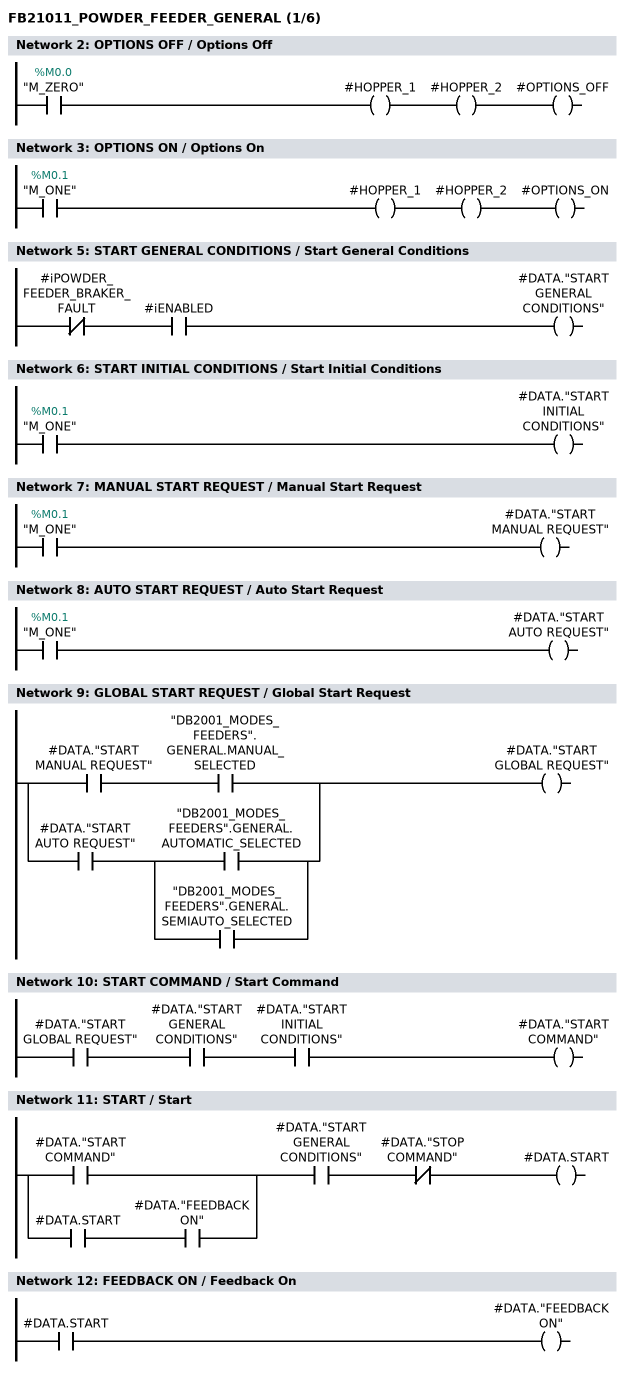
   RUNG wire#powerrail
      Contact( "M_ZERO" )
      Coil( #HOPPER_1 )
      Coil( #HOPPER_2 )
      Coil( #OPTIONS_OFF )
   END_RUNG
   // the same network as SCL:
   #HOPPER_1 := "M_ZERO";
   #HOPPER_2 := "M_ZERO";
   #OPTIONS_OFF := "M_ZERO";
END_REGION

REGION Network 3: OPTIONS ON / Options On
   RUNG wire#powerrail
      Contact( "M_ONE" )
      Coil( #HOPPER_1 )
      Coil( #HOPPER_2 )
      Coil( #OPTIONS_ON )
   END_RUNG
   // the same network as SCL:
   #HOPPER_1 := "M_ONE";
   #HOPPER_2 := "M_ONE";
   #OPTIONS_ON := "M_ONE";
END_REGION

REGION Network 4: INPUT / Input
END_REGION

REGION Network 5: START GENERAL CONDITIONS / Start General Conditions
   RUNG wire#powerrail
      I_Contact( #iPOWDER_FEEDER_BRAKER_FAULT )
      Contact( #iENABLED )
      Coil( #DATA."START GENERAL CONDITIONS" )
   END_RUNG
   // the same network as SCL:
   #DATA."START GENERAL CONDITIONS" := NOT #iPOWDER_FEEDER_BRAKER_FAULT AND #iENABLED;
END_REGION

REGION Network 6: START INITIAL CONDITIONS / Start Initial Conditions
   RUNG wire#powerrail
      Contact( "M_ONE" )
      Coil( #DATA."START INITIAL CONDITIONS" )
   END_RUNG
   // the same network as SCL:
   #DATA."START INITIAL CONDITIONS" := "M_ONE";
END_REGION

REGION Network 7: MANUAL START REQUEST / Manual Start Request
   RUNG wire#powerrail
      Contact( "M_ONE" )
      Coil( #DATA."START MANUAL REQUEST" )
   END_RUNG
   // the same network as SCL:
   #DATA."START MANUAL REQUEST" := "M_ONE";
END_REGION

REGION Network 8: AUTO START REQUEST / Auto Start Request
   RUNG wire#powerrail
      Contact( "M_ONE" )
      Coil( #DATA."START AUTO REQUEST" )
   END_RUNG
   // the same network as SCL:
   #DATA."START AUTO REQUEST" := "M_ONE";
END_REGION

REGION Network 9: GLOBAL START REQUEST / Global Start Request
   RUNG wire#powerrail
      Contact( #DATA."START MANUAL REQUEST" )
      Contact( "DB2001_MODES_FEEDERS".GENERAL.MANUAL_SELECTED )
      wire#w1
      Coil( #DATA."START GLOBAL REQUEST" )
   END_RUNG
   RUNG wire#powerrail
      Contact( #DATA."START AUTO REQUEST" )
      wire#w2
      Contact( "DB2001_MODES_FEEDERS".GENERAL.AUTOMATIC_SELECTED )
   END_RUNG wire#w1
   RUNG wire#w2
      Contact( "DB2001_MODES_FEEDERS".GENERAL.SEMIAUTO_SELECTED )
   END_RUNG wire#w1
   // the same network as SCL:
   #DATA."START GLOBAL REQUEST" := (#DATA."START MANUAL REQUEST" AND "DB2001_MODES_FEEDERS".GENERAL.MANUAL_SELECTED) OR (#DATA."START AUTO REQUEST" AND ("DB2001_MODES_FEEDERS".GENERAL.AUTOMATIC_SELECTED OR "DB2001_MODES_FEEDERS".GENERAL.SEMIAUTO_SELECTED));
END_REGION

REGION Network 10: START COMMAND / Start Command
   RUNG wire#powerrail
      Contact( #DATA."START GLOBAL REQUEST" )
      Contact( #DATA."START GENERAL CONDITIONS" )
      Contact( #DATA."START INITIAL CONDITIONS" )
      Coil( #DATA."START COMMAND" )
   END_RUNG
   // the same network as SCL:
   #DATA."START COMMAND" := #DATA."START GLOBAL REQUEST" AND #DATA."START GENERAL CONDITIONS" AND #DATA."START INITIAL CONDITIONS";
END_REGION

REGION Network 11: START / Start
   RUNG wire#powerrail
      Contact( #DATA."START COMMAND" )
      wire#w1
      Contact( #DATA."START GENERAL CONDITIONS" )
      I_Contact( #DATA."STOP COMMAND" )
      Coil( #DATA.START )
   END_RUNG
   RUNG wire#powerrail
      Contact( #DATA.START )
      Contact( #DATA."FEEDBACK ON" )
   END_RUNG wire#w1
   // the same network as SCL:
   #DATA.START := (#DATA."START COMMAND" OR (#DATA.START AND #DATA."FEEDBACK ON")) AND #DATA."START GENERAL CONDITIONS" AND NOT #DATA."STOP COMMAND";
END_REGION

REGION Network 12: FEEDBACK ON / Feedback On
   RUNG wire#powerrail
      Contact( #DATA.START )
      Coil( #DATA."FEEDBACK ON" )
   END_RUNG
   // the same network as SCL:
   #DATA."FEEDBACK ON" := #DATA.START;
END_REGION

REGION Network 13: STOP GENERAL CONDITIONS / Stop General Conditions
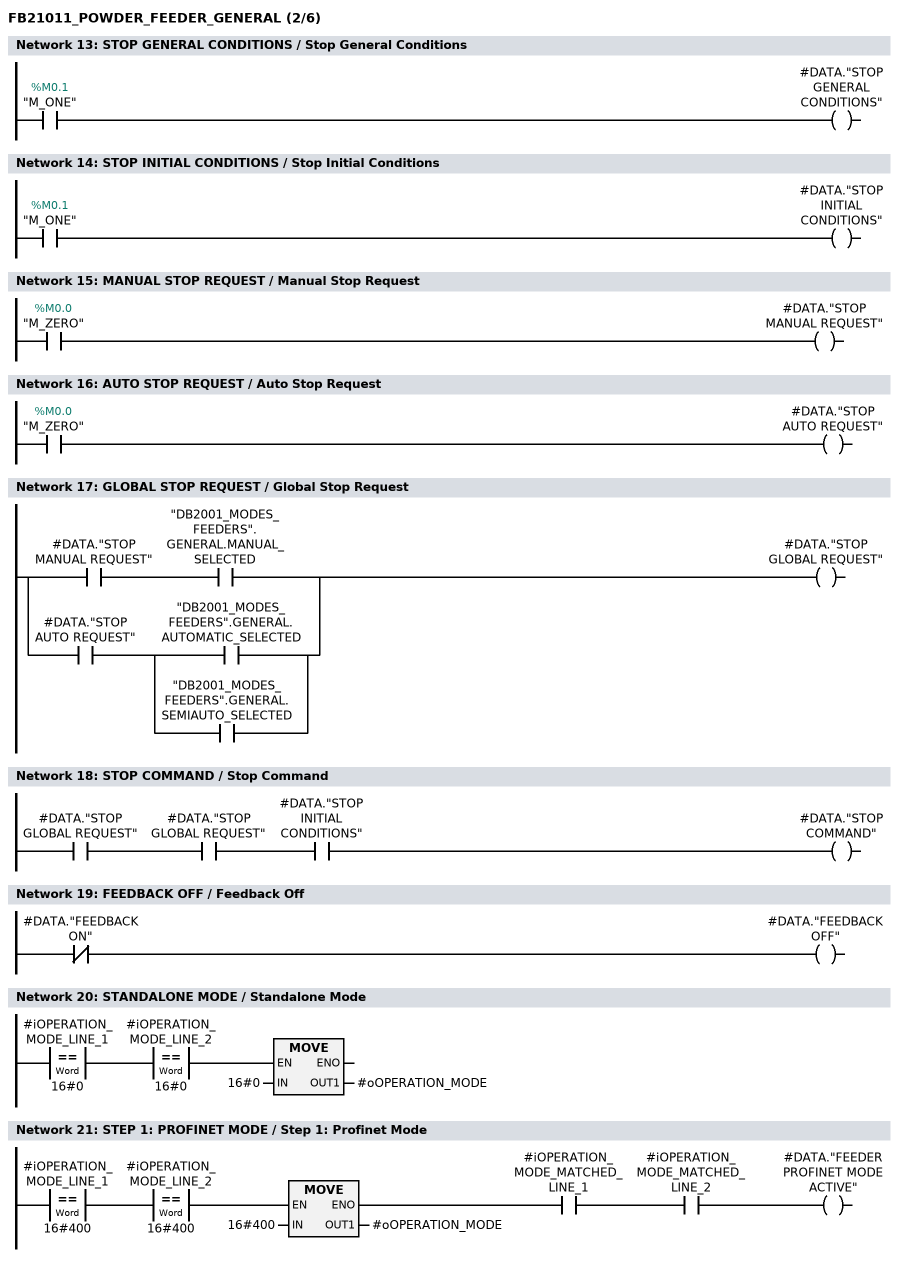
   RUNG wire#powerrail
      Contact( "M_ONE" )
      Coil( #DATA."STOP GENERAL CONDITIONS" )
   END_RUNG
   // the same network as SCL:
   #DATA."STOP GENERAL CONDITIONS" := "M_ONE";
END_REGION

REGION Network 14: STOP INITIAL CONDITIONS / Stop Initial Conditions
   RUNG wire#powerrail
      Contact( "M_ONE" )
      Coil( #DATA."STOP INITIAL CONDITIONS" )
   END_RUNG
   // the same network as SCL:
   #DATA."STOP INITIAL CONDITIONS" := "M_ONE";
END_REGION

REGION Network 15: MANUAL STOP REQUEST / Manual Stop Request
   RUNG wire#powerrail
      Contact( "M_ZERO" )
      Coil( #DATA."STOP MANUAL REQUEST" )
   END_RUNG
   // the same network as SCL:
   #DATA."STOP MANUAL REQUEST" := "M_ZERO";
END_REGION

REGION Network 16: AUTO STOP REQUEST / Auto Stop Request
   RUNG wire#powerrail
      Contact( "M_ZERO" )
      Coil( #DATA."STOP AUTO REQUEST" )
   END_RUNG
   // the same network as SCL:
   #DATA."STOP AUTO REQUEST" := "M_ZERO";
END_REGION

REGION Network 17: GLOBAL STOP REQUEST / Global Stop Request
   RUNG wire#powerrail
      Contact( #DATA."STOP MANUAL REQUEST" )
      Contact( "DB2001_MODES_FEEDERS".GENERAL.MANUAL_SELECTED )
      wire#w1
      Coil( #DATA."STOP GLOBAL REQUEST" )
   END_RUNG
   RUNG wire#powerrail
      Contact( #DATA."STOP AUTO REQUEST" )
      wire#w2
      Contact( "DB2001_MODES_FEEDERS".GENERAL.AUTOMATIC_SELECTED )
   END_RUNG wire#w1
   RUNG wire#w2
      Contact( "DB2001_MODES_FEEDERS".GENERAL.SEMIAUTO_SELECTED )
   END_RUNG wire#w1
   // the same network as SCL:
   #DATA."STOP GLOBAL REQUEST" := (#DATA."STOP MANUAL REQUEST" AND "DB2001_MODES_FEEDERS".GENERAL.MANUAL_SELECTED) OR (#DATA."STOP AUTO REQUEST" AND ("DB2001_MODES_FEEDERS".GENERAL.AUTOMATIC_SELECTED OR "DB2001_MODES_FEEDERS".GENERAL.SEMIAUTO_SELECTED));
END_REGION

REGION Network 18: STOP COMMAND / Stop Command
   RUNG wire#powerrail
      Contact( #DATA."STOP GLOBAL REQUEST" )
      Contact( #DATA."STOP GLOBAL REQUEST" )
      Contact( #DATA."STOP INITIAL CONDITIONS" )
      Coil( #DATA."STOP COMMAND" )
   END_RUNG
   // the same network as SCL:
   #DATA."STOP COMMAND" := #DATA."STOP GLOBAL REQUEST" AND #DATA."STOP GLOBAL REQUEST" AND #DATA."STOP INITIAL CONDITIONS";
END_REGION

REGION Network 19: FEEDBACK OFF / Feedback Off
   RUNG wire#powerrail
      I_Contact( #DATA."FEEDBACK ON" )
      Coil( #DATA."FEEDBACK OFF" )
   END_RUNG
   // the same network as SCL:
   #DATA."FEEDBACK OFF" := NOT #DATA."FEEDBACK ON";
END_REGION

REGION Network 20: STANDALONE MODE / Standalone Mode
   RUNG wire#powerrail
      { S7_Templates := "SrcType := Word" } EQ_Contact(in1 := #iOPERATION_MODE_LINE_1, in2 := 16#0)
      { S7_Templates := "SrcType := Word" } EQ_Contact(in1 := #iOPERATION_MODE_LINE_2, in2 := 16#0)
      Move(in := 16#0, out1 => #oOPERATION_MODE)
   END_RUNG
   // the same network as SCL:
   IF (#iOPERATION_MODE_LINE_1 = 16#0) AND (#iOPERATION_MODE_LINE_2 = 16#0) THEN
       #oOPERATION_MODE := 16#0;
   END_IF;
END_REGION

REGION Network 21: STEP 1: PROFINET MODE / Step 1: Profinet Mode
   RUNG wire#powerrail
      { S7_Templates := "SrcType := Word" } EQ_Contact(in1 := #iOPERATION_MODE_LINE_1, in2 := 16#400)
      { S7_Templates := "SrcType := Word" } EQ_Contact(in1 := #iOPERATION_MODE_LINE_2, in2 := 16#400)
      Move(in := 16#400, out1 => #oOPERATION_MODE)
      Contact( #iOPERATION_MODE_MATCHED_LINE_1 )
      Contact( #iOPERATION_MODE_MATCHED_LINE_2 )
      Coil( #DATA."FEEDER PROFINET MODE ACTIVE" )
   END_RUNG
   // the same network as SCL:
   #_w1 := (#iOPERATION_MODE_LINE_1 = 16#400) AND (#iOPERATION_MODE_LINE_2 = 16#400);
   IF #_w1 THEN #oOPERATION_MODE := 16#400; END_IF;
   #DATA."FEEDER PROFINET MODE ACTIVE" := #_w1 AND #iOPERATION_MODE_MATCHED_LINE_1 AND #iOPERATION_MODE_MATCHED_LINE_2;
END_REGION

REGION Network 22: STEP 2: PRODUCTION MODE / Step 2: Production Mode
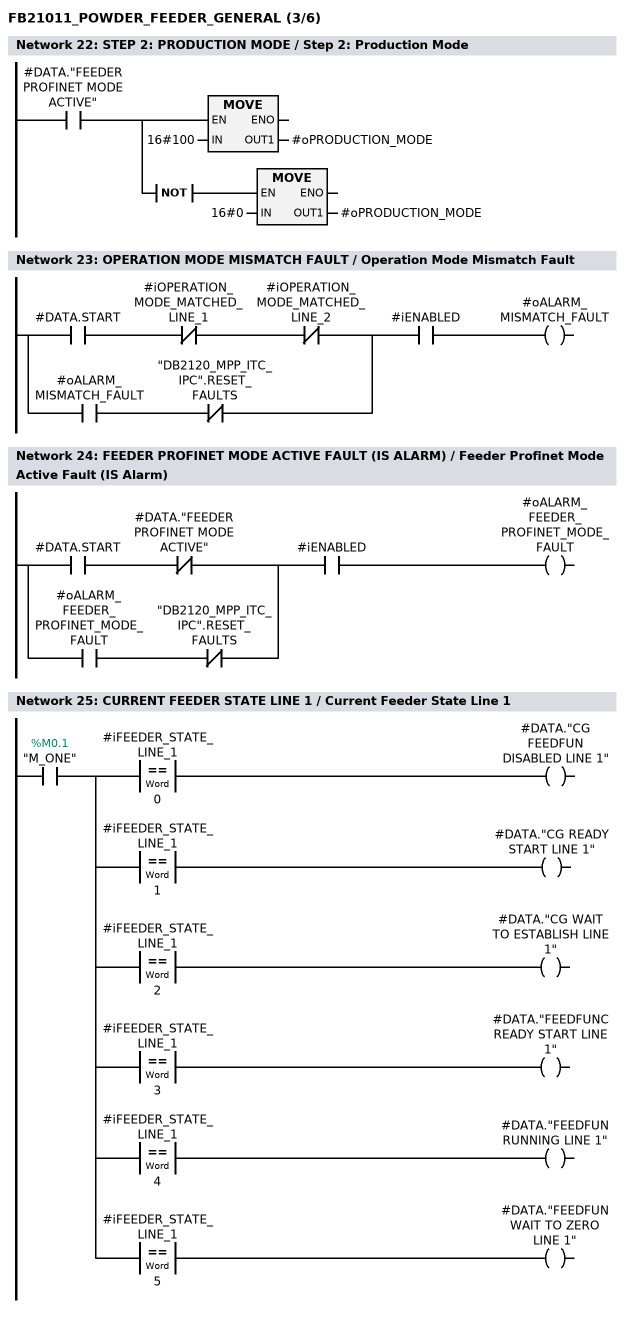
   RUNG wire#powerrail
      Contact( #DATA."FEEDER PROFINET MODE ACTIVE" )
      wire#w1
      Move(in := 16#100, out1 => #oPRODUCTION_MODE)
   END_RUNG
   RUNG wire#w1
      Not()
      Move(in := 16#0, out1 => #oPRODUCTION_MODE)
   END_RUNG
   // the same network as SCL:
   IF #DATA."FEEDER PROFINET MODE ACTIVE" THEN #oPRODUCTION_MODE := 16#100; END_IF;
   IF NOT #DATA."FEEDER PROFINET MODE ACTIVE" THEN #oPRODUCTION_MODE := 16#0; END_IF;
END_REGION

REGION Network 23: OPERATION MODE MISMATCH FAULT / Operation Mode Mismatch Fault
   RUNG wire#powerrail
      Contact( #DATA.START )
      I_Contact( #iOPERATION_MODE_MATCHED_LINE_1 )
      I_Contact( #iOPERATION_MODE_MATCHED_LINE_2 )
      wire#w1
      Contact( #iENABLED )
      Coil( #oALARM_MISMATCH_FAULT )
   END_RUNG
   RUNG wire#powerrail
      Contact( #oALARM_MISMATCH_FAULT )
      I_Contact( "DB2120_MPP_ITC_IPC".RESET_FAULTS )
   END_RUNG wire#w1
   // the same network as SCL:
   #oALARM_MISMATCH_FAULT := ((#DATA.START AND NOT #iOPERATION_MODE_MATCHED_LINE_1 AND NOT #iOPERATION_MODE_MATCHED_LINE_2) OR (#oALARM_MISMATCH_FAULT AND NOT "DB2120_MPP_ITC_IPC".RESET_FAULTS)) AND #iENABLED;
END_REGION

REGION Network 24: FEEDER PROFINET MODE ACTIVE FAULT (IS ALARM) / Feeder Profinet Mode Active Fault (IS Alarm)
   RUNG wire#powerrail
      Contact( #DATA.START )
      I_Contact( #DATA."FEEDER PROFINET MODE ACTIVE" )
      wire#w1
      Contact( #iENABLED )
      Coil( #oALARM_FEEDER_PROFINET_MODE_FAULT )
   END_RUNG
   RUNG wire#powerrail
      Contact( #oALARM_FEEDER_PROFINET_MODE_FAULT )
      I_Contact( "DB2120_MPP_ITC_IPC".RESET_FAULTS )
   END_RUNG wire#w1
   // the same network as SCL:
   #oALARM_FEEDER_PROFINET_MODE_FAULT := ((#DATA.START AND NOT #DATA."FEEDER PROFINET MODE ACTIVE") OR (#oALARM_FEEDER_PROFINET_MODE_FAULT AND NOT "DB2120_MPP_ITC_IPC".RESET_FAULTS)) AND #iENABLED;
END_REGION

REGION Network 25: CURRENT FEEDER STATE LINE 1 / Current Feeder State Line 1
   RUNG wire#powerrail
      Contact( "M_ONE" )
      wire#w1
      { S7_Templates := "SrcType := Word" } EQ_Contact(in1 := #iFEEDER_STATE_LINE_1, in2 := 0)
      Coil( #DATA."CG FEEDFUN DISABLED LINE 1" )
   END_RUNG
   RUNG wire#w1
      { S7_Templates := "SrcType := Word" } EQ_Contact(in1 := #iFEEDER_STATE_LINE_1, in2 := 1)
      Coil( #DATA."CG READY START LINE 1" )
   END_RUNG
   RUNG wire#w1
      { S7_Templates := "SrcType := Word" } EQ_Contact(in1 := #iFEEDER_STATE_LINE_1, in2 := 2)
      Coil( #DATA."CG WAIT TO ESTABLISH LINE 1" )
   END_RUNG
   RUNG wire#w1
      { S7_Templates := "SrcType := Word" } EQ_Contact(in1 := #iFEEDER_STATE_LINE_1, in2 := 3)
      Coil( #DATA."FEEDFUNC READY START LINE 1" )
   END_RUNG
   RUNG wire#w1
      { S7_Templates := "SrcType := Word" } EQ_Contact(in1 := #iFEEDER_STATE_LINE_1, in2 := 4)
      Coil( #DATA."FEEDFUN RUNNING LINE 1" )
   END_RUNG
   RUNG wire#w1
      { S7_Templates := "SrcType := Word" } EQ_Contact(in1 := #iFEEDER_STATE_LINE_1, in2 := 5)
      Coil( #DATA."FEEDFUN WAIT TO ZERO LINE 1" )
   END_RUNG
   // the same network as SCL:
   #DATA."CG FEEDFUN DISABLED LINE 1" := "M_ONE" AND (#iFEEDER_STATE_LINE_1 = 0);
   #DATA."CG READY START LINE 1" := "M_ONE" AND (#iFEEDER_STATE_LINE_1 = 1);
   #DATA."CG WAIT TO ESTABLISH LINE 1" := "M_ONE" AND (#iFEEDER_STATE_LINE_1 = 2);
   #DATA."FEEDFUNC READY START LINE 1" := "M_ONE" AND (#iFEEDER_STATE_LINE_1 = 3);
   #DATA."FEEDFUN RUNNING LINE 1" := "M_ONE" AND (#iFEEDER_STATE_LINE_1 = 4);
   #DATA."FEEDFUN WAIT TO ZERO LINE 1" := "M_ONE" AND (#iFEEDER_STATE_LINE_1 = 5);
END_REGION

REGION Network 26: CURRENT FEEDER STATE LINE 2 / Current Feeder State Line 2
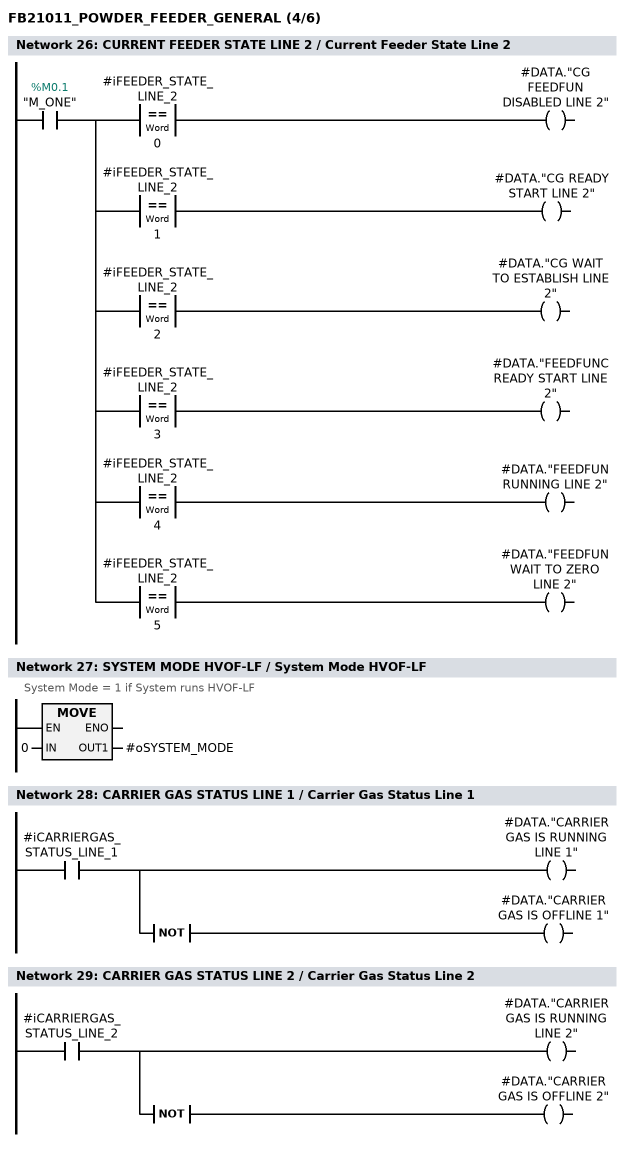
   RUNG wire#powerrail
      Contact( "M_ONE" )
      wire#w1
      { S7_Templates := "SrcType := Word" } EQ_Contact(in1 := #iFEEDER_STATE_LINE_2, in2 := 0)
      Coil( #DATA."CG FEEDFUN DISABLED LINE 2" )
   END_RUNG
   RUNG wire#w1
      { S7_Templates := "SrcType := Word" } EQ_Contact(in1 := #iFEEDER_STATE_LINE_2, in2 := 1)
      Coil( #DATA."CG READY START LINE 2" )
   END_RUNG
   RUNG wire#w1
      { S7_Templates := "SrcType := Word" } EQ_Contact(in1 := #iFEEDER_STATE_LINE_2, in2 := 2)
      Coil( #DATA."CG WAIT TO ESTABLISH LINE 2" )
   END_RUNG
   RUNG wire#w1
      { S7_Templates := "SrcType := Word" } EQ_Contact(in1 := #iFEEDER_STATE_LINE_2, in2 := 3)
      Coil( #DATA."FEEDFUNC READY START LINE 2" )
   END_RUNG
   RUNG wire#w1
      { S7_Templates := "SrcType := Word" } EQ_Contact(in1 := #iFEEDER_STATE_LINE_2, in2 := 4)
      Coil( #DATA."FEEDFUN RUNNING LINE 2" )
   END_RUNG
   RUNG wire#w1
      { S7_Templates := "SrcType := Word" } EQ_Contact(in1 := #iFEEDER_STATE_LINE_2, in2 := 5)
      Coil( #DATA."FEEDFUN WAIT TO ZERO LINE 2" )
   END_RUNG
   // the same network as SCL:
   #DATA."CG FEEDFUN DISABLED LINE 2" := "M_ONE" AND (#iFEEDER_STATE_LINE_2 = 0);
   #DATA."CG READY START LINE 2" := "M_ONE" AND (#iFEEDER_STATE_LINE_2 = 1);
   #DATA."CG WAIT TO ESTABLISH LINE 2" := "M_ONE" AND (#iFEEDER_STATE_LINE_2 = 2);
   #DATA."FEEDFUNC READY START LINE 2" := "M_ONE" AND (#iFEEDER_STATE_LINE_2 = 3);
   #DATA."FEEDFUN RUNNING LINE 2" := "M_ONE" AND (#iFEEDER_STATE_LINE_2 = 4);
   #DATA."FEEDFUN WAIT TO ZERO LINE 2" := "M_ONE" AND (#iFEEDER_STATE_LINE_2 = 5);
END_REGION

REGION Network 27: SYSTEM MODE HVOF-LF / System Mode HVOF-LF
   // System Mode = 1 if System runs HVOF-LF
   RUNG wire#powerrail
      Move(in := 0, out1 => #oSYSTEM_MODE)
   END_RUNG
   // the same network as SCL:
   #oSYSTEM_MODE := 0;
END_REGION

REGION Network 28: CARRIER GAS STATUS LINE 1 / Carrier Gas Status Line 1
   RUNG wire#powerrail
      Contact( #iCARRIERGAS_STATUS_LINE_1 )
      wire#w1
      Coil( #DATA."CARRIER GAS IS RUNNING LINE 1" )
   END_RUNG
   RUNG wire#w1
      Not()
      Coil( #DATA."CARRIER GAS IS OFFLINE 1" )
   END_RUNG
   // the same network as SCL:
   #DATA."CARRIER GAS IS RUNNING LINE 1" := #iCARRIERGAS_STATUS_LINE_1;
   #DATA."CARRIER GAS IS OFFLINE 1" := NOT #iCARRIERGAS_STATUS_LINE_1;
END_REGION

REGION Network 29: CARRIER GAS STATUS LINE 2 / Carrier Gas Status Line 2
   RUNG wire#powerrail
      Contact( #iCARRIERGAS_STATUS_LINE_2 )
      wire#w1
      Coil( #DATA."CARRIER GAS IS RUNNING LINE 2" )
   END_RUNG
   RUNG wire#w1
      Not()
      Coil( #DATA."CARRIER GAS IS OFFLINE 2" )
   END_RUNG
   // the same network as SCL:
   #DATA."CARRIER GAS IS RUNNING LINE 2" := #iCARRIERGAS_STATUS_LINE_2;
   #DATA."CARRIER GAS IS OFFLINE 2" := NOT #iCARRIERGAS_STATUS_LINE_2;
END_REGION

REGION Network 30: INMEDIATE STOP ALARMS / Inmediate Stop Alarms
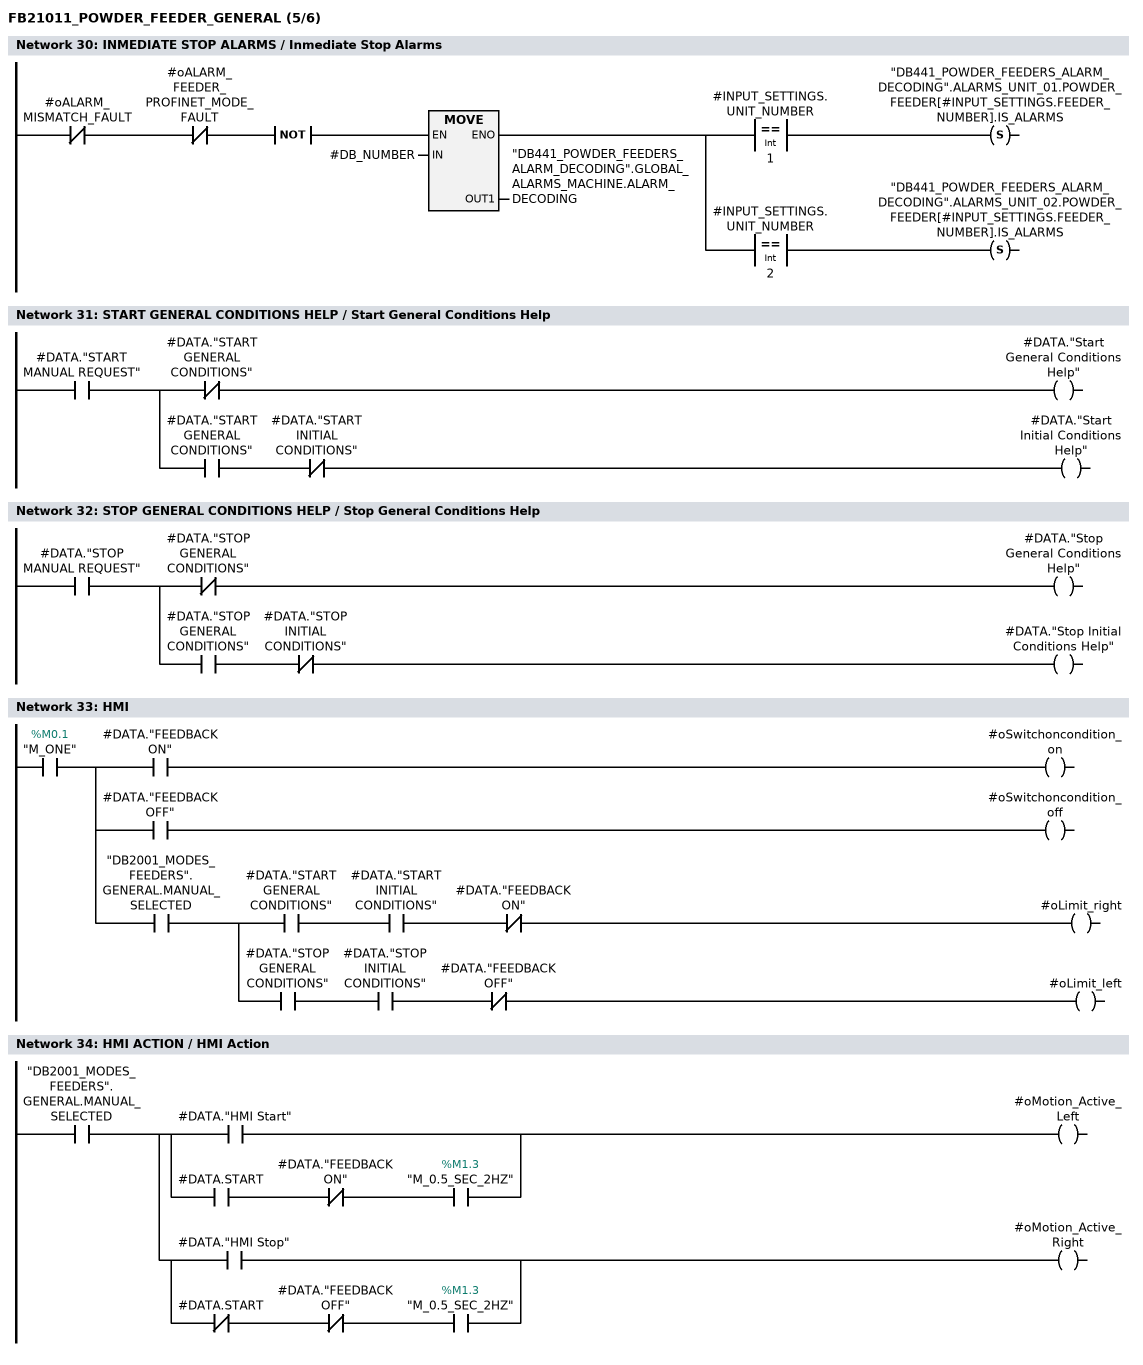
   RUNG wire#powerrail
      I_Contact( #oALARM_MISMATCH_FAULT )
      I_Contact( #oALARM_FEEDER_PROFINET_MODE_FAULT )
      Not()
      Move(in := #DB_NUMBER, out1 => "DB441_POWDER_FEEDERS_ALARM_DECODING".GLOBAL_ALARMS_MACHINE.ALARM_DECODING)
      wire#w1
      { S7_Templates := "SrcType := Int" } EQ_Contact(in1 := #INPUT_SETTINGS.UNIT_NUMBER, in2 := 1)
      S_Coil( "DB441_POWDER_FEEDERS_ALARM_DECODING".ALARMS_UNIT_01.POWDER_FEEDER[#INPUT_SETTINGS.FEEDER_NUMBER].IS_ALARMS )
   END_RUNG
   RUNG wire#w1
      { S7_Templates := "SrcType := Int" } EQ_Contact(in1 := #INPUT_SETTINGS.UNIT_NUMBER, in2 := 2)
      S_Coil( "DB441_POWDER_FEEDERS_ALARM_DECODING".ALARMS_UNIT_02.POWDER_FEEDER[#INPUT_SETTINGS.FEEDER_NUMBER].IS_ALARMS )
   END_RUNG
   // the same network as SCL:
   #_w1 := NOT (NOT #oALARM_MISMATCH_FAULT AND NOT #oALARM_FEEDER_PROFINET_MODE_FAULT);
   IF #_w1 THEN
       "DB441_POWDER_FEEDERS_ALARM_DECODING".GLOBAL_ALARMS_MACHINE.ALARM_DECODING := #DB_NUMBER;
   END_IF;
   IF #_w1 AND (#INPUT_SETTINGS.UNIT_NUMBER = 1) THEN
       "DB441_POWDER_FEEDERS_ALARM_DECODING".ALARMS_UNIT_01.POWDER_FEEDER[#INPUT_SETTINGS.FEEDER_NUMBER].IS_ALARMS := TRUE;
   END_IF;
   IF #_w1 AND (#INPUT_SETTINGS.UNIT_NUMBER = 2) THEN
       "DB441_POWDER_FEEDERS_ALARM_DECODING".ALARMS_UNIT_02.POWDER_FEEDER[#INPUT_SETTINGS.FEEDER_NUMBER].IS_ALARMS := TRUE;
   END_IF;
END_REGION

REGION Network 31: START GENERAL CONDITIONS HELP / Start General Conditions Help
   RUNG wire#powerrail
      Contact( #DATA."START MANUAL REQUEST" )
      wire#w1
      I_Contact( #DATA."START GENERAL CONDITIONS" )
      Coil( #DATA."Start General Conditions Help" )
   END_RUNG
   RUNG wire#w1
      Contact( #DATA."START GENERAL CONDITIONS" )
      I_Contact( #DATA."START INITIAL CONDITIONS" )
      Coil( #DATA."Start Initial Conditions Help" )
   END_RUNG
   // the same network as SCL:
   #DATA."Start General Conditions Help" := #DATA."START MANUAL REQUEST" AND NOT #DATA."START GENERAL CONDITIONS";
   #DATA."Start Initial Conditions Help" := #DATA."START MANUAL REQUEST" AND #DATA."START GENERAL CONDITIONS" AND NOT #DATA."START INITIAL CONDITIONS";
END_REGION

REGION Network 32: STOP GENERAL CONDITIONS HELP / Stop General Conditions Help
   RUNG wire#powerrail
      Contact( #DATA."STOP MANUAL REQUEST" )
      wire#w1
      I_Contact( #DATA."STOP GENERAL CONDITIONS" )
      Coil( #DATA."Stop General Conditions Help" )
   END_RUNG
   RUNG wire#w1
      Contact( #DATA."STOP GENERAL CONDITIONS" )
      I_Contact( #DATA."STOP INITIAL CONDITIONS" )
      Coil( #DATA."Stop Initial Conditions Help" )
   END_RUNG
   // the same network as SCL:
   #DATA."Stop General Conditions Help" := #DATA."STOP MANUAL REQUEST" AND NOT #DATA."STOP GENERAL CONDITIONS";
   #DATA."Stop Initial Conditions Help" := #DATA."STOP MANUAL REQUEST" AND #DATA."STOP GENERAL CONDITIONS" AND NOT #DATA."STOP INITIAL CONDITIONS";
END_REGION

REGION Network 33: HMI
   RUNG wire#powerrail
      Contact( "M_ONE" )
      wire#w1
      Contact( #DATA."FEEDBACK ON" )
      Coil( #oSwitchoncondition_on )
   END_RUNG
   RUNG wire#w1
      Contact( #DATA."FEEDBACK OFF" )
      Coil( #oSwitchoncondition_off )
   END_RUNG
   RUNG wire#w1
      Contact( "DB2001_MODES_FEEDERS".GENERAL.MANUAL_SELECTED )
      wire#w2
      Contact( #DATA."START GENERAL CONDITIONS" )
      Contact( #DATA."START INITIAL CONDITIONS" )
      I_Contact( #DATA."FEEDBACK ON" )
      Coil( #oLimit_right )
   END_RUNG
   RUNG wire#w2
      Contact( #DATA."STOP GENERAL CONDITIONS" )
      Contact( #DATA."STOP INITIAL CONDITIONS" )
      I_Contact( #DATA."FEEDBACK OFF" )
      Coil( #oLimit_left )
   END_RUNG
   // the same network as SCL:
   #oSwitchoncondition_on := "M_ONE" AND #DATA."FEEDBACK ON";
   #oSwitchoncondition_off := "M_ONE" AND #DATA."FEEDBACK OFF";
   #_w1 := "M_ONE" AND "DB2001_MODES_FEEDERS".GENERAL.MANUAL_SELECTED;
   #oLimit_right := #_w1 AND #DATA."START GENERAL CONDITIONS" AND #DATA."START INITIAL CONDITIONS" AND NOT #DATA."FEEDBACK ON";
   #oLimit_left := #_w1 AND #DATA."STOP GENERAL CONDITIONS" AND #DATA."STOP INITIAL CONDITIONS" AND NOT #DATA."FEEDBACK OFF";
END_REGION

REGION Network 34: HMI ACTION / HMI Action
   RUNG wire#powerrail
      Contact( "DB2001_MODES_FEEDERS".GENERAL.MANUAL_SELECTED )
      wire#w1
      Contact( #DATA."HMI Start" )
      wire#w2
      Coil( #oMotion_Active_Left )
   END_RUNG
   RUNG wire#w1
      Contact( #DATA.START )
      I_Contact( #DATA."FEEDBACK ON" )
      Contact( "M_0.5_SEC_2HZ" )
   END_RUNG wire#w2
   RUNG wire#w1
      Contact( #DATA."HMI Stop" )
      wire#w3
      Coil( #oMotion_Active_Right )
   END_RUNG
   RUNG wire#w1
      I_Contact( #DATA.START )
      I_Contact( #DATA."FEEDBACK OFF" )
      Contact( "M_0.5_SEC_2HZ" )
   END_RUNG wire#w3
   // the same network as SCL:
   #oMotion_Active_Left := "DB2001_MODES_FEEDERS".GENERAL.MANUAL_SELECTED AND (#DATA."HMI Start" OR (#DATA.START AND NOT #DATA."FEEDBACK ON" AND "M_0.5_SEC_2HZ"));
   #oMotion_Active_Right := "DB2001_MODES_FEEDERS".GENERAL.MANUAL_SELECTED AND (#DATA."HMI Stop" OR (NOT #DATA.START AND NOT #DATA."FEEDBACK OFF" AND "M_0.5_SEC_2HZ"));
END_REGION

REGION Network 35: FEEDBACK ON AUX FOR HMI / Feedback On Aux for HMI
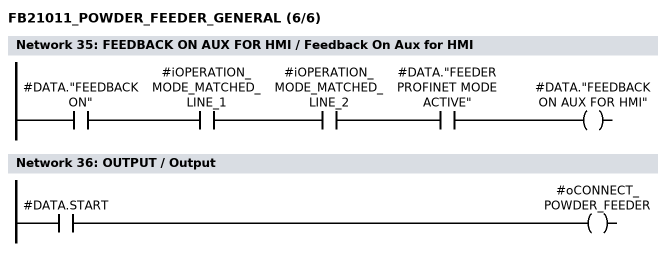
   RUNG wire#powerrail
      Contact( #DATA."FEEDBACK ON" )
      Contact( #iOPERATION_MODE_MATCHED_LINE_1 )
      Contact( #iOPERATION_MODE_MATCHED_LINE_2 )
      Contact( #DATA."FEEDER PROFINET MODE ACTIVE" )
      Coil( #DATA."FEEDBACK ON AUX FOR HMI" )
   END_RUNG
   // the same network as SCL:
   #DATA."FEEDBACK ON AUX FOR HMI" := #DATA."FEEDBACK ON" AND #iOPERATION_MODE_MATCHED_LINE_1 AND #iOPERATION_MODE_MATCHED_LINE_2 AND #DATA."FEEDER PROFINET MODE ACTIVE";
END_REGION

REGION Network 36: OUTPUT / Output
   RUNG wire#powerrail
      Contact( #DATA.START )
      Coil( #oCONNECT_POWDER_FEEDER )
   END_RUNG
   // the same network as SCL:
   #oCONNECT_POWDER_FEEDER := #DATA.START;
END_REGION
END_FUNCTION_BLOCK

FUNCTION "FC21012_POWDER_FEEDER_HEATER_JKL" : Void   // FC21012, LAD
TITLE = FC21012 POWDER FEEDER HEATER JKL
{ S7_Optimized_Access := 'TRUE' }
VERSION : 0.1
// stored: AutoNumber false, IsIECCheckEnabled false, SetENOAutomatically false, UDAEnableTagReadback false
BEGIN

REGION Network 1: /////_UNIT_01_/////
END_REGION

REGION Network 2: CALL FB21012 POWDER FEEDER 1 HEATER JKL UNIT 01
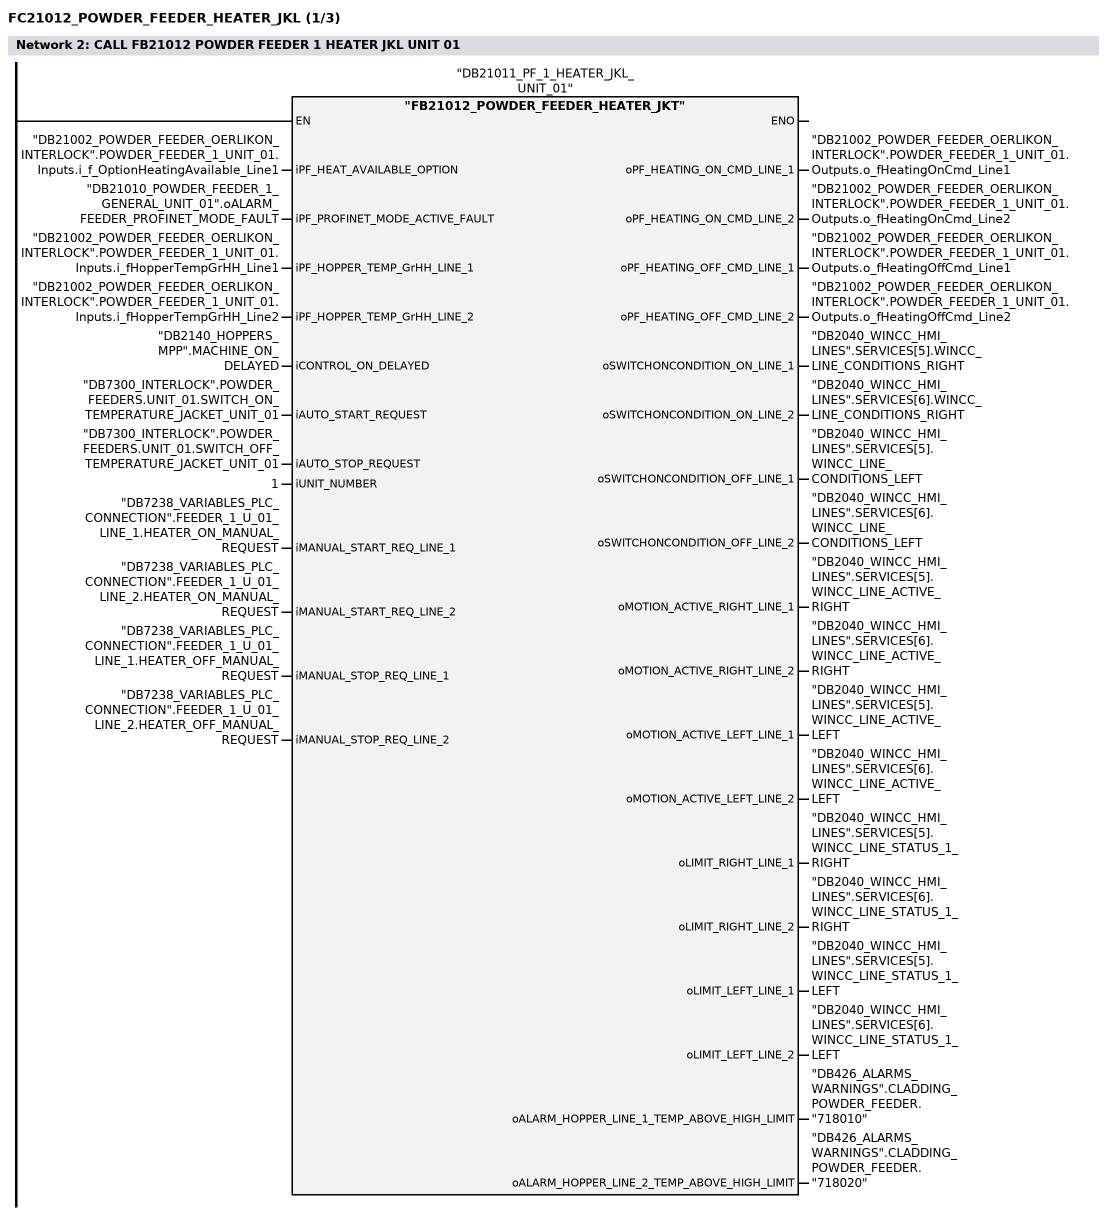
   RUNG wire#powerrail
      "DB21011_PF_1_HEATER_JKL_UNIT_01"(iPF_HEAT_AVAILABLE_OPTION := "DB21002_POWDER_FEEDER_OERLIKON_INTERLOCK".POWDER_FEEDER_1_UNIT_01.Inputs.i_f_OptionHeatingAvailable_Line1, iPF_PROFINET_MODE_ACTIVE_FAULT := "DB21010_POWDER_FEEDER_1_GENERAL_UNIT_01".oALARM_FEEDER_PROFINET_MODE_FAULT, iPF_HOPPER_TEMP_GrHH_LINE_1 := "DB21002_POWDER_FEEDER_OERLIKON_INTERLOCK".POWDER_FEEDER_1_UNIT_01.Inputs.i_fHopperTempGrHH_Line1, iPF_HOPPER_TEMP_GrHH_LINE_2 := "DB21002_POWDER_FEEDER_OERLIKON_INTERLOCK".POWDER_FEEDER_1_UNIT_01.Inputs.i_fHopperTempGrHH_Line2, iCONTROL_ON_DELAYED := "DB2140_HOPPERS_MPP".MACHINE_ON_DELAYED, iAUTO_START_REQUEST := "DB7300_INTERLOCK".POWDER_FEEDERS.UNIT_01.SWITCH_ON_TEMPERATURE_JACKET_UNIT_01, iAUTO_STOP_REQUEST := "DB7300_INTERLOCK".POWDER_FEEDERS.UNIT_01.SWITCH_OFF_TEMPERATURE_JACKET_UNIT_01, iUNIT_NUMBER := 1, iMANUAL_START_REQ_LINE_1 := "DB7238_VARIABLES_PLC_CONNECTION".FEEDER_1_U_01_LINE_1.HEATER_ON_MANUAL_REQUEST, iMANUAL_START_REQ_LINE_2 := "DB7238_VARIABLES_PLC_CONNECTION".FEEDER_1_U_01_LINE_2.HEATER_ON_MANUAL_REQUEST, iMANUAL_STOP_REQ_LINE_1 := "DB7238_VARIABLES_PLC_CONNECTION".FEEDER_1_U_01_LINE_1.HEATER_OFF_MANUAL_REQUEST, iMANUAL_STOP_REQ_LINE_2 := "DB7238_VARIABLES_PLC_CONNECTION".FEEDER_1_U_01_LINE_2.HEATER_OFF_MANUAL_REQUEST, oPF_HEATING_ON_CMD_LINE_1 => "DB21002_POWDER_FEEDER_OERLIKON_INTERLOCK".POWDER_FEEDER_1_UNIT_01.Outputs.o_fHeatingOnCmd_Line1, oPF_HEATING_ON_CMD_LINE_2 => "DB21002_POWDER_FEEDER_OERLIKON_INTERLOCK".POWDER_FEEDER_1_UNIT_01.Outputs.o_fHeatingOnCmd_Line2, oPF_HEATING_OFF_CMD_LINE_1 => "DB21002_POWDER_FEEDER_OERLIKON_INTERLOCK".POWDER_FEEDER_1_UNIT_01.Outputs.o_fHeatingOffCmd_Line1, oPF_HEATING_OFF_CMD_LINE_2 => "DB21002_POWDER_FEEDER_OERLIKON_INTERLOCK".POWDER_FEEDER_1_UNIT_01.Outputs.o_fHeatingOffCmd_Line2, oSWITCHONCONDITION_ON_LINE_1 => "DB2040_WINCC_HMI_LINES".SERVICES[5].WINCC_LINE_CONDITIONS_RIGHT, oSWITCHONCONDITION_ON_LINE_2 => "DB2040_WINCC_HMI_LINES".SERVICES[6].WINCC_LINE_CONDITIONS_RIGHT, oSWITCHONCONDITION_OFF_LINE_1 => "DB2040_WINCC_HMI_LINES".SERVICES[5].WINCC_LINE_CONDITIONS_LEFT, oSWITCHONCONDITION_OFF_LINE_2 => "DB2040_WINCC_HMI_LINES".SERVICES[6].WINCC_LINE_CONDITIONS_LEFT, oMOTION_ACTIVE_RIGHT_LINE_1 => "DB2040_WINCC_HMI_LINES".SERVICES[5].WINCC_LINE_ACTIVE_RIGHT, oMOTION_ACTIVE_RIGHT_LINE_2 => "DB2040_WINCC_HMI_LINES".SERVICES[6].WINCC_LINE_ACTIVE_RIGHT, oMOTION_ACTIVE_LEFT_LINE_1 => "DB2040_WINCC_HMI_LINES".SERVICES[5].WINCC_LINE_ACTIVE_LEFT, oMOTION_ACTIVE_LEFT_LINE_2 => "DB2040_WINCC_HMI_LINES".SERVICES[6].WINCC_LINE_ACTIVE_LEFT, oLIMIT_RIGHT_LINE_1 => "DB2040_WINCC_HMI_LINES".SERVICES[5].WINCC_LINE_STATUS_1_RIGHT, oLIMIT_RIGHT_LINE_2 => "DB2040_WINCC_HMI_LINES".SERVICES[6].WINCC_LINE_STATUS_1_RIGHT, oLIMIT_LEFT_LINE_1 => "DB2040_WINCC_HMI_LINES".SERVICES[5].WINCC_LINE_STATUS_1_LEFT, oLIMIT_LEFT_LINE_2 => "DB2040_WINCC_HMI_LINES".SERVICES[6].WINCC_LINE_STATUS_1_LEFT, oALARM_HOPPER_LINE_1_TEMP_ABOVE_HIGH_LIMIT => "DB426_ALARMS_WARNINGS".CLADDING_POWDER_FEEDER."718010", oALARM_HOPPER_LINE_2_TEMP_ABOVE_HIGH_LIMIT => "DB426_ALARMS_WARNINGS".CLADDING_POWDER_FEEDER."718020")
   END_RUNG
   // the same network as SCL:
   "DB21011_PF_1_HEATER_JKL_UNIT_01"(iPF_HEAT_AVAILABLE_OPTION := "DB21002_POWDER_FEEDER_OERLIKON_INTERLOCK".POWDER_FEEDER_1_UNIT_01.Inputs.i_f_OptionHeatingAvailable_Line1,   // "FB21012_POWDER_FEEDER_HEATER_JKT"
                           iPF_PROFINET_MODE_ACTIVE_FAULT := "DB21010_POWDER_FEEDER_1_GENERAL_UNIT_01".oALARM_FEEDER_PROFINET_MODE_FAULT,
                           iPF_HOPPER_TEMP_GrHH_LINE_1 := "DB21002_POWDER_FEEDER_OERLIKON_INTERLOCK".POWDER_FEEDER_1_UNIT_01.Inputs.i_fHopperTempGrHH_Line1,
                           iPF_HOPPER_TEMP_GrHH_LINE_2 := "DB21002_POWDER_FEEDER_OERLIKON_INTERLOCK".POWDER_FEEDER_1_UNIT_01.Inputs.i_fHopperTempGrHH_Line2,
                           iCONTROL_ON_DELAYED := "DB2140_HOPPERS_MPP".MACHINE_ON_DELAYED,
                           iAUTO_START_REQUEST := "DB7300_INTERLOCK".POWDER_FEEDERS.UNIT_01.SWITCH_ON_TEMPERATURE_JACKET_UNIT_01,
                           iAUTO_STOP_REQUEST := "DB7300_INTERLOCK".POWDER_FEEDERS.UNIT_01.SWITCH_OFF_TEMPERATURE_JACKET_UNIT_01,
                           iUNIT_NUMBER := 1,
                           iMANUAL_START_REQ_LINE_1 := "DB7238_VARIABLES_PLC_CONNECTION".FEEDER_1_U_01_LINE_1.HEATER_ON_MANUAL_REQUEST,
                           iMANUAL_START_REQ_LINE_2 := "DB7238_VARIABLES_PLC_CONNECTION".FEEDER_1_U_01_LINE_2.HEATER_ON_MANUAL_REQUEST,
                           iMANUAL_STOP_REQ_LINE_1 := "DB7238_VARIABLES_PLC_CONNECTION".FEEDER_1_U_01_LINE_1.HEATER_OFF_MANUAL_REQUEST,
                           iMANUAL_STOP_REQ_LINE_2 := "DB7238_VARIABLES_PLC_CONNECTION".FEEDER_1_U_01_LINE_2.HEATER_OFF_MANUAL_REQUEST,
                           oPF_HEATING_ON_CMD_LINE_1 => "DB21002_POWDER_FEEDER_OERLIKON_INTERLOCK".POWDER_FEEDER_1_UNIT_01.Outputs.o_fHeatingOnCmd_Line1,
                           oPF_HEATING_ON_CMD_LINE_2 => "DB21002_POWDER_FEEDER_OERLIKON_INTERLOCK".POWDER_FEEDER_1_UNIT_01.Outputs.o_fHeatingOnCmd_Line2,
                           oPF_HEATING_OFF_CMD_LINE_1 => "DB21002_POWDER_FEEDER_OERLIKON_INTERLOCK".POWDER_FEEDER_1_UNIT_01.Outputs.o_fHeatingOffCmd_Line1,
                           oPF_HEATING_OFF_CMD_LINE_2 => "DB21002_POWDER_FEEDER_OERLIKON_INTERLOCK".POWDER_FEEDER_1_UNIT_01.Outputs.o_fHeatingOffCmd_Line2,
                           oSWITCHONCONDITION_ON_LINE_1 => "DB2040_WINCC_HMI_LINES".SERVICES[5].WINCC_LINE_CONDITIONS_RIGHT,
                           oSWITCHONCONDITION_ON_LINE_2 => "DB2040_WINCC_HMI_LINES".SERVICES[6].WINCC_LINE_CONDITIONS_RIGHT,
                           oSWITCHONCONDITION_OFF_LINE_1 => "DB2040_WINCC_HMI_LINES".SERVICES[5].WINCC_LINE_CONDITIONS_LEFT,
                           oSWITCHONCONDITION_OFF_LINE_2 => "DB2040_WINCC_HMI_LINES".SERVICES[6].WINCC_LINE_CONDITIONS_LEFT,
                           oMOTION_ACTIVE_RIGHT_LINE_1 => "DB2040_WINCC_HMI_LINES".SERVICES[5].WINCC_LINE_ACTIVE_RIGHT,
                           oMOTION_ACTIVE_RIGHT_LINE_2 => "DB2040_WINCC_HMI_LINES".SERVICES[6].WINCC_LINE_ACTIVE_RIGHT,
                           oMOTION_ACTIVE_LEFT_LINE_1 => "DB2040_WINCC_HMI_LINES".SERVICES[5].WINCC_LINE_ACTIVE_LEFT,
                           oMOTION_ACTIVE_LEFT_LINE_2 => "DB2040_WINCC_HMI_LINES".SERVICES[6].WINCC_LINE_ACTIVE_LEFT,
                           oLIMIT_RIGHT_LINE_1 => "DB2040_WINCC_HMI_LINES".SERVICES[5].WINCC_LINE_STATUS_1_RIGHT,
                           oLIMIT_RIGHT_LINE_2 => "DB2040_WINCC_HMI_LINES".SERVICES[6].WINCC_LINE_STATUS_1_RIGHT,
                           oLIMIT_LEFT_LINE_1 => "DB2040_WINCC_HMI_LINES".SERVICES[5].WINCC_LINE_STATUS_1_LEFT,
                           oLIMIT_LEFT_LINE_2 => "DB2040_WINCC_HMI_LINES".SERVICES[6].WINCC_LINE_STATUS_1_LEFT,
                           oALARM_HOPPER_LINE_1_TEMP_ABOVE_HIGH_LIMIT => "DB426_ALARMS_WARNINGS".CLADDING_POWDER_FEEDER."718010",
                           oALARM_HOPPER_LINE_2_TEMP_ABOVE_HIGH_LIMIT => "DB426_ALARMS_WARNINGS".CLADDING_POWDER_FEEDER."718020");
END_REGION

REGION Network 3: /////_UNIT_02_/////
END_REGION

REGION Network 4: CALL FB21012 POWDER FEEDER 1 HEATER JKL UNIT 02
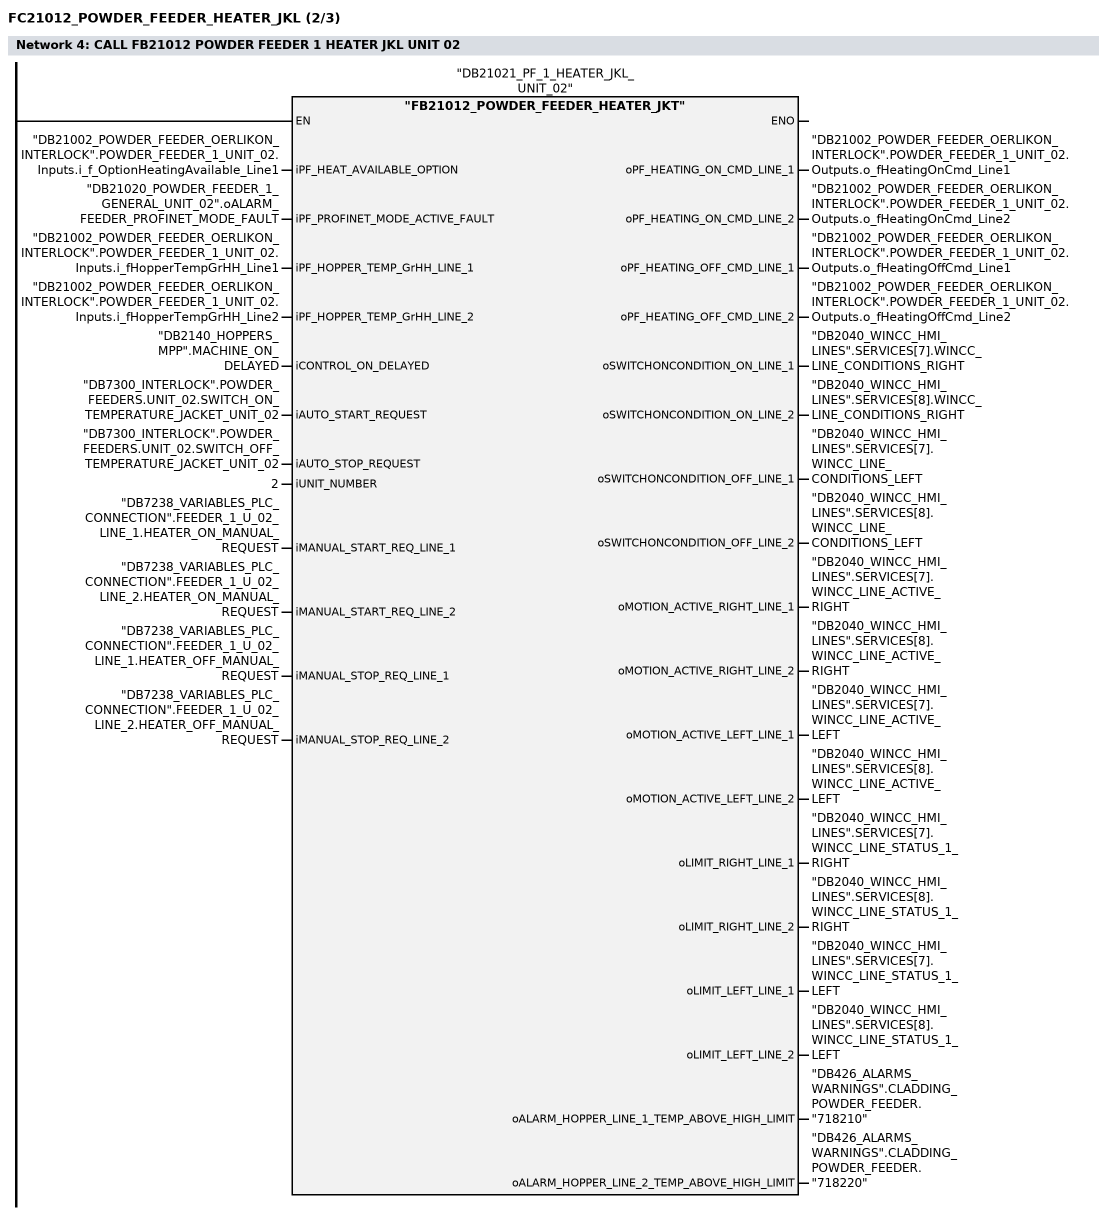
   RUNG wire#powerrail
      "DB21021_PF_1_HEATER_JKL_UNIT_02"(iPF_HEAT_AVAILABLE_OPTION := "DB21002_POWDER_FEEDER_OERLIKON_INTERLOCK".POWDER_FEEDER_1_UNIT_02.Inputs.i_f_OptionHeatingAvailable_Line1, iPF_PROFINET_MODE_ACTIVE_FAULT := "DB21020_POWDER_FEEDER_1_GENERAL_UNIT_02".oALARM_FEEDER_PROFINET_MODE_FAULT, iPF_HOPPER_TEMP_GrHH_LINE_1 := "DB21002_POWDER_FEEDER_OERLIKON_INTERLOCK".POWDER_FEEDER_1_UNIT_02.Inputs.i_fHopperTempGrHH_Line1, iPF_HOPPER_TEMP_GrHH_LINE_2 := "DB21002_POWDER_FEEDER_OERLIKON_INTERLOCK".POWDER_FEEDER_1_UNIT_02.Inputs.i_fHopperTempGrHH_Line2, iCONTROL_ON_DELAYED := "DB2140_HOPPERS_MPP".MACHINE_ON_DELAYED, iAUTO_START_REQUEST := "DB7300_INTERLOCK".POWDER_FEEDERS.UNIT_02.SWITCH_ON_TEMPERATURE_JACKET_UNIT_02, iAUTO_STOP_REQUEST := "DB7300_INTERLOCK".POWDER_FEEDERS.UNIT_02.SWITCH_OFF_TEMPERATURE_JACKET_UNIT_02, iUNIT_NUMBER := 2, iMANUAL_START_REQ_LINE_1 := "DB7238_VARIABLES_PLC_CONNECTION".FEEDER_1_U_02_LINE_1.HEATER_ON_MANUAL_REQUEST, iMANUAL_START_REQ_LINE_2 := "DB7238_VARIABLES_PLC_CONNECTION".FEEDER_1_U_02_LINE_2.HEATER_ON_MANUAL_REQUEST, iMANUAL_STOP_REQ_LINE_1 := "DB7238_VARIABLES_PLC_CONNECTION".FEEDER_1_U_02_LINE_1.HEATER_OFF_MANUAL_REQUEST, iMANUAL_STOP_REQ_LINE_2 := "DB7238_VARIABLES_PLC_CONNECTION".FEEDER_1_U_02_LINE_2.HEATER_OFF_MANUAL_REQUEST, oPF_HEATING_ON_CMD_LINE_1 => "DB21002_POWDER_FEEDER_OERLIKON_INTERLOCK".POWDER_FEEDER_1_UNIT_02.Outputs.o_fHeatingOnCmd_Line1, oPF_HEATING_ON_CMD_LINE_2 => "DB21002_POWDER_FEEDER_OERLIKON_INTERLOCK".POWDER_FEEDER_1_UNIT_02.Outputs.o_fHeatingOnCmd_Line2, oPF_HEATING_OFF_CMD_LINE_1 => "DB21002_POWDER_FEEDER_OERLIKON_INTERLOCK".POWDER_FEEDER_1_UNIT_02.Outputs.o_fHeatingOffCmd_Line1, oPF_HEATING_OFF_CMD_LINE_2 => "DB21002_POWDER_FEEDER_OERLIKON_INTERLOCK".POWDER_FEEDER_1_UNIT_02.Outputs.o_fHeatingOffCmd_Line2, oSWITCHONCONDITION_ON_LINE_1 => "DB2040_WINCC_HMI_LINES".SERVICES[7].WINCC_LINE_CONDITIONS_RIGHT, oSWITCHONCONDITION_ON_LINE_2 => "DB2040_WINCC_HMI_LINES".SERVICES[8].WINCC_LINE_CONDITIONS_RIGHT, oSWITCHONCONDITION_OFF_LINE_1 => "DB2040_WINCC_HMI_LINES".SERVICES[7].WINCC_LINE_CONDITIONS_LEFT, oSWITCHONCONDITION_OFF_LINE_2 => "DB2040_WINCC_HMI_LINES".SERVICES[8].WINCC_LINE_CONDITIONS_LEFT, oMOTION_ACTIVE_RIGHT_LINE_1 => "DB2040_WINCC_HMI_LINES".SERVICES[7].WINCC_LINE_ACTIVE_RIGHT, oMOTION_ACTIVE_RIGHT_LINE_2 => "DB2040_WINCC_HMI_LINES".SERVICES[8].WINCC_LINE_ACTIVE_RIGHT, oMOTION_ACTIVE_LEFT_LINE_1 => "DB2040_WINCC_HMI_LINES".SERVICES[7].WINCC_LINE_ACTIVE_LEFT, oMOTION_ACTIVE_LEFT_LINE_2 => "DB2040_WINCC_HMI_LINES".SERVICES[8].WINCC_LINE_ACTIVE_LEFT, oLIMIT_RIGHT_LINE_1 => "DB2040_WINCC_HMI_LINES".SERVICES[7].WINCC_LINE_STATUS_1_RIGHT, oLIMIT_RIGHT_LINE_2 => "DB2040_WINCC_HMI_LINES".SERVICES[8].WINCC_LINE_STATUS_1_RIGHT, oLIMIT_LEFT_LINE_1 => "DB2040_WINCC_HMI_LINES".SERVICES[7].WINCC_LINE_STATUS_1_LEFT, oLIMIT_LEFT_LINE_2 => "DB2040_WINCC_HMI_LINES".SERVICES[8].WINCC_LINE_STATUS_1_LEFT, oALARM_HOPPER_LINE_1_TEMP_ABOVE_HIGH_LIMIT => "DB426_ALARMS_WARNINGS".CLADDING_POWDER_FEEDER."718210", oALARM_HOPPER_LINE_2_TEMP_ABOVE_HIGH_LIMIT => "DB426_ALARMS_WARNINGS".CLADDING_POWDER_FEEDER."718220")
   END_RUNG
   // the same network as SCL:
   "DB21021_PF_1_HEATER_JKL_UNIT_02"(iPF_HEAT_AVAILABLE_OPTION := "DB21002_POWDER_FEEDER_OERLIKON_INTERLOCK".POWDER_FEEDER_1_UNIT_02.Inputs.i_f_OptionHeatingAvailable_Line1,   // "FB21012_POWDER_FEEDER_HEATER_JKT"
                           iPF_PROFINET_MODE_ACTIVE_FAULT := "DB21020_POWDER_FEEDER_1_GENERAL_UNIT_02".oALARM_FEEDER_PROFINET_MODE_FAULT,
                           iPF_HOPPER_TEMP_GrHH_LINE_1 := "DB21002_POWDER_FEEDER_OERLIKON_INTERLOCK".POWDER_FEEDER_1_UNIT_02.Inputs.i_fHopperTempGrHH_Line1,
                           iPF_HOPPER_TEMP_GrHH_LINE_2 := "DB21002_POWDER_FEEDER_OERLIKON_INTERLOCK".POWDER_FEEDER_1_UNIT_02.Inputs.i_fHopperTempGrHH_Line2,
                           iCONTROL_ON_DELAYED := "DB2140_HOPPERS_MPP".MACHINE_ON_DELAYED,
                           iAUTO_START_REQUEST := "DB7300_INTERLOCK".POWDER_FEEDERS.UNIT_02.SWITCH_ON_TEMPERATURE_JACKET_UNIT_02,
                           iAUTO_STOP_REQUEST := "DB7300_INTERLOCK".POWDER_FEEDERS.UNIT_02.SWITCH_OFF_TEMPERATURE_JACKET_UNIT_02,
                           iUNIT_NUMBER := 2,
                           iMANUAL_START_REQ_LINE_1 := "DB7238_VARIABLES_PLC_CONNECTION".FEEDER_1_U_02_LINE_1.HEATER_ON_MANUAL_REQUEST,
                           iMANUAL_START_REQ_LINE_2 := "DB7238_VARIABLES_PLC_CONNECTION".FEEDER_1_U_02_LINE_2.HEATER_ON_MANUAL_REQUEST,
                           iMANUAL_STOP_REQ_LINE_1 := "DB7238_VARIABLES_PLC_CONNECTION".FEEDER_1_U_02_LINE_1.HEATER_OFF_MANUAL_REQUEST,
                           iMANUAL_STOP_REQ_LINE_2 := "DB7238_VARIABLES_PLC_CONNECTION".FEEDER_1_U_02_LINE_2.HEATER_OFF_MANUAL_REQUEST,
                           oPF_HEATING_ON_CMD_LINE_1 => "DB21002_POWDER_FEEDER_OERLIKON_INTERLOCK".POWDER_FEEDER_1_UNIT_02.Outputs.o_fHeatingOnCmd_Line1,
                           oPF_HEATING_ON_CMD_LINE_2 => "DB21002_POWDER_FEEDER_OERLIKON_INTERLOCK".POWDER_FEEDER_1_UNIT_02.Outputs.o_fHeatingOnCmd_Line2,
                           oPF_HEATING_OFF_CMD_LINE_1 => "DB21002_POWDER_FEEDER_OERLIKON_INTERLOCK".POWDER_FEEDER_1_UNIT_02.Outputs.o_fHeatingOffCmd_Line1,
                           oPF_HEATING_OFF_CMD_LINE_2 => "DB21002_POWDER_FEEDER_OERLIKON_INTERLOCK".POWDER_FEEDER_1_UNIT_02.Outputs.o_fHeatingOffCmd_Line2,
                           oSWITCHONCONDITION_ON_LINE_1 => "DB2040_WINCC_HMI_LINES".SERVICES[7].WINCC_LINE_CONDITIONS_RIGHT,
                           oSWITCHONCONDITION_ON_LINE_2 => "DB2040_WINCC_HMI_LINES".SERVICES[8].WINCC_LINE_CONDITIONS_RIGHT,
                           oSWITCHONCONDITION_OFF_LINE_1 => "DB2040_WINCC_HMI_LINES".SERVICES[7].WINCC_LINE_CONDITIONS_LEFT,
                           oSWITCHONCONDITION_OFF_LINE_2 => "DB2040_WINCC_HMI_LINES".SERVICES[8].WINCC_LINE_CONDITIONS_LEFT,
                           oMOTION_ACTIVE_RIGHT_LINE_1 => "DB2040_WINCC_HMI_LINES".SERVICES[7].WINCC_LINE_ACTIVE_RIGHT,
                           oMOTION_ACTIVE_RIGHT_LINE_2 => "DB2040_WINCC_HMI_LINES".SERVICES[8].WINCC_LINE_ACTIVE_RIGHT,
                           oMOTION_ACTIVE_LEFT_LINE_1 => "DB2040_WINCC_HMI_LINES".SERVICES[7].WINCC_LINE_ACTIVE_LEFT,
                           oMOTION_ACTIVE_LEFT_LINE_2 => "DB2040_WINCC_HMI_LINES".SERVICES[8].WINCC_LINE_ACTIVE_LEFT,
                           oLIMIT_RIGHT_LINE_1 => "DB2040_WINCC_HMI_LINES".SERVICES[7].WINCC_LINE_STATUS_1_RIGHT,
                           oLIMIT_RIGHT_LINE_2 => "DB2040_WINCC_HMI_LINES".SERVICES[8].WINCC_LINE_STATUS_1_RIGHT,
                           oLIMIT_LEFT_LINE_1 => "DB2040_WINCC_HMI_LINES".SERVICES[7].WINCC_LINE_STATUS_1_LEFT,
                           oLIMIT_LEFT_LINE_2 => "DB2040_WINCC_HMI_LINES".SERVICES[8].WINCC_LINE_STATUS_1_LEFT,
                           oALARM_HOPPER_LINE_1_TEMP_ABOVE_HIGH_LIMIT => "DB426_ALARMS_WARNINGS".CLADDING_POWDER_FEEDER."718210",
                           oALARM_HOPPER_LINE_2_TEMP_ABOVE_HIGH_LIMIT => "DB426_ALARMS_WARNINGS".CLADDING_POWDER_FEEDER."718220");
END_REGION

REGION Network 5: CALL FB21012 POWDER FEEDER 2 HEATER JKL UNIT 02
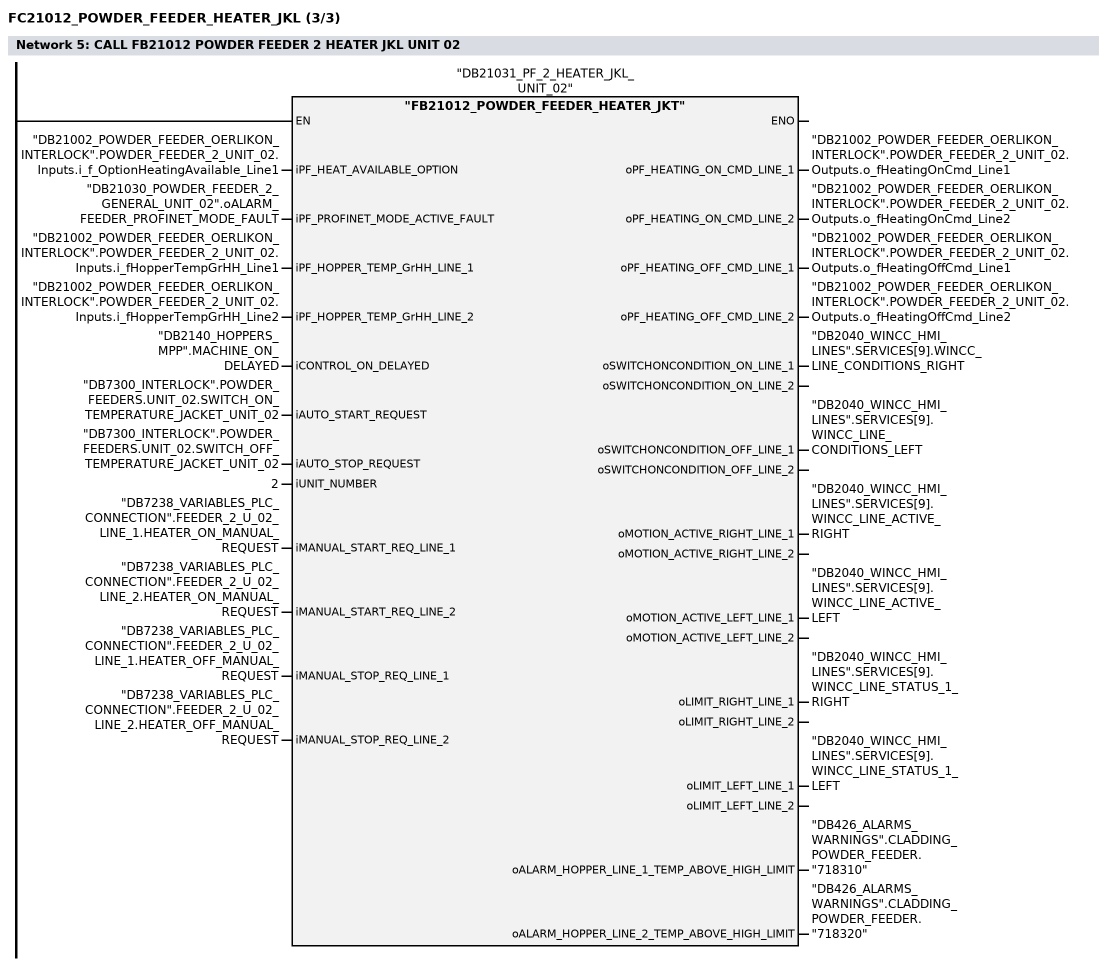
   RUNG wire#powerrail
      "DB21031_PF_2_HEATER_JKL_UNIT_02"(iPF_HEAT_AVAILABLE_OPTION := "DB21002_POWDER_FEEDER_OERLIKON_INTERLOCK".POWDER_FEEDER_2_UNIT_02.Inputs.i_f_OptionHeatingAvailable_Line1, iPF_PROFINET_MODE_ACTIVE_FAULT := "DB21030_POWDER_FEEDER_2_GENERAL_UNIT_02".oALARM_FEEDER_PROFINET_MODE_FAULT, iPF_HOPPER_TEMP_GrHH_LINE_1 := "DB21002_POWDER_FEEDER_OERLIKON_INTERLOCK".POWDER_FEEDER_2_UNIT_02.Inputs.i_fHopperTempGrHH_Line1, iPF_HOPPER_TEMP_GrHH_LINE_2 := "DB21002_POWDER_FEEDER_OERLIKON_INTERLOCK".POWDER_FEEDER_2_UNIT_02.Inputs.i_fHopperTempGrHH_Line2, iCONTROL_ON_DELAYED := "DB2140_HOPPERS_MPP".MACHINE_ON_DELAYED, iAUTO_START_REQUEST := "DB7300_INTERLOCK".POWDER_FEEDERS.UNIT_02.SWITCH_ON_TEMPERATURE_JACKET_UNIT_02, iAUTO_STOP_REQUEST := "DB7300_INTERLOCK".POWDER_FEEDERS.UNIT_02.SWITCH_OFF_TEMPERATURE_JACKET_UNIT_02, iUNIT_NUMBER := 2, iMANUAL_START_REQ_LINE_1 := "DB7238_VARIABLES_PLC_CONNECTION".FEEDER_2_U_02_LINE_1.HEATER_ON_MANUAL_REQUEST, iMANUAL_START_REQ_LINE_2 := "DB7238_VARIABLES_PLC_CONNECTION".FEEDER_2_U_02_LINE_2.HEATER_ON_MANUAL_REQUEST, iMANUAL_STOP_REQ_LINE_1 := "DB7238_VARIABLES_PLC_CONNECTION".FEEDER_2_U_02_LINE_1.HEATER_OFF_MANUAL_REQUEST, iMANUAL_STOP_REQ_LINE_2 := "DB7238_VARIABLES_PLC_CONNECTION".FEEDER_2_U_02_LINE_2.HEATER_OFF_MANUAL_REQUEST, oPF_HEATING_ON_CMD_LINE_1 => "DB21002_POWDER_FEEDER_OERLIKON_INTERLOCK".POWDER_FEEDER_2_UNIT_02.Outputs.o_fHeatingOnCmd_Line1, oPF_HEATING_ON_CMD_LINE_2 => "DB21002_POWDER_FEEDER_OERLIKON_INTERLOCK".POWDER_FEEDER_2_UNIT_02.Outputs.o_fHeatingOnCmd_Line2, oPF_HEATING_OFF_CMD_LINE_1 => "DB21002_POWDER_FEEDER_OERLIKON_INTERLOCK".POWDER_FEEDER_2_UNIT_02.Outputs.o_fHeatingOffCmd_Line1, oPF_HEATING_OFF_CMD_LINE_2 => "DB21002_POWDER_FEEDER_OERLIKON_INTERLOCK".POWDER_FEEDER_2_UNIT_02.Outputs.o_fHeatingOffCmd_Line2, oSWITCHONCONDITION_ON_LINE_1 => "DB2040_WINCC_HMI_LINES".SERVICES[9].WINCC_LINE_CONDITIONS_RIGHT, oSWITCHONCONDITION_ON_LINE_2 =>, oSWITCHONCONDITION_OFF_LINE_1 => "DB2040_WINCC_HMI_LINES".SERVICES[9].WINCC_LINE_CONDITIONS_LEFT, oSWITCHONCONDITION_OFF_LINE_2 =>, oMOTION_ACTIVE_RIGHT_LINE_1 => "DB2040_WINCC_HMI_LINES".SERVICES[9].WINCC_LINE_ACTIVE_RIGHT, oMOTION_ACTIVE_RIGHT_LINE_2 =>, oMOTION_ACTIVE_LEFT_LINE_1 => "DB2040_WINCC_HMI_LINES".SERVICES[9].WINCC_LINE_ACTIVE_LEFT, oMOTION_ACTIVE_LEFT_LINE_2 =>, oLIMIT_RIGHT_LINE_1 => "DB2040_WINCC_HMI_LINES".SERVICES[9].WINCC_LINE_STATUS_1_RIGHT, oLIMIT_RIGHT_LINE_2 =>, oLIMIT_LEFT_LINE_1 => "DB2040_WINCC_HMI_LINES".SERVICES[9].WINCC_LINE_STATUS_1_LEFT, oLIMIT_LEFT_LINE_2 =>, oALARM_HOPPER_LINE_1_TEMP_ABOVE_HIGH_LIMIT => "DB426_ALARMS_WARNINGS".CLADDING_POWDER_FEEDER."718310", oALARM_HOPPER_LINE_2_TEMP_ABOVE_HIGH_LIMIT => "DB426_ALARMS_WARNINGS".CLADDING_POWDER_FEEDER."718320")
   END_RUNG
   // the same network as SCL:
   "DB21031_PF_2_HEATER_JKL_UNIT_02"(iPF_HEAT_AVAILABLE_OPTION := "DB21002_POWDER_FEEDER_OERLIKON_INTERLOCK".POWDER_FEEDER_2_UNIT_02.Inputs.i_f_OptionHeatingAvailable_Line1,   // "FB21012_POWDER_FEEDER_HEATER_JKT"
                           iPF_PROFINET_MODE_ACTIVE_FAULT := "DB21030_POWDER_FEEDER_2_GENERAL_UNIT_02".oALARM_FEEDER_PROFINET_MODE_FAULT,
                           iPF_HOPPER_TEMP_GrHH_LINE_1 := "DB21002_POWDER_FEEDER_OERLIKON_INTERLOCK".POWDER_FEEDER_2_UNIT_02.Inputs.i_fHopperTempGrHH_Line1,
                           iPF_HOPPER_TEMP_GrHH_LINE_2 := "DB21002_POWDER_FEEDER_OERLIKON_INTERLOCK".POWDER_FEEDER_2_UNIT_02.Inputs.i_fHopperTempGrHH_Line2,
                           iCONTROL_ON_DELAYED := "DB2140_HOPPERS_MPP".MACHINE_ON_DELAYED,
                           iAUTO_START_REQUEST := "DB7300_INTERLOCK".POWDER_FEEDERS.UNIT_02.SWITCH_ON_TEMPERATURE_JACKET_UNIT_02,
                           iAUTO_STOP_REQUEST := "DB7300_INTERLOCK".POWDER_FEEDERS.UNIT_02.SWITCH_OFF_TEMPERATURE_JACKET_UNIT_02,
                           iUNIT_NUMBER := 2,
                           iMANUAL_START_REQ_LINE_1 := "DB7238_VARIABLES_PLC_CONNECTION".FEEDER_2_U_02_LINE_1.HEATER_ON_MANUAL_REQUEST,
                           iMANUAL_START_REQ_LINE_2 := "DB7238_VARIABLES_PLC_CONNECTION".FEEDER_2_U_02_LINE_2.HEATER_ON_MANUAL_REQUEST,
                           iMANUAL_STOP_REQ_LINE_1 := "DB7238_VARIABLES_PLC_CONNECTION".FEEDER_2_U_02_LINE_1.HEATER_OFF_MANUAL_REQUEST,
                           iMANUAL_STOP_REQ_LINE_2 := "DB7238_VARIABLES_PLC_CONNECTION".FEEDER_2_U_02_LINE_2.HEATER_OFF_MANUAL_REQUEST,
                           oPF_HEATING_ON_CMD_LINE_1 => "DB21002_POWDER_FEEDER_OERLIKON_INTERLOCK".POWDER_FEEDER_2_UNIT_02.Outputs.o_fHeatingOnCmd_Line1,
                           oPF_HEATING_ON_CMD_LINE_2 => "DB21002_POWDER_FEEDER_OERLIKON_INTERLOCK".POWDER_FEEDER_2_UNIT_02.Outputs.o_fHeatingOnCmd_Line2,
                           oPF_HEATING_OFF_CMD_LINE_1 => "DB21002_POWDER_FEEDER_OERLIKON_INTERLOCK".POWDER_FEEDER_2_UNIT_02.Outputs.o_fHeatingOffCmd_Line1,
                           oPF_HEATING_OFF_CMD_LINE_2 => "DB21002_POWDER_FEEDER_OERLIKON_INTERLOCK".POWDER_FEEDER_2_UNIT_02.Outputs.o_fHeatingOffCmd_Line2,
                           oSWITCHONCONDITION_ON_LINE_1 => "DB2040_WINCC_HMI_LINES".SERVICES[9].WINCC_LINE_CONDITIONS_RIGHT,
                           oSWITCHONCONDITION_OFF_LINE_1 => "DB2040_WINCC_HMI_LINES".SERVICES[9].WINCC_LINE_CONDITIONS_LEFT,
                           oMOTION_ACTIVE_RIGHT_LINE_1 => "DB2040_WINCC_HMI_LINES".SERVICES[9].WINCC_LINE_ACTIVE_RIGHT,
                           oMOTION_ACTIVE_LEFT_LINE_1 => "DB2040_WINCC_HMI_LINES".SERVICES[9].WINCC_LINE_ACTIVE_LEFT,
                           oLIMIT_RIGHT_LINE_1 => "DB2040_WINCC_HMI_LINES".SERVICES[9].WINCC_LINE_STATUS_1_RIGHT,
                           oLIMIT_LEFT_LINE_1 => "DB2040_WINCC_HMI_LINES".SERVICES[9].WINCC_LINE_STATUS_1_LEFT,
                           oALARM_HOPPER_LINE_1_TEMP_ABOVE_HIGH_LIMIT => "DB426_ALARMS_WARNINGS".CLADDING_POWDER_FEEDER."718310",
                           oALARM_HOPPER_LINE_2_TEMP_ABOVE_HIGH_LIMIT => "DB426_ALARMS_WARNINGS".CLADDING_POWDER_FEEDER."718320");
END_REGION
END_FUNCTION

FUNCTION_BLOCK "FB21012_POWDER_FEEDER_HEATER_JKT"   // FB21012, LAD
TITLE = FB21012 POWDER FEEDER HEATER JKT
{ S7_Optimized_Access := 'FALSE' }
VERSION : 0.1
// stored: AutoNumber false, IsIECCheckEnabled false, SetENOAutomatically false, UDAEnableTagReadback false
   VAR_INPUT
      iPF_HEAT_AVAILABLE_OPTION : Bool;
      iPF_PROFINET_MODE_ACTIVE_FAULT : Bool;
      iPF_HOPPER_TEMP_GrHH_LINE_1 : Bool;   // POWDER FEEDER HOPPER TEMPERATURE LINE 1 ALARM
      iPF_HOPPER_TEMP_GrHH_LINE_2 : Bool;   // POWDER FEEDER HOPPER TEMPERATURE LINE 2 ALARM
      iCONTROL_ON_DELAYED : Bool;   // LOCAL MACHINE ON
      iAUTO_START_REQUEST : Bool;   // AUTO START REQUEST
      iAUTO_STOP_REQUEST : Bool;   // AUTO STOP SEQUEST
      iUNIT_NUMBER : Byte;
      iMANUAL_START_REQ_LINE_1 : Bool;
      iMANUAL_START_REQ_LINE_2 : Bool;
      iMANUAL_STOP_REQ_LINE_1 : Bool;
      iMANUAL_STOP_REQ_LINE_2 : Bool;
   END_VAR
   VAR_OUTPUT
      oPF_HEATING_ON_CMD_LINE_1 : Bool;   // POWDER FEEDER HEATING ON COMMAND LINE 1
      oPF_HEATING_ON_CMD_LINE_2 : Bool;   // POWDER FEEDER HEATING ON COMMAND LINE 2
      oPF_HEATING_OFF_CMD_LINE_1 : Bool;   // POWDER FEEDER HEATING OF COMMAND LINE 1
      oPF_HEATING_OFF_CMD_LINE_2 : Bool;   // POWDER FEEDER HEATING OF COMMAND LINE 2
      oSWITCHONCONDITION_ON_LINE_1 : Bool;
      oSWITCHONCONDITION_ON_LINE_2 : Bool;
      oSWITCHONCONDITION_OFF_LINE_1 : Bool;
      oSWITCHONCONDITION_OFF_LINE_2 : Bool;
      oMOTION_ACTIVE_RIGHT_LINE_1 : Bool;
      oMOTION_ACTIVE_RIGHT_LINE_2 : Bool;
      oMOTION_ACTIVE_LEFT_LINE_1 : Bool;
      oMOTION_ACTIVE_LEFT_LINE_2 : Bool;
      oLIMIT_RIGHT_LINE_1 : Bool;
      oLIMIT_RIGHT_LINE_2 : Bool;
      oLIMIT_LEFT_LINE_1 : Bool;
      oLIMIT_LEFT_LINE_2 : Bool;
      oALARM_HOPPER_LINE_1_TEMP_ABOVE_HIGH_LIMIT : Bool;
      oALARM_HOPPER_LINE_2_TEMP_ABOVE_HIGH_LIMIT : Bool;
   END_VAR
   VAR DB_SPECIFIC
      DATA : "POWDER FEEDER HEATER JKT";
      INPUT_SETTINGS : Struct
         UNIT_NUMBER : Int;
         FEEDER_NUMBER : Int;
      END_STRUCT;
      HEATER_STATUS_LINE_1 { S7_SetPoint := 'True'} : Byte;
      HEATER_STATUS_LINE_2 : Byte;
   END_VAR
   VAR_TEMP
      DB_NUMBER : DInt;
   END_VAR
   VAR_TEMP   // added for the SCL form of the ladder/FBD networks
      _w1 : Bool;
      _w2 : Bool;
   END_VAR
BEGIN

NETWORK
TITLE = READ INSTANCE DB NUMBER
      L     DINO;
      +     10#800000;
      T     #DB_NUMBER;

REGION Network 2: START GENERAL CONDITIONS / Start General Conditions
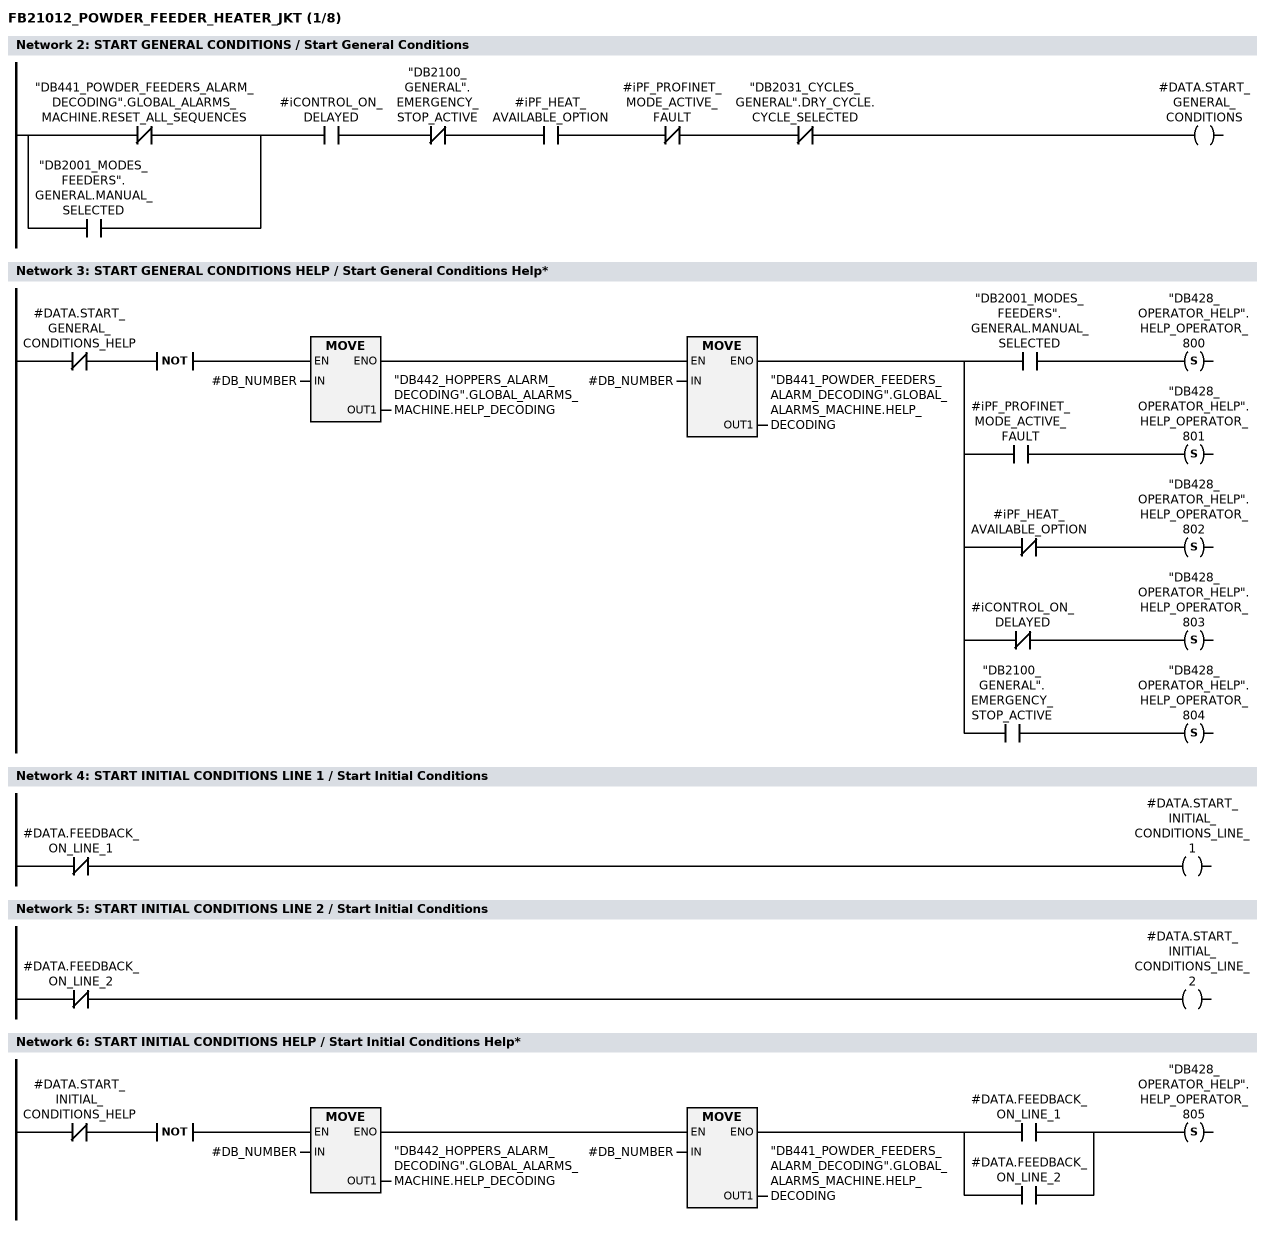
   RUNG wire#powerrail
      I_Contact( "DB441_POWDER_FEEDERS_ALARM_DECODING".GLOBAL_ALARMS_MACHINE.RESET_ALL_SEQUENCES )
      wire#w1
      Contact( #iCONTROL_ON_DELAYED )
      I_Contact( "DB2100_GENERAL".EMERGENCY_STOP_ACTIVE )
      Contact( #iPF_HEAT_AVAILABLE_OPTION )
      I_Contact( #iPF_PROFINET_MODE_ACTIVE_FAULT )
      I_Contact( "DB2031_CYCLES_GENERAL".DRY_CYCLE.CYCLE_SELECTED )
      Coil( #DATA.START_GENERAL_CONDITIONS )
   END_RUNG
   RUNG wire#powerrail
      Contact( "DB2001_MODES_FEEDERS".GENERAL.MANUAL_SELECTED )
   END_RUNG wire#w1
   // the same network as SCL:
   #DATA.START_GENERAL_CONDITIONS := (NOT "DB441_POWDER_FEEDERS_ALARM_DECODING".GLOBAL_ALARMS_MACHINE.RESET_ALL_SEQUENCES OR "DB2001_MODES_FEEDERS".GENERAL.MANUAL_SELECTED) AND #iCONTROL_ON_DELAYED AND NOT "DB2100_GENERAL".EMERGENCY_STOP_ACTIVE AND #iPF_HEAT_AVAILABLE_OPTION AND NOT #iPF_PROFINET_MODE_ACTIVE_FAULT AND NOT "DB2031_CYCLES_GENERAL".DRY_CYCLE.CYCLE_SELECTED;
END_REGION

REGION Network 3: START GENERAL CONDITIONS HELP / Start General Conditions Help*
   RUNG wire#powerrail
      I_Contact( #DATA.START_GENERAL_CONDITIONS_HELP )
      Not()
      Move(in := #DB_NUMBER, out1 => "DB442_HOPPERS_ALARM_DECODING".GLOBAL_ALARMS_MACHINE.HELP_DECODING)
      Move(in := #DB_NUMBER, out1 => "DB441_POWDER_FEEDERS_ALARM_DECODING".GLOBAL_ALARMS_MACHINE.HELP_DECODING)
      wire#w1
      Contact( "DB2001_MODES_FEEDERS".GENERAL.MANUAL_SELECTED )
      S_Coil( "DB428_OPERATOR_HELP".HELP_OPERATOR_800 )
   END_RUNG
   RUNG wire#w1
      Contact( #iPF_PROFINET_MODE_ACTIVE_FAULT )
      S_Coil( "DB428_OPERATOR_HELP".HELP_OPERATOR_801 )
   END_RUNG
   RUNG wire#w1
      I_Contact( #iPF_HEAT_AVAILABLE_OPTION )
      S_Coil( "DB428_OPERATOR_HELP".HELP_OPERATOR_802 )
   END_RUNG
   RUNG wire#w1
      I_Contact( #iCONTROL_ON_DELAYED )
      S_Coil( "DB428_OPERATOR_HELP".HELP_OPERATOR_803 )
   END_RUNG
   RUNG wire#w1
      Contact( "DB2100_GENERAL".EMERGENCY_STOP_ACTIVE )
      S_Coil( "DB428_OPERATOR_HELP".HELP_OPERATOR_804 )
   END_RUNG
   // the same network as SCL:
   #_w1 := NOT (NOT #DATA.START_GENERAL_CONDITIONS_HELP);
   IF #_w1 THEN
       "DB442_HOPPERS_ALARM_DECODING".GLOBAL_ALARMS_MACHINE.HELP_DECODING := #DB_NUMBER;
       "DB441_POWDER_FEEDERS_ALARM_DECODING".GLOBAL_ALARMS_MACHINE.HELP_DECODING := #DB_NUMBER;
   END_IF;
   IF #_w1 AND "DB2001_MODES_FEEDERS".GENERAL.MANUAL_SELECTED THEN
       "DB428_OPERATOR_HELP".HELP_OPERATOR_800 := TRUE;
   END_IF;
   IF #_w1 AND #iPF_PROFINET_MODE_ACTIVE_FAULT THEN "DB428_OPERATOR_HELP".HELP_OPERATOR_801 := TRUE; END_IF;
   IF #_w1 AND NOT #iPF_HEAT_AVAILABLE_OPTION THEN "DB428_OPERATOR_HELP".HELP_OPERATOR_802 := TRUE; END_IF;
   IF #_w1 AND NOT #iCONTROL_ON_DELAYED THEN "DB428_OPERATOR_HELP".HELP_OPERATOR_803 := TRUE; END_IF;
   IF #_w1 AND "DB2100_GENERAL".EMERGENCY_STOP_ACTIVE THEN
       "DB428_OPERATOR_HELP".HELP_OPERATOR_804 := TRUE;
   END_IF;
END_REGION

REGION Network 4: START INITIAL CONDITIONS LINE 1 / Start Initial Conditions
   RUNG wire#powerrail
      I_Contact( #DATA.FEEDBACK_ON_LINE_1 )
      Coil( #DATA.START_INITIAL_CONDITIONS_LINE_1 )
   END_RUNG
   // the same network as SCL:
   #DATA.START_INITIAL_CONDITIONS_LINE_1 := NOT #DATA.FEEDBACK_ON_LINE_1;
END_REGION

REGION Network 5: START INITIAL CONDITIONS LINE 2 / Start Initial Conditions
   RUNG wire#powerrail
      I_Contact( #DATA.FEEDBACK_ON_LINE_2 )
      Coil( #DATA.START_INITIAL_CONDITIONS_LINE_2 )
   END_RUNG
   // the same network as SCL:
   #DATA.START_INITIAL_CONDITIONS_LINE_2 := NOT #DATA.FEEDBACK_ON_LINE_2;
END_REGION

REGION Network 6: START INITIAL CONDITIONS HELP / Start Initial Conditions Help*
   RUNG wire#powerrail
      I_Contact( #DATA.START_INITIAL_CONDITIONS_HELP )
      Not()
      Move(in := #DB_NUMBER, out1 => "DB442_HOPPERS_ALARM_DECODING".GLOBAL_ALARMS_MACHINE.HELP_DECODING)
      Move(in := #DB_NUMBER, out1 => "DB441_POWDER_FEEDERS_ALARM_DECODING".GLOBAL_ALARMS_MACHINE.HELP_DECODING)
      wire#w1
      Contact( #DATA.FEEDBACK_ON_LINE_1 )
      wire#w2
      S_Coil( "DB428_OPERATOR_HELP".HELP_OPERATOR_805 )
   END_RUNG
   RUNG wire#w1
      Contact( #DATA.FEEDBACK_ON_LINE_2 )
   END_RUNG wire#w2
   // the same network as SCL:
   #_w1 := NOT (NOT #DATA.START_INITIAL_CONDITIONS_HELP);
   IF #_w1 THEN
       "DB442_HOPPERS_ALARM_DECODING".GLOBAL_ALARMS_MACHINE.HELP_DECODING := #DB_NUMBER;
       "DB441_POWDER_FEEDERS_ALARM_DECODING".GLOBAL_ALARMS_MACHINE.HELP_DECODING := #DB_NUMBER;
   END_IF;
   IF #_w1 AND (#DATA.FEEDBACK_ON_LINE_1 OR #DATA.FEEDBACK_ON_LINE_2) THEN
       "DB428_OPERATOR_HELP".HELP_OPERATOR_805 := TRUE;
   END_IF;
END_REGION

REGION Network 7: MANUAL MODE NOT SELECTED HELP / Manual Mode Not Selected Help*
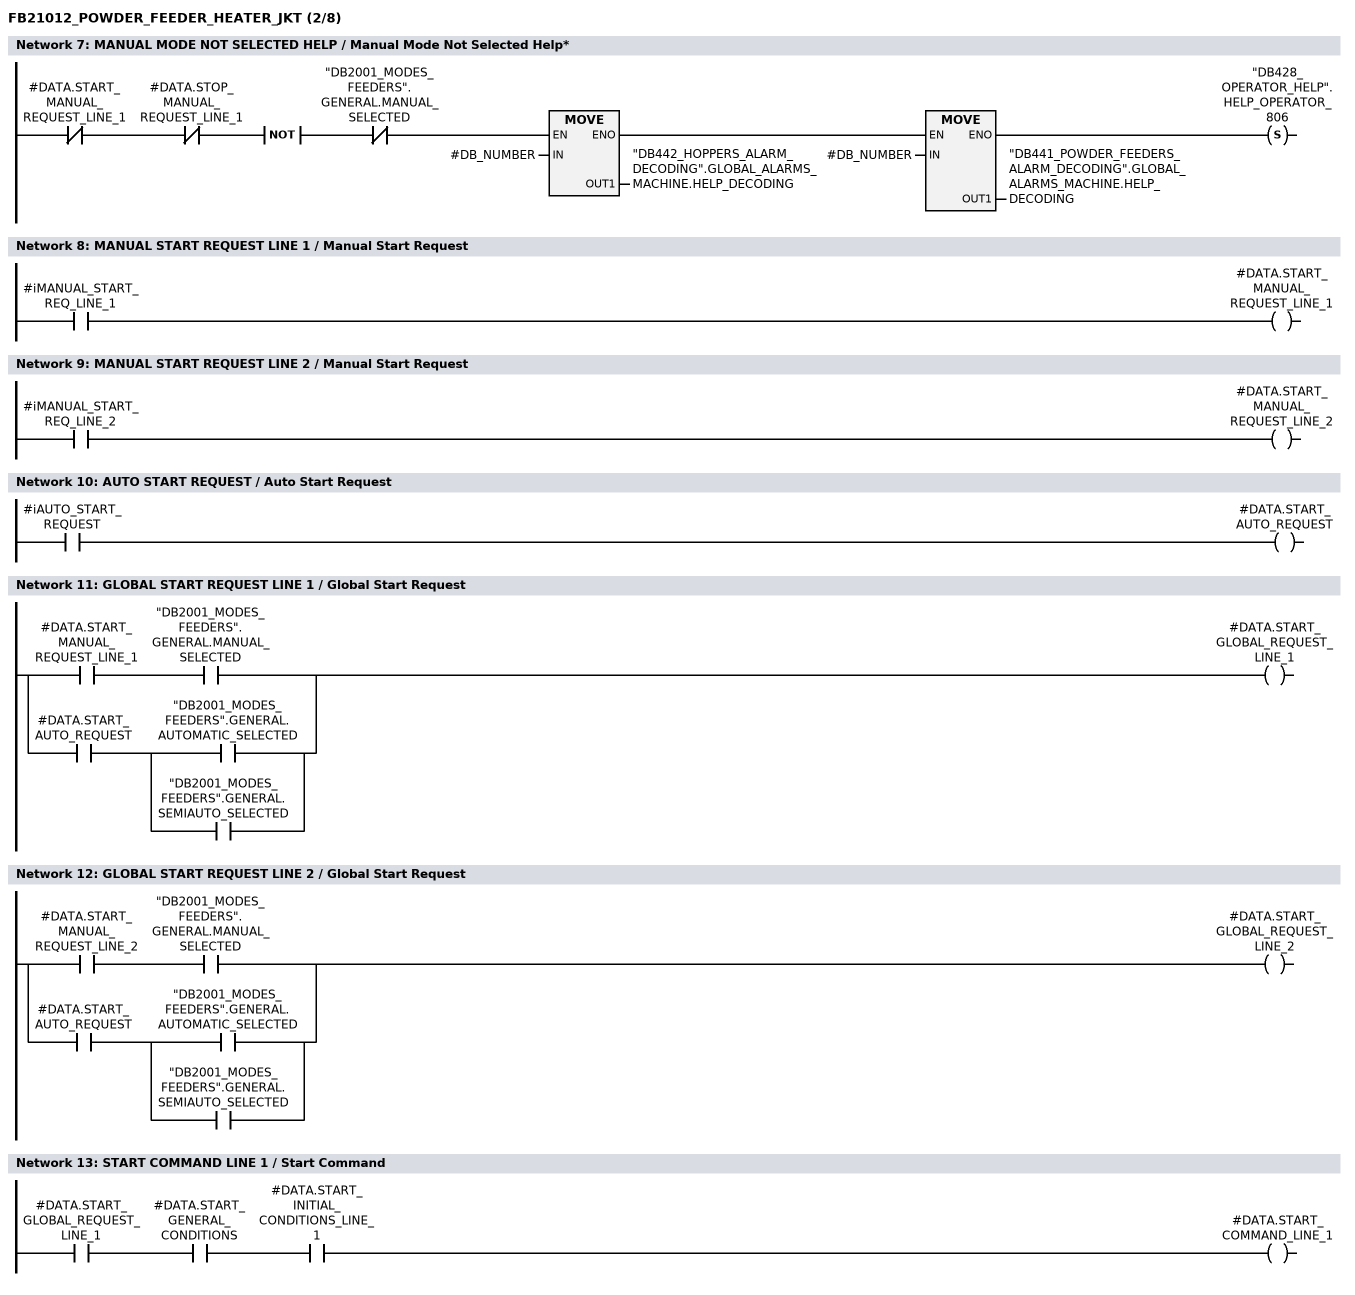
   RUNG wire#powerrail
      I_Contact( #DATA.START_MANUAL_REQUEST_LINE_1 )
      I_Contact( #DATA.STOP_MANUAL_REQUEST_LINE_1 )
      Not()
      I_Contact( "DB2001_MODES_FEEDERS".GENERAL.MANUAL_SELECTED )
      Move(in := #DB_NUMBER, out1 => "DB442_HOPPERS_ALARM_DECODING".GLOBAL_ALARMS_MACHINE.HELP_DECODING)
      Move(in := #DB_NUMBER, out1 => "DB441_POWDER_FEEDERS_ALARM_DECODING".GLOBAL_ALARMS_MACHINE.HELP_DECODING)
      S_Coil( "DB428_OPERATOR_HELP".HELP_OPERATOR_806 )
   END_RUNG
   // the same network as SCL:
   IF NOT (NOT #DATA.START_MANUAL_REQUEST_LINE_1 AND NOT #DATA.STOP_MANUAL_REQUEST_LINE_1) AND NOT "DB2001_MODES_FEEDERS".GENERAL.MANUAL_SELECTED THEN
       "DB442_HOPPERS_ALARM_DECODING".GLOBAL_ALARMS_MACHINE.HELP_DECODING := #DB_NUMBER;
       "DB441_POWDER_FEEDERS_ALARM_DECODING".GLOBAL_ALARMS_MACHINE.HELP_DECODING := #DB_NUMBER;
       "DB428_OPERATOR_HELP".HELP_OPERATOR_806 := TRUE;
   END_IF;
END_REGION

REGION Network 8: MANUAL START REQUEST LINE 1 / Manual Start Request
   RUNG wire#powerrail
      Contact( #iMANUAL_START_REQ_LINE_1 )
      Coil( #DATA.START_MANUAL_REQUEST_LINE_1 )
   END_RUNG
   // the same network as SCL:
   #DATA.START_MANUAL_REQUEST_LINE_1 := #iMANUAL_START_REQ_LINE_1;
END_REGION

REGION Network 9: MANUAL START REQUEST LINE 2 / Manual Start Request
   RUNG wire#powerrail
      Contact( #iMANUAL_START_REQ_LINE_2 )
      Coil( #DATA.START_MANUAL_REQUEST_LINE_2 )
   END_RUNG
   // the same network as SCL:
   #DATA.START_MANUAL_REQUEST_LINE_2 := #iMANUAL_START_REQ_LINE_2;
END_REGION

REGION Network 10: AUTO START REQUEST / Auto Start Request
   RUNG wire#powerrail
      Contact( #iAUTO_START_REQUEST )
      Coil( #DATA.START_AUTO_REQUEST )
   END_RUNG
   // the same network as SCL:
   #DATA.START_AUTO_REQUEST := #iAUTO_START_REQUEST;
END_REGION

REGION Network 11: GLOBAL START REQUEST LINE 1 / Global Start Request
   RUNG wire#powerrail
      Contact( #DATA.START_MANUAL_REQUEST_LINE_1 )
      Contact( "DB2001_MODES_FEEDERS".GENERAL.MANUAL_SELECTED )
      wire#w1
      Coil( #DATA.START_GLOBAL_REQUEST_LINE_1 )
   END_RUNG
   RUNG wire#powerrail
      Contact( #DATA.START_AUTO_REQUEST )
      wire#w2
      Contact( "DB2001_MODES_FEEDERS".GENERAL.AUTOMATIC_SELECTED )
   END_RUNG wire#w1
   RUNG wire#w2
      Contact( "DB2001_MODES_FEEDERS".GENERAL.SEMIAUTO_SELECTED )
   END_RUNG wire#w1
   // the same network as SCL:
   #DATA.START_GLOBAL_REQUEST_LINE_1 := (#DATA.START_MANUAL_REQUEST_LINE_1 AND "DB2001_MODES_FEEDERS".GENERAL.MANUAL_SELECTED) OR (#DATA.START_AUTO_REQUEST AND ("DB2001_MODES_FEEDERS".GENERAL.AUTOMATIC_SELECTED OR "DB2001_MODES_FEEDERS".GENERAL.SEMIAUTO_SELECTED));
END_REGION

REGION Network 12: GLOBAL START REQUEST LINE 2 / Global Start Request
   RUNG wire#powerrail
      Contact( #DATA.START_MANUAL_REQUEST_LINE_2 )
      Contact( "DB2001_MODES_FEEDERS".GENERAL.MANUAL_SELECTED )
      wire#w1
      Coil( #DATA.START_GLOBAL_REQUEST_LINE_2 )
   END_RUNG
   RUNG wire#powerrail
      Contact( #DATA.START_AUTO_REQUEST )
      wire#w2
      Contact( "DB2001_MODES_FEEDERS".GENERAL.AUTOMATIC_SELECTED )
   END_RUNG wire#w1
   RUNG wire#w2
      Contact( "DB2001_MODES_FEEDERS".GENERAL.SEMIAUTO_SELECTED )
   END_RUNG wire#w1
   // the same network as SCL:
   #DATA.START_GLOBAL_REQUEST_LINE_2 := (#DATA.START_MANUAL_REQUEST_LINE_2 AND "DB2001_MODES_FEEDERS".GENERAL.MANUAL_SELECTED) OR (#DATA.START_AUTO_REQUEST AND ("DB2001_MODES_FEEDERS".GENERAL.AUTOMATIC_SELECTED OR "DB2001_MODES_FEEDERS".GENERAL.SEMIAUTO_SELECTED));
END_REGION

REGION Network 13: START COMMAND LINE 1 / Start Command
   RUNG wire#powerrail
      Contact( #DATA.START_GLOBAL_REQUEST_LINE_1 )
      Contact( #DATA.START_GENERAL_CONDITIONS )
      Contact( #DATA.START_INITIAL_CONDITIONS_LINE_1 )
      Coil( #DATA.START_COMMAND_LINE_1 )
   END_RUNG
   // the same network as SCL:
   #DATA.START_COMMAND_LINE_1 := #DATA.START_GLOBAL_REQUEST_LINE_1 AND #DATA.START_GENERAL_CONDITIONS AND #DATA.START_INITIAL_CONDITIONS_LINE_1;
END_REGION

REGION Network 14: START COMMAND LINE 2 / Start Command
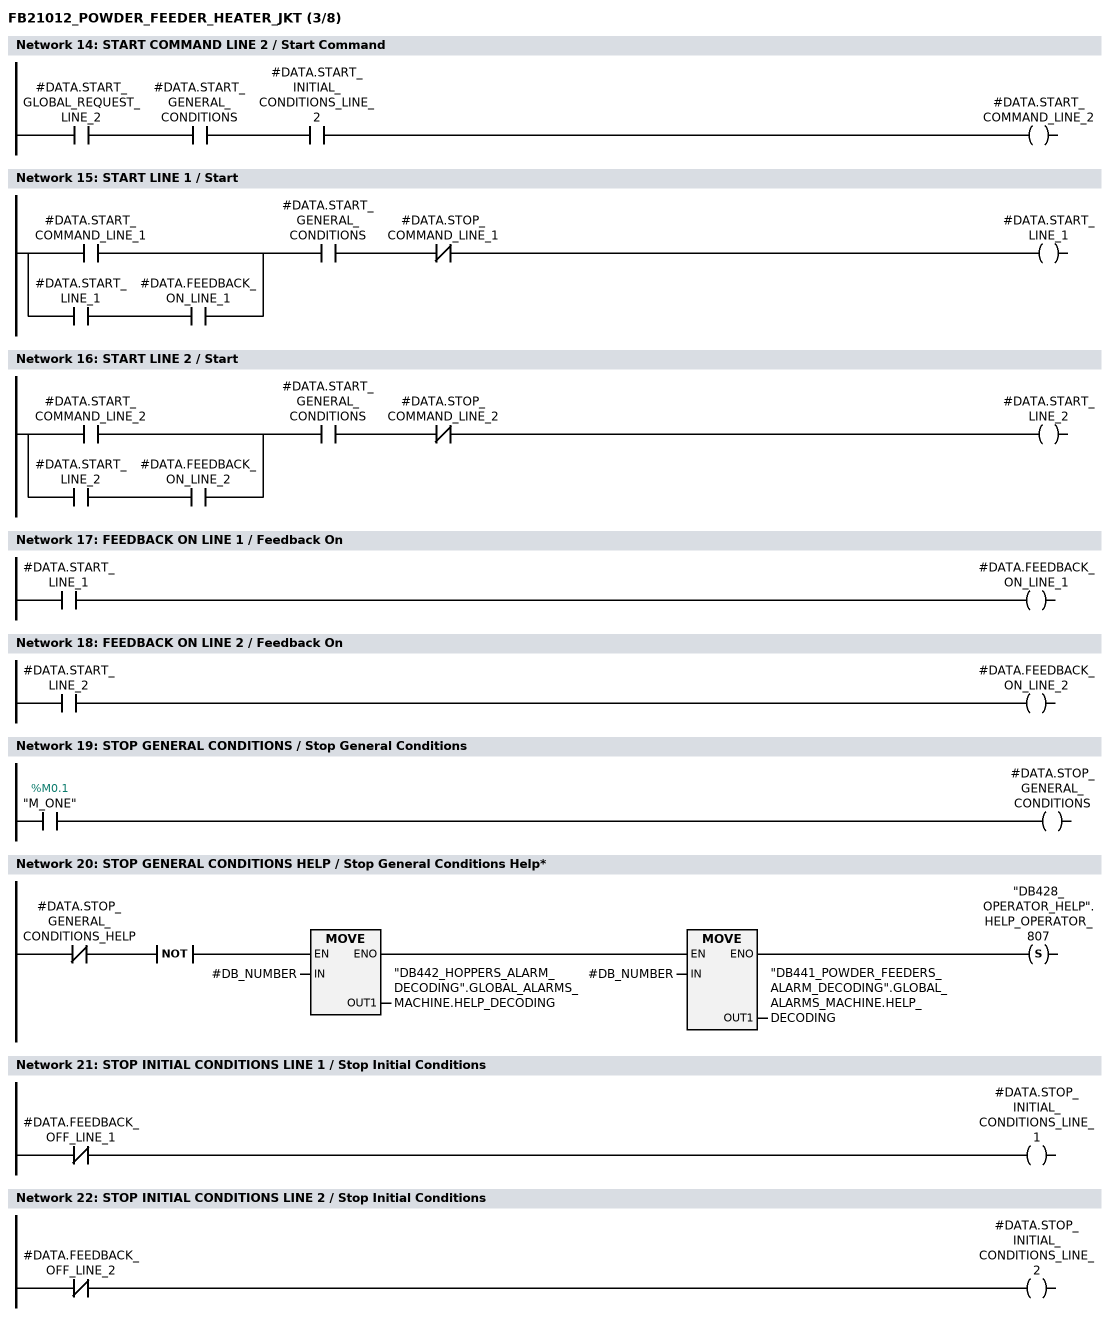
   RUNG wire#powerrail
      Contact( #DATA.START_GLOBAL_REQUEST_LINE_2 )
      Contact( #DATA.START_GENERAL_CONDITIONS )
      Contact( #DATA.START_INITIAL_CONDITIONS_LINE_2 )
      Coil( #DATA.START_COMMAND_LINE_2 )
   END_RUNG
   // the same network as SCL:
   #DATA.START_COMMAND_LINE_2 := #DATA.START_GLOBAL_REQUEST_LINE_2 AND #DATA.START_GENERAL_CONDITIONS AND #DATA.START_INITIAL_CONDITIONS_LINE_2;
END_REGION

REGION Network 15: START LINE 1 / Start
   RUNG wire#powerrail
      Contact( #DATA.START_COMMAND_LINE_1 )
      wire#w1
      Contact( #DATA.START_GENERAL_CONDITIONS )
      I_Contact( #DATA.STOP_COMMAND_LINE_1 )
      Coil( #DATA.START_LINE_1 )
   END_RUNG
   RUNG wire#powerrail
      Contact( #DATA.START_LINE_1 )
      Contact( #DATA.FEEDBACK_ON_LINE_1 )
   END_RUNG wire#w1
   // the same network as SCL:
   #DATA.START_LINE_1 := (#DATA.START_COMMAND_LINE_1 OR (#DATA.START_LINE_1 AND #DATA.FEEDBACK_ON_LINE_1)) AND #DATA.START_GENERAL_CONDITIONS AND NOT #DATA.STOP_COMMAND_LINE_1;
END_REGION

REGION Network 16: START LINE 2 / Start
   RUNG wire#powerrail
      Contact( #DATA.START_COMMAND_LINE_2 )
      wire#w1
      Contact( #DATA.START_GENERAL_CONDITIONS )
      I_Contact( #DATA.STOP_COMMAND_LINE_2 )
      Coil( #DATA.START_LINE_2 )
   END_RUNG
   RUNG wire#powerrail
      Contact( #DATA.START_LINE_2 )
      Contact( #DATA.FEEDBACK_ON_LINE_2 )
   END_RUNG wire#w1
   // the same network as SCL:
   #DATA.START_LINE_2 := (#DATA.START_COMMAND_LINE_2 OR (#DATA.START_LINE_2 AND #DATA.FEEDBACK_ON_LINE_2)) AND #DATA.START_GENERAL_CONDITIONS AND NOT #DATA.STOP_COMMAND_LINE_2;
END_REGION

REGION Network 17: FEEDBACK ON LINE 1 / Feedback On
   RUNG wire#powerrail
      Contact( #DATA.START_LINE_1 )
      Coil( #DATA.FEEDBACK_ON_LINE_1 )
   END_RUNG
   // the same network as SCL:
   #DATA.FEEDBACK_ON_LINE_1 := #DATA.START_LINE_1;
END_REGION

REGION Network 18: FEEDBACK ON LINE 2 / Feedback On
   RUNG wire#powerrail
      Contact( #DATA.START_LINE_2 )
      Coil( #DATA.FEEDBACK_ON_LINE_2 )
   END_RUNG
   // the same network as SCL:
   #DATA.FEEDBACK_ON_LINE_2 := #DATA.START_LINE_2;
END_REGION

REGION Network 19: STOP GENERAL CONDITIONS / Stop General Conditions
   RUNG wire#powerrail
      Contact( "M_ONE" )
      Coil( #DATA.STOP_GENERAL_CONDITIONS )
   END_RUNG
   // the same network as SCL:
   #DATA.STOP_GENERAL_CONDITIONS := "M_ONE";
END_REGION

REGION Network 20: STOP GENERAL CONDITIONS HELP / Stop General Conditions Help*
   RUNG wire#powerrail
      I_Contact( #DATA.STOP_GENERAL_CONDITIONS_HELP )
      Not()
      Move(in := #DB_NUMBER, out1 => "DB442_HOPPERS_ALARM_DECODING".GLOBAL_ALARMS_MACHINE.HELP_DECODING)
      Move(in := #DB_NUMBER, out1 => "DB441_POWDER_FEEDERS_ALARM_DECODING".GLOBAL_ALARMS_MACHINE.HELP_DECODING)
      S_Coil( "DB428_OPERATOR_HELP".HELP_OPERATOR_807 )
   END_RUNG
   // the same network as SCL:
   IF NOT (NOT #DATA.STOP_GENERAL_CONDITIONS_HELP) THEN
       "DB442_HOPPERS_ALARM_DECODING".GLOBAL_ALARMS_MACHINE.HELP_DECODING := #DB_NUMBER;
       "DB441_POWDER_FEEDERS_ALARM_DECODING".GLOBAL_ALARMS_MACHINE.HELP_DECODING := #DB_NUMBER;
       "DB428_OPERATOR_HELP".HELP_OPERATOR_807 := TRUE;
   END_IF;
END_REGION

REGION Network 21: STOP INITIAL CONDITIONS LINE 1 / Stop Initial Conditions
   RUNG wire#powerrail
      I_Contact( #DATA.FEEDBACK_OFF_LINE_1 )
      Coil( #DATA.STOP_INITIAL_CONDITIONS_LINE_1 )
   END_RUNG
   // the same network as SCL:
   #DATA.STOP_INITIAL_CONDITIONS_LINE_1 := NOT #DATA.FEEDBACK_OFF_LINE_1;
END_REGION

REGION Network 22: STOP INITIAL CONDITIONS LINE 2 / Stop Initial Conditions
   RUNG wire#powerrail
      I_Contact( #DATA.FEEDBACK_OFF_LINE_2 )
      Coil( #DATA.STOP_INITIAL_CONDITIONS_LINE_2 )
   END_RUNG
   // the same network as SCL:
   #DATA.STOP_INITIAL_CONDITIONS_LINE_2 := NOT #DATA.FEEDBACK_OFF_LINE_2;
END_REGION

REGION Network 23: STOP INITIAL CONDITIONS HELP / Stop Initial Conditions Help*
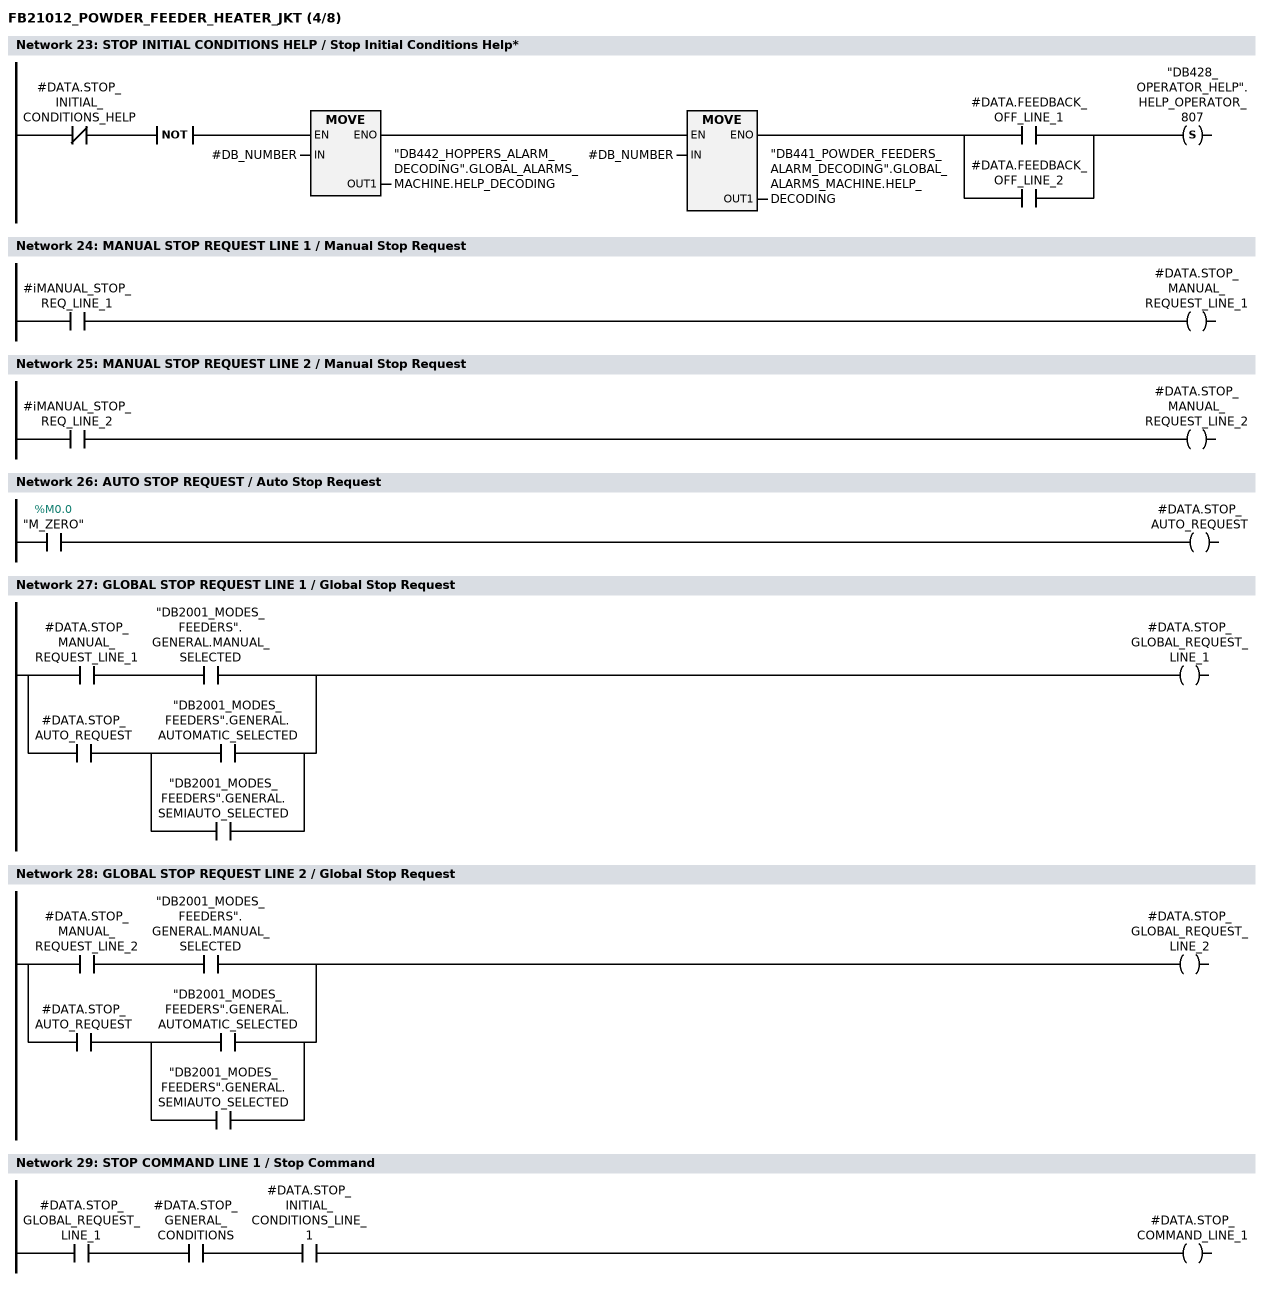
   RUNG wire#powerrail
      I_Contact( #DATA.STOP_INITIAL_CONDITIONS_HELP )
      Not()
      Move(in := #DB_NUMBER, out1 => "DB442_HOPPERS_ALARM_DECODING".GLOBAL_ALARMS_MACHINE.HELP_DECODING)
      Move(in := #DB_NUMBER, out1 => "DB441_POWDER_FEEDERS_ALARM_DECODING".GLOBAL_ALARMS_MACHINE.HELP_DECODING)
      wire#w1
      Contact( #DATA.FEEDBACK_OFF_LINE_1 )
      wire#w2
      S_Coil( "DB428_OPERATOR_HELP".HELP_OPERATOR_807 )
   END_RUNG
   RUNG wire#w1
      Contact( #DATA.FEEDBACK_OFF_LINE_2 )
   END_RUNG wire#w2
   // the same network as SCL:
   #_w1 := NOT (NOT #DATA.STOP_INITIAL_CONDITIONS_HELP);
   IF #_w1 THEN
       "DB442_HOPPERS_ALARM_DECODING".GLOBAL_ALARMS_MACHINE.HELP_DECODING := #DB_NUMBER;
       "DB441_POWDER_FEEDERS_ALARM_DECODING".GLOBAL_ALARMS_MACHINE.HELP_DECODING := #DB_NUMBER;
   END_IF;
   IF #_w1 AND (#DATA.FEEDBACK_OFF_LINE_1 OR #DATA.FEEDBACK_OFF_LINE_2) THEN
       "DB428_OPERATOR_HELP".HELP_OPERATOR_807 := TRUE;
   END_IF;
END_REGION

REGION Network 24: MANUAL STOP REQUEST LINE 1 / Manual Stop Request
   RUNG wire#powerrail
      Contact( #iMANUAL_STOP_REQ_LINE_1 )
      Coil( #DATA.STOP_MANUAL_REQUEST_LINE_1 )
   END_RUNG
   // the same network as SCL:
   #DATA.STOP_MANUAL_REQUEST_LINE_1 := #iMANUAL_STOP_REQ_LINE_1;
END_REGION

REGION Network 25: MANUAL STOP REQUEST LINE 2 / Manual Stop Request
   RUNG wire#powerrail
      Contact( #iMANUAL_STOP_REQ_LINE_2 )
      Coil( #DATA.STOP_MANUAL_REQUEST_LINE_2 )
   END_RUNG
   // the same network as SCL:
   #DATA.STOP_MANUAL_REQUEST_LINE_2 := #iMANUAL_STOP_REQ_LINE_2;
END_REGION

REGION Network 26: AUTO STOP REQUEST / Auto Stop Request
   RUNG wire#powerrail
      Contact( "M_ZERO" )
      Coil( #DATA.STOP_AUTO_REQUEST )
   END_RUNG
   // the same network as SCL:
   #DATA.STOP_AUTO_REQUEST := "M_ZERO";
END_REGION

REGION Network 27: GLOBAL STOP REQUEST LINE 1 / Global Stop Request
   RUNG wire#powerrail
      Contact( #DATA.STOP_MANUAL_REQUEST_LINE_1 )
      Contact( "DB2001_MODES_FEEDERS".GENERAL.MANUAL_SELECTED )
      wire#w1
      Coil( #DATA.STOP_GLOBAL_REQUEST_LINE_1 )
   END_RUNG
   RUNG wire#powerrail
      Contact( #DATA.STOP_AUTO_REQUEST )
      wire#w2
      Contact( "DB2001_MODES_FEEDERS".GENERAL.AUTOMATIC_SELECTED )
   END_RUNG wire#w1
   RUNG wire#w2
      Contact( "DB2001_MODES_FEEDERS".GENERAL.SEMIAUTO_SELECTED )
   END_RUNG wire#w1
   // the same network as SCL:
   #DATA.STOP_GLOBAL_REQUEST_LINE_1 := (#DATA.STOP_MANUAL_REQUEST_LINE_1 AND "DB2001_MODES_FEEDERS".GENERAL.MANUAL_SELECTED) OR (#DATA.STOP_AUTO_REQUEST AND ("DB2001_MODES_FEEDERS".GENERAL.AUTOMATIC_SELECTED OR "DB2001_MODES_FEEDERS".GENERAL.SEMIAUTO_SELECTED));
END_REGION

REGION Network 28: GLOBAL STOP REQUEST LINE 2 / Global Stop Request
   RUNG wire#powerrail
      Contact( #DATA.STOP_MANUAL_REQUEST_LINE_2 )
      Contact( "DB2001_MODES_FEEDERS".GENERAL.MANUAL_SELECTED )
      wire#w1
      Coil( #DATA.STOP_GLOBAL_REQUEST_LINE_2 )
   END_RUNG
   RUNG wire#powerrail
      Contact( #DATA.STOP_AUTO_REQUEST )
      wire#w2
      Contact( "DB2001_MODES_FEEDERS".GENERAL.AUTOMATIC_SELECTED )
   END_RUNG wire#w1
   RUNG wire#w2
      Contact( "DB2001_MODES_FEEDERS".GENERAL.SEMIAUTO_SELECTED )
   END_RUNG wire#w1
   // the same network as SCL:
   #DATA.STOP_GLOBAL_REQUEST_LINE_2 := (#DATA.STOP_MANUAL_REQUEST_LINE_2 AND "DB2001_MODES_FEEDERS".GENERAL.MANUAL_SELECTED) OR (#DATA.STOP_AUTO_REQUEST AND ("DB2001_MODES_FEEDERS".GENERAL.AUTOMATIC_SELECTED OR "DB2001_MODES_FEEDERS".GENERAL.SEMIAUTO_SELECTED));
END_REGION

REGION Network 29: STOP COMMAND LINE 1 / Stop Command
   RUNG wire#powerrail
      Contact( #DATA.STOP_GLOBAL_REQUEST_LINE_1 )
      Contact( #DATA.STOP_GENERAL_CONDITIONS )
      Contact( #DATA.STOP_INITIAL_CONDITIONS_LINE_1 )
      Coil( #DATA.STOP_COMMAND_LINE_1 )
   END_RUNG
   // the same network as SCL:
   #DATA.STOP_COMMAND_LINE_1 := #DATA.STOP_GLOBAL_REQUEST_LINE_1 AND #DATA.STOP_GENERAL_CONDITIONS AND #DATA.STOP_INITIAL_CONDITIONS_LINE_1;
END_REGION

REGION Network 30: STOP COMMAND LINE 2 / Stop Command
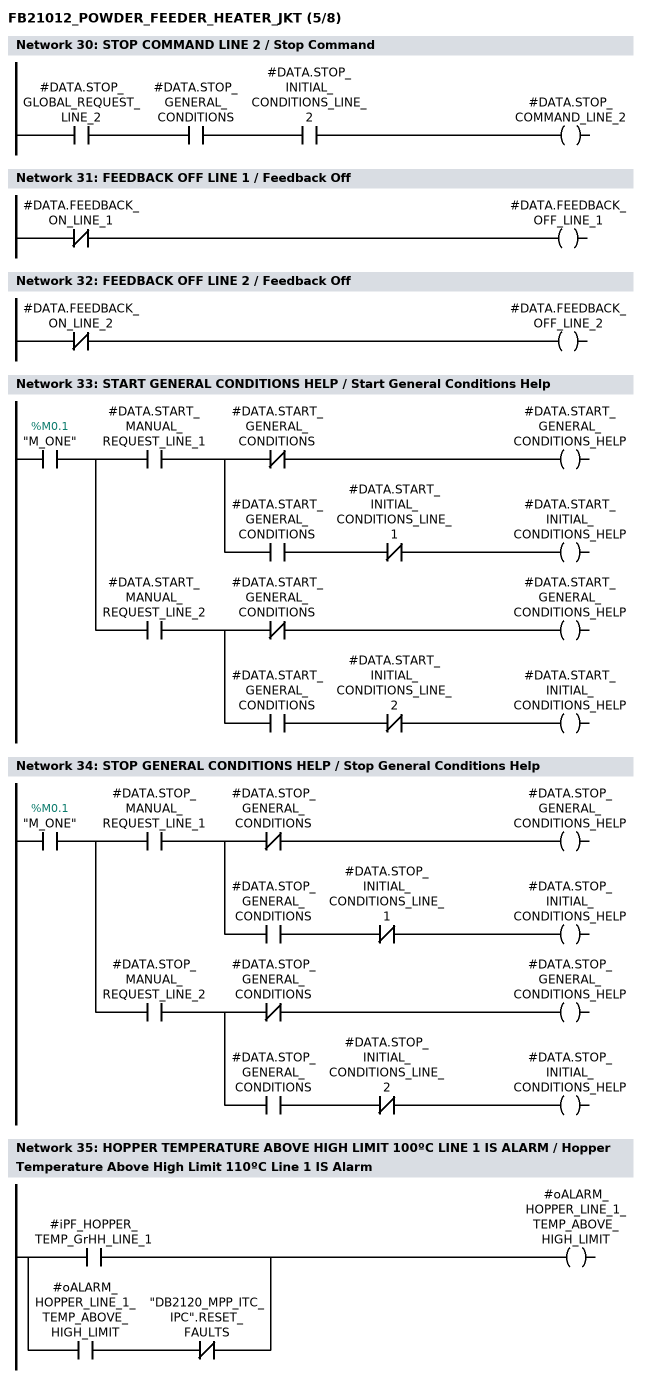
   RUNG wire#powerrail
      Contact( #DATA.STOP_GLOBAL_REQUEST_LINE_2 )
      Contact( #DATA.STOP_GENERAL_CONDITIONS )
      Contact( #DATA.STOP_INITIAL_CONDITIONS_LINE_2 )
      Coil( #DATA.STOP_COMMAND_LINE_2 )
   END_RUNG
   // the same network as SCL:
   #DATA.STOP_COMMAND_LINE_2 := #DATA.STOP_GLOBAL_REQUEST_LINE_2 AND #DATA.STOP_GENERAL_CONDITIONS AND #DATA.STOP_INITIAL_CONDITIONS_LINE_2;
END_REGION

REGION Network 31: FEEDBACK OFF LINE 1 / Feedback Off
   RUNG wire#powerrail
      I_Contact( #DATA.FEEDBACK_ON_LINE_1 )
      Coil( #DATA.FEEDBACK_OFF_LINE_1 )
   END_RUNG
   // the same network as SCL:
   #DATA.FEEDBACK_OFF_LINE_1 := NOT #DATA.FEEDBACK_ON_LINE_1;
END_REGION

REGION Network 32: FEEDBACK OFF LINE 2 / Feedback Off
   RUNG wire#powerrail
      I_Contact( #DATA.FEEDBACK_ON_LINE_2 )
      Coil( #DATA.FEEDBACK_OFF_LINE_2 )
   END_RUNG
   // the same network as SCL:
   #DATA.FEEDBACK_OFF_LINE_2 := NOT #DATA.FEEDBACK_ON_LINE_2;
END_REGION

REGION Network 33: START GENERAL CONDITIONS HELP / Start General Conditions Help
   RUNG wire#powerrail
      Contact( "M_ONE" )
      wire#w1
      Contact( #DATA.START_MANUAL_REQUEST_LINE_1 )
      wire#w2
      I_Contact( #DATA.START_GENERAL_CONDITIONS )
      Coil( #DATA.START_GENERAL_CONDITIONS_HELP )
   END_RUNG
   RUNG wire#w2
      Contact( #DATA.START_GENERAL_CONDITIONS )
      I_Contact( #DATA.START_INITIAL_CONDITIONS_LINE_1 )
      Coil( #DATA.START_INITIAL_CONDITIONS_HELP )
   END_RUNG
   RUNG wire#w1
      Contact( #DATA.START_MANUAL_REQUEST_LINE_2 )
      wire#w3
      I_Contact( #DATA.START_GENERAL_CONDITIONS )
      Coil( #DATA.START_GENERAL_CONDITIONS_HELP )
   END_RUNG
   RUNG wire#w3
      Contact( #DATA.START_GENERAL_CONDITIONS )
      I_Contact( #DATA.START_INITIAL_CONDITIONS_LINE_2 )
      Coil( #DATA.START_INITIAL_CONDITIONS_HELP )
   END_RUNG
   // the same network as SCL:
   #_w1 := "M_ONE" AND #DATA.START_MANUAL_REQUEST_LINE_1;
   #DATA.START_GENERAL_CONDITIONS_HELP := #_w1 AND NOT #DATA.START_GENERAL_CONDITIONS;
   #DATA.START_INITIAL_CONDITIONS_HELP := #_w1 AND #DATA.START_GENERAL_CONDITIONS AND NOT #DATA.START_INITIAL_CONDITIONS_LINE_1;
   #_w2 := "M_ONE" AND #DATA.START_MANUAL_REQUEST_LINE_2;
   #DATA.START_GENERAL_CONDITIONS_HELP := #_w2 AND NOT #DATA.START_GENERAL_CONDITIONS;
   #DATA.START_INITIAL_CONDITIONS_HELP := #_w2 AND #DATA.START_GENERAL_CONDITIONS AND NOT #DATA.START_INITIAL_CONDITIONS_LINE_2;
END_REGION

REGION Network 34: STOP GENERAL CONDITIONS HELP / Stop General Conditions Help
   RUNG wire#powerrail
      Contact( "M_ONE" )
      wire#w1
      Contact( #DATA.STOP_MANUAL_REQUEST_LINE_1 )
      wire#w2
      I_Contact( #DATA.STOP_GENERAL_CONDITIONS )
      Coil( #DATA.STOP_GENERAL_CONDITIONS_HELP )
   END_RUNG
   RUNG wire#w2
      Contact( #DATA.STOP_GENERAL_CONDITIONS )
      I_Contact( #DATA.STOP_INITIAL_CONDITIONS_LINE_1 )
      Coil( #DATA.STOP_INITIAL_CONDITIONS_HELP )
   END_RUNG
   RUNG wire#w1
      Contact( #DATA.STOP_MANUAL_REQUEST_LINE_2 )
      wire#w3
      I_Contact( #DATA.STOP_GENERAL_CONDITIONS )
      Coil( #DATA.STOP_GENERAL_CONDITIONS_HELP )
   END_RUNG
   RUNG wire#w3
      Contact( #DATA.STOP_GENERAL_CONDITIONS )
      I_Contact( #DATA.STOP_INITIAL_CONDITIONS_LINE_2 )
      Coil( #DATA.STOP_INITIAL_CONDITIONS_HELP )
   END_RUNG
   // the same network as SCL:
   #_w1 := "M_ONE" AND #DATA.STOP_MANUAL_REQUEST_LINE_1;
   #DATA.STOP_GENERAL_CONDITIONS_HELP := #_w1 AND NOT #DATA.STOP_GENERAL_CONDITIONS;
   #DATA.STOP_INITIAL_CONDITIONS_HELP := #_w1 AND #DATA.STOP_GENERAL_CONDITIONS AND NOT #DATA.STOP_INITIAL_CONDITIONS_LINE_1;
   #_w2 := "M_ONE" AND #DATA.STOP_MANUAL_REQUEST_LINE_2;
   #DATA.STOP_GENERAL_CONDITIONS_HELP := #_w2 AND NOT #DATA.STOP_GENERAL_CONDITIONS;
   #DATA.STOP_INITIAL_CONDITIONS_HELP := #_w2 AND #DATA.STOP_GENERAL_CONDITIONS AND NOT #DATA.STOP_INITIAL_CONDITIONS_LINE_2;
END_REGION

REGION Network 35: HOPPER TEMPERATURE ABOVE HIGH LIMIT 100ºC LINE 1 IS ALARM / Hopper Temperature Above High Limit 110ºC Line 1 IS Alarm
   RUNG wire#powerrail
      Contact( #iPF_HOPPER_TEMP_GrHH_LINE_1 )
      wire#w1
      Coil( #oALARM_HOPPER_LINE_1_TEMP_ABOVE_HIGH_LIMIT )
   END_RUNG
   RUNG wire#powerrail
      Contact( #oALARM_HOPPER_LINE_1_TEMP_ABOVE_HIGH_LIMIT )
      I_Contact( "DB2120_MPP_ITC_IPC".RESET_FAULTS )
   END_RUNG wire#w1
   // the same network as SCL:
   #oALARM_HOPPER_LINE_1_TEMP_ABOVE_HIGH_LIMIT := #iPF_HOPPER_TEMP_GrHH_LINE_1 OR (#oALARM_HOPPER_LINE_1_TEMP_ABOVE_HIGH_LIMIT AND NOT "DB2120_MPP_ITC_IPC".RESET_FAULTS);
END_REGION

REGION Network 36: HOPPER TEMPERATURE ABOVE HIGH LIMIT 100ºC LINE 2 IS ALARM / Hopper Temperature Above High Limit 110ºC Line 1 IS Alarm
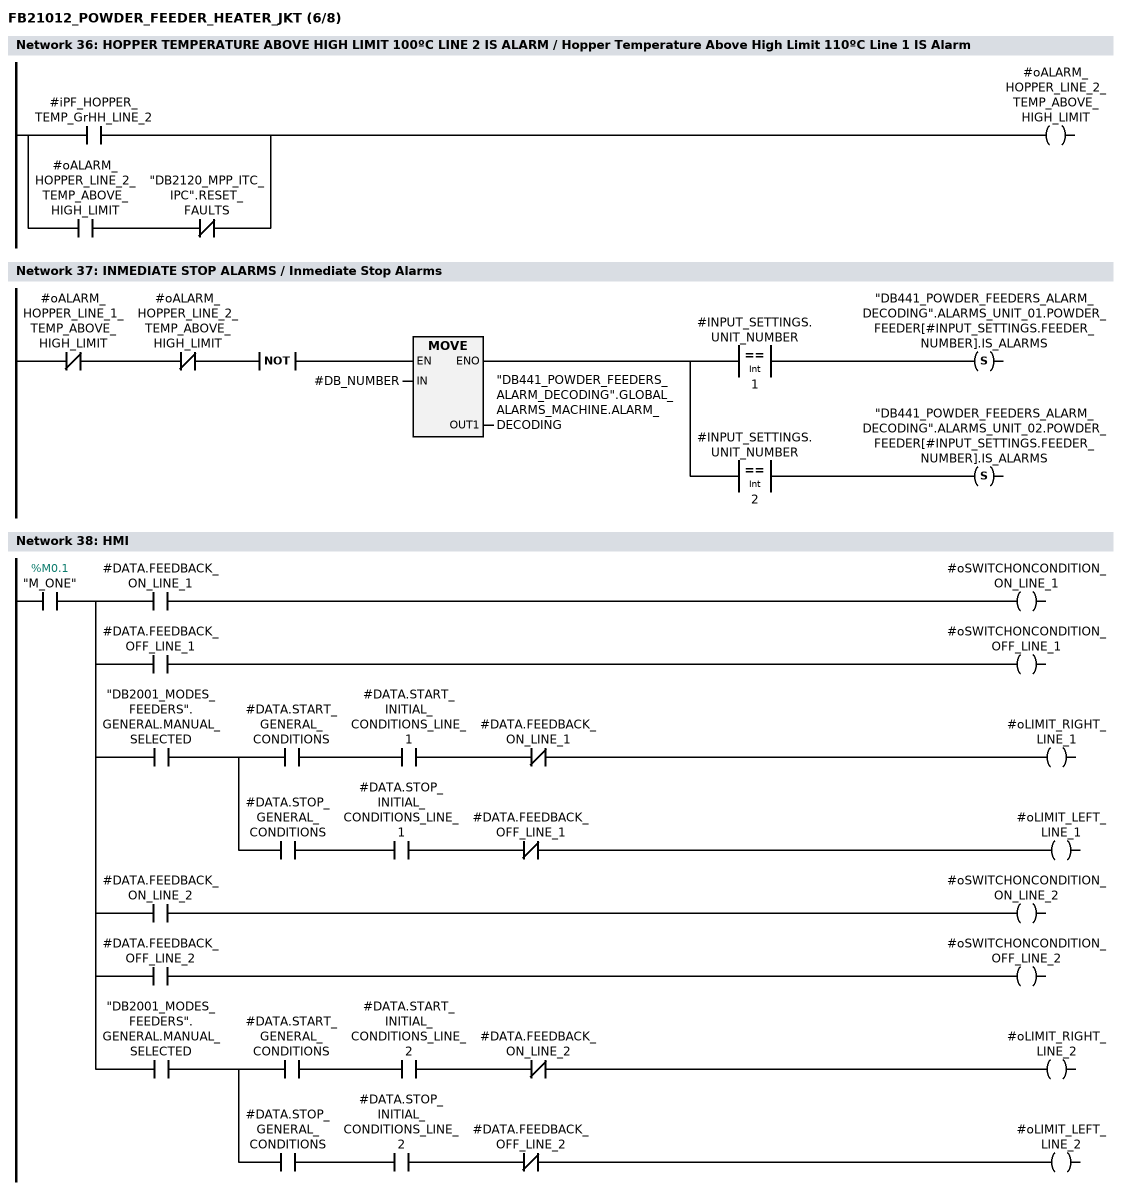
   RUNG wire#powerrail
      Contact( #iPF_HOPPER_TEMP_GrHH_LINE_2 )
      wire#w1
      Coil( #oALARM_HOPPER_LINE_2_TEMP_ABOVE_HIGH_LIMIT )
   END_RUNG
   RUNG wire#powerrail
      Contact( #oALARM_HOPPER_LINE_2_TEMP_ABOVE_HIGH_LIMIT )
      I_Contact( "DB2120_MPP_ITC_IPC".RESET_FAULTS )
   END_RUNG wire#w1
   // the same network as SCL:
   #oALARM_HOPPER_LINE_2_TEMP_ABOVE_HIGH_LIMIT := #iPF_HOPPER_TEMP_GrHH_LINE_2 OR (#oALARM_HOPPER_LINE_2_TEMP_ABOVE_HIGH_LIMIT AND NOT "DB2120_MPP_ITC_IPC".RESET_FAULTS);
END_REGION

REGION Network 37: INMEDIATE STOP ALARMS / Inmediate Stop Alarms
   RUNG wire#powerrail
      I_Contact( #oALARM_HOPPER_LINE_1_TEMP_ABOVE_HIGH_LIMIT )
      I_Contact( #oALARM_HOPPER_LINE_2_TEMP_ABOVE_HIGH_LIMIT )
      Not()
      Move(in := #DB_NUMBER, out1 => "DB441_POWDER_FEEDERS_ALARM_DECODING".GLOBAL_ALARMS_MACHINE.ALARM_DECODING)
      wire#w1
      { S7_Templates := "SrcType := Int" } EQ_Contact(in1 := #INPUT_SETTINGS.UNIT_NUMBER, in2 := 1)
      S_Coil( "DB441_POWDER_FEEDERS_ALARM_DECODING".ALARMS_UNIT_01.POWDER_FEEDER[#INPUT_SETTINGS.FEEDER_NUMBER].IS_ALARMS )
   END_RUNG
   RUNG wire#w1
      { S7_Templates := "SrcType := Int" } EQ_Contact(in1 := #INPUT_SETTINGS.UNIT_NUMBER, in2 := 2)
      S_Coil( "DB441_POWDER_FEEDERS_ALARM_DECODING".ALARMS_UNIT_02.POWDER_FEEDER[#INPUT_SETTINGS.FEEDER_NUMBER].IS_ALARMS )
   END_RUNG
   // the same network as SCL:
   #_w1 := NOT (NOT #oALARM_HOPPER_LINE_1_TEMP_ABOVE_HIGH_LIMIT AND NOT #oALARM_HOPPER_LINE_2_TEMP_ABOVE_HIGH_LIMIT);
   IF #_w1 THEN
       "DB441_POWDER_FEEDERS_ALARM_DECODING".GLOBAL_ALARMS_MACHINE.ALARM_DECODING := #DB_NUMBER;
   END_IF;
   IF #_w1 AND (#INPUT_SETTINGS.UNIT_NUMBER = 1) THEN
       "DB441_POWDER_FEEDERS_ALARM_DECODING".ALARMS_UNIT_01.POWDER_FEEDER[#INPUT_SETTINGS.FEEDER_NUMBER].IS_ALARMS := TRUE;
   END_IF;
   IF #_w1 AND (#INPUT_SETTINGS.UNIT_NUMBER = 2) THEN
       "DB441_POWDER_FEEDERS_ALARM_DECODING".ALARMS_UNIT_02.POWDER_FEEDER[#INPUT_SETTINGS.FEEDER_NUMBER].IS_ALARMS := TRUE;
   END_IF;
END_REGION

REGION Network 38: HMI
   RUNG wire#powerrail
      Contact( "M_ONE" )
      wire#w1
      Contact( #DATA.FEEDBACK_ON_LINE_1 )
      Coil( #oSWITCHONCONDITION_ON_LINE_1 )
   END_RUNG
   RUNG wire#w1
      Contact( #DATA.FEEDBACK_OFF_LINE_1 )
      Coil( #oSWITCHONCONDITION_OFF_LINE_1 )
   END_RUNG
   RUNG wire#w1
      Contact( "DB2001_MODES_FEEDERS".GENERAL.MANUAL_SELECTED )
      wire#w2
      Contact( #DATA.START_GENERAL_CONDITIONS )
      Contact( #DATA.START_INITIAL_CONDITIONS_LINE_1 )
      I_Contact( #DATA.FEEDBACK_ON_LINE_1 )
      Coil( #oLIMIT_RIGHT_LINE_1 )
   END_RUNG
   RUNG wire#w2
      Contact( #DATA.STOP_GENERAL_CONDITIONS )
      Contact( #DATA.STOP_INITIAL_CONDITIONS_LINE_1 )
      I_Contact( #DATA.FEEDBACK_OFF_LINE_1 )
      Coil( #oLIMIT_LEFT_LINE_1 )
   END_RUNG
   RUNG wire#w1
      Contact( #DATA.FEEDBACK_ON_LINE_2 )
      Coil( #oSWITCHONCONDITION_ON_LINE_2 )
   END_RUNG
   RUNG wire#w1
      Contact( #DATA.FEEDBACK_OFF_LINE_2 )
      Coil( #oSWITCHONCONDITION_OFF_LINE_2 )
   END_RUNG
   RUNG wire#w1
      Contact( "DB2001_MODES_FEEDERS".GENERAL.MANUAL_SELECTED )
      wire#w3
      Contact( #DATA.START_GENERAL_CONDITIONS )
      Contact( #DATA.START_INITIAL_CONDITIONS_LINE_2 )
      I_Contact( #DATA.FEEDBACK_ON_LINE_2 )
      Coil( #oLIMIT_RIGHT_LINE_2 )
   END_RUNG
   RUNG wire#w3
      Contact( #DATA.STOP_GENERAL_CONDITIONS )
      Contact( #DATA.STOP_INITIAL_CONDITIONS_LINE_2 )
      I_Contact( #DATA.FEEDBACK_OFF_LINE_2 )
      Coil( #oLIMIT_LEFT_LINE_2 )
   END_RUNG
   // the same network as SCL:
   #oSWITCHONCONDITION_ON_LINE_1 := "M_ONE" AND #DATA.FEEDBACK_ON_LINE_1;
   #oSWITCHONCONDITION_OFF_LINE_1 := "M_ONE" AND #DATA.FEEDBACK_OFF_LINE_1;
   #_w1 := "M_ONE" AND "DB2001_MODES_FEEDERS".GENERAL.MANUAL_SELECTED;
   #oLIMIT_RIGHT_LINE_1 := #_w1 AND #DATA.START_GENERAL_CONDITIONS AND #DATA.START_INITIAL_CONDITIONS_LINE_1 AND NOT #DATA.FEEDBACK_ON_LINE_1;
   #oLIMIT_LEFT_LINE_1 := #_w1 AND #DATA.STOP_GENERAL_CONDITIONS AND #DATA.STOP_INITIAL_CONDITIONS_LINE_1 AND NOT #DATA.FEEDBACK_OFF_LINE_1;
   #oSWITCHONCONDITION_ON_LINE_2 := "M_ONE" AND #DATA.FEEDBACK_ON_LINE_2;
   #oSWITCHONCONDITION_OFF_LINE_2 := "M_ONE" AND #DATA.FEEDBACK_OFF_LINE_2;
   #_w2 := "M_ONE" AND "DB2001_MODES_FEEDERS".GENERAL.MANUAL_SELECTED;
   #oLIMIT_RIGHT_LINE_2 := #_w2 AND #DATA.START_GENERAL_CONDITIONS AND #DATA.START_INITIAL_CONDITIONS_LINE_2 AND NOT #DATA.FEEDBACK_ON_LINE_2;
   #oLIMIT_LEFT_LINE_2 := #_w2 AND #DATA.STOP_GENERAL_CONDITIONS AND #DATA.STOP_INITIAL_CONDITIONS_LINE_2 AND NOT #DATA.FEEDBACK_OFF_LINE_2;
END_REGION

REGION Network 39: HMI ACTIONS / HMI Action
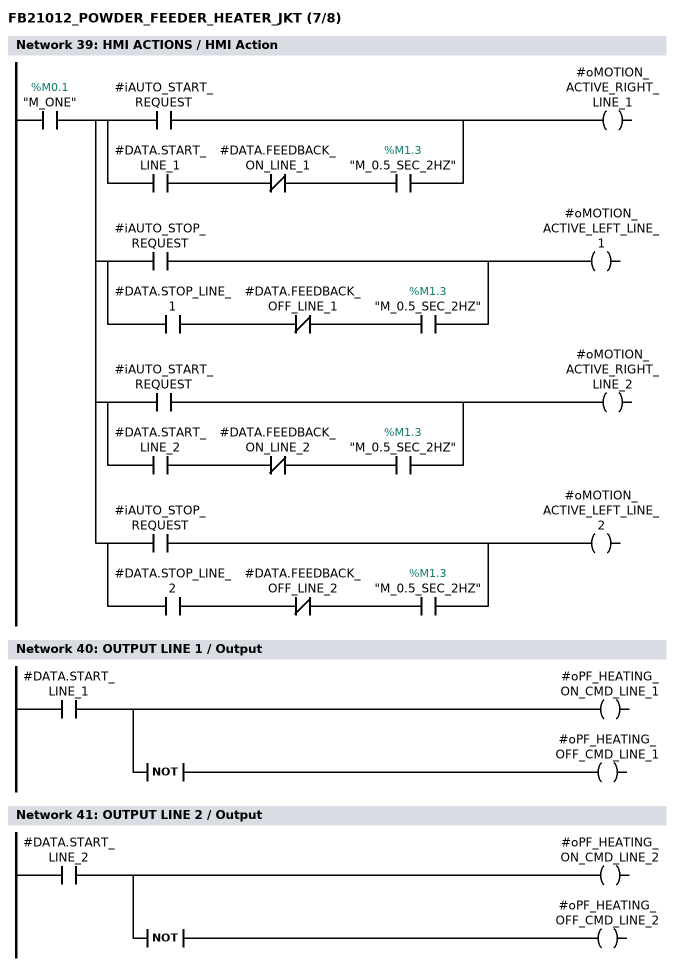
   RUNG wire#powerrail
      Contact( "M_ONE" )
      wire#w1
      Contact( #iAUTO_START_REQUEST )
      wire#w2
      Coil( #oMOTION_ACTIVE_RIGHT_LINE_1 )
   END_RUNG
   RUNG wire#w1
      Contact( #DATA.START_LINE_1 )
      I_Contact( #DATA.FEEDBACK_ON_LINE_1 )
      Contact( "M_0.5_SEC_2HZ" )
   END_RUNG wire#w2
   RUNG wire#w1
      Contact( #iAUTO_STOP_REQUEST )
      wire#w3
      Coil( #oMOTION_ACTIVE_LEFT_LINE_1 )
   END_RUNG
   RUNG wire#w1
      Contact( #DATA.STOP_LINE_1 )
      I_Contact( #DATA.FEEDBACK_OFF_LINE_1 )
      Contact( "M_0.5_SEC_2HZ" )
   END_RUNG wire#w3
   RUNG wire#w1
      Contact( #iAUTO_START_REQUEST )
      wire#w4
      Coil( #oMOTION_ACTIVE_RIGHT_LINE_2 )
   END_RUNG
   RUNG wire#w1
      Contact( #DATA.START_LINE_2 )
      I_Contact( #DATA.FEEDBACK_ON_LINE_2 )
      Contact( "M_0.5_SEC_2HZ" )
   END_RUNG wire#w4
   RUNG wire#w1
      Contact( #iAUTO_STOP_REQUEST )
      wire#w5
      Coil( #oMOTION_ACTIVE_LEFT_LINE_2 )
   END_RUNG
   RUNG wire#w1
      Contact( #DATA.STOP_LINE_2 )
      I_Contact( #DATA.FEEDBACK_OFF_LINE_2 )
      Contact( "M_0.5_SEC_2HZ" )
   END_RUNG wire#w5
   // the same network as SCL:
   #oMOTION_ACTIVE_RIGHT_LINE_1 := "M_ONE" AND (#iAUTO_START_REQUEST OR (#DATA.START_LINE_1 AND NOT #DATA.FEEDBACK_ON_LINE_1 AND "M_0.5_SEC_2HZ"));
   #oMOTION_ACTIVE_LEFT_LINE_1 := "M_ONE" AND (#iAUTO_STOP_REQUEST OR (#DATA.STOP_LINE_1 AND NOT #DATA.FEEDBACK_OFF_LINE_1 AND "M_0.5_SEC_2HZ"));
   #oMOTION_ACTIVE_RIGHT_LINE_2 := "M_ONE" AND (#iAUTO_START_REQUEST OR (#DATA.START_LINE_2 AND NOT #DATA.FEEDBACK_ON_LINE_2 AND "M_0.5_SEC_2HZ"));
   #oMOTION_ACTIVE_LEFT_LINE_2 := "M_ONE" AND (#iAUTO_STOP_REQUEST OR (#DATA.STOP_LINE_2 AND NOT #DATA.FEEDBACK_OFF_LINE_2 AND "M_0.5_SEC_2HZ"));
END_REGION

REGION Network 40: OUTPUT LINE 1 / Output
   RUNG wire#powerrail
      Contact( #DATA.START_LINE_1 )
      wire#w1
      Coil( #oPF_HEATING_ON_CMD_LINE_1 )
   END_RUNG
   RUNG wire#w1
      Not()
      Coil( #oPF_HEATING_OFF_CMD_LINE_1 )
   END_RUNG
   // the same network as SCL:
   #oPF_HEATING_ON_CMD_LINE_1 := #DATA.START_LINE_1;
   #oPF_HEATING_OFF_CMD_LINE_1 := NOT #DATA.START_LINE_1;
END_REGION

REGION Network 41: OUTPUT LINE 2 / Output
   RUNG wire#powerrail
      Contact( #DATA.START_LINE_2 )
      wire#w1
      Coil( #oPF_HEATING_ON_CMD_LINE_2 )
   END_RUNG
   RUNG wire#w1
      Not()
      Coil( #oPF_HEATING_OFF_CMD_LINE_2 )
   END_RUNG
   // the same network as SCL:
   #oPF_HEATING_ON_CMD_LINE_2 := #DATA.START_LINE_2;
   #oPF_HEATING_OFF_CMD_LINE_2 := NOT #DATA.START_LINE_2;
END_REGION

REGION Network 42: HEATER STATUS
   // STATUS:
   // 0: OFF WITH NO CONDITIONS
   // 1: ON
   // 2: OFF WITH CONDITIONS TO SWITCH ON
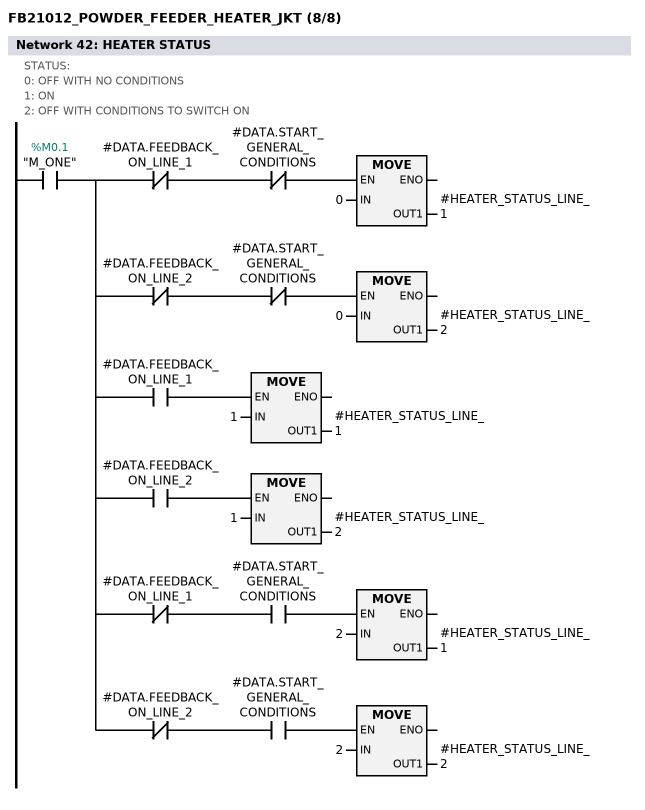
   RUNG wire#powerrail
      Contact( "M_ONE" )
      wire#w1
      I_Contact( #DATA.FEEDBACK_ON_LINE_1 )
      I_Contact( #DATA.START_GENERAL_CONDITIONS )
      Move(in := 0, out1 => #HEATER_STATUS_LINE_1)
   END_RUNG
   RUNG wire#w1
      I_Contact( #DATA.FEEDBACK_ON_LINE_2 )
      I_Contact( #DATA.START_GENERAL_CONDITIONS )
      Move(in := 0, out1 => #HEATER_STATUS_LINE_2)
   END_RUNG
   RUNG wire#w1
      Contact( #DATA.FEEDBACK_ON_LINE_1 )
      Move(in := 1, out1 => #HEATER_STATUS_LINE_1)
   END_RUNG
   RUNG wire#w1
      Contact( #DATA.FEEDBACK_ON_LINE_2 )
      Move(in := 1, out1 => #HEATER_STATUS_LINE_2)
   END_RUNG
   RUNG wire#w1
      I_Contact( #DATA.FEEDBACK_ON_LINE_1 )
      Contact( #DATA.START_GENERAL_CONDITIONS )
      Move(in := 2, out1 => #HEATER_STATUS_LINE_1)
   END_RUNG
   RUNG wire#w1
      I_Contact( #DATA.FEEDBACK_ON_LINE_2 )
      Contact( #DATA.START_GENERAL_CONDITIONS )
      Move(in := 2, out1 => #HEATER_STATUS_LINE_2)
   END_RUNG
   // the same network as SCL:
   IF "M_ONE" AND NOT #DATA.FEEDBACK_ON_LINE_1 AND NOT #DATA.START_GENERAL_CONDITIONS THEN
       #HEATER_STATUS_LINE_1 := 0;
   END_IF;
   IF "M_ONE" AND NOT #DATA.FEEDBACK_ON_LINE_2 AND NOT #DATA.START_GENERAL_CONDITIONS THEN
       #HEATER_STATUS_LINE_2 := 0;
   END_IF;
   IF "M_ONE" AND #DATA.FEEDBACK_ON_LINE_1 THEN #HEATER_STATUS_LINE_1 := 1; END_IF;
   IF "M_ONE" AND #DATA.FEEDBACK_ON_LINE_2 THEN #HEATER_STATUS_LINE_2 := 1; END_IF;
   IF "M_ONE" AND NOT #DATA.FEEDBACK_ON_LINE_1 AND #DATA.START_GENERAL_CONDITIONS THEN
       #HEATER_STATUS_LINE_1 := 2;
   END_IF;
   IF "M_ONE" AND NOT #DATA.FEEDBACK_ON_LINE_2 AND #DATA.START_GENERAL_CONDITIONS THEN
       #HEATER_STATUS_LINE_2 := 2;
   END_IF;
END_REGION
END_FUNCTION_BLOCK

FUNCTION "FC21013_POWDER_FEEDER_HOPPER" : Void   // FC21013, LAD
TITLE = FC21011 POWDER FEEDER HOPPER
{ S7_Optimized_Access := 'TRUE' }
VERSION : 0.1
// stored: AutoNumber false, IsIECCheckEnabled false, SetENOAutomatically false, UDAEnableTagReadback false
   VAR_TEMP
      AUX_PRESSURE : Int;
      AUX_DIGITAL1 : Bool;
      AUX_DIGITAL2 : Bool;
      AUX_SCATTER : Array[0..15] of Bool;
      PRESSURE_NORM : Real;
      PRESSURE_SCALE : Real;
      AUX_PRESSURE2 : Real;
      SCALED2 : Real;
   END_VAR
BEGIN

REGION Network 1: /////_UNIT_01_/////
END_REGION

REGION Network 2: CALL FB21013 POWDER FEEDER 1 HOPPER UNIT 01
   // 2#0000_0001 OPTIONS 0 BIT 0 LINE 1 ENABLED OPTION
   // 2#0000_0010 OPTIONS 0 BIT 1 LINE 2 ENABLED OPTION
   // 2#0000_0100 OPTIONS 0 BIT 2 SPARE
   // 2#0000_1000 OPTIONS 0 BIT 3 SPARE
   // 2#0001_0000 OPTIONS 0 BIT 4 SPARE
   // 2#0010_0000 OPTIONS 0 BIT 5 SPARE
   // 2#0100_0000 OPTIONS 0 BIT 6 SPARE
   // 2#1000_0000 OPTIONS 0 BIT 7 SPARE
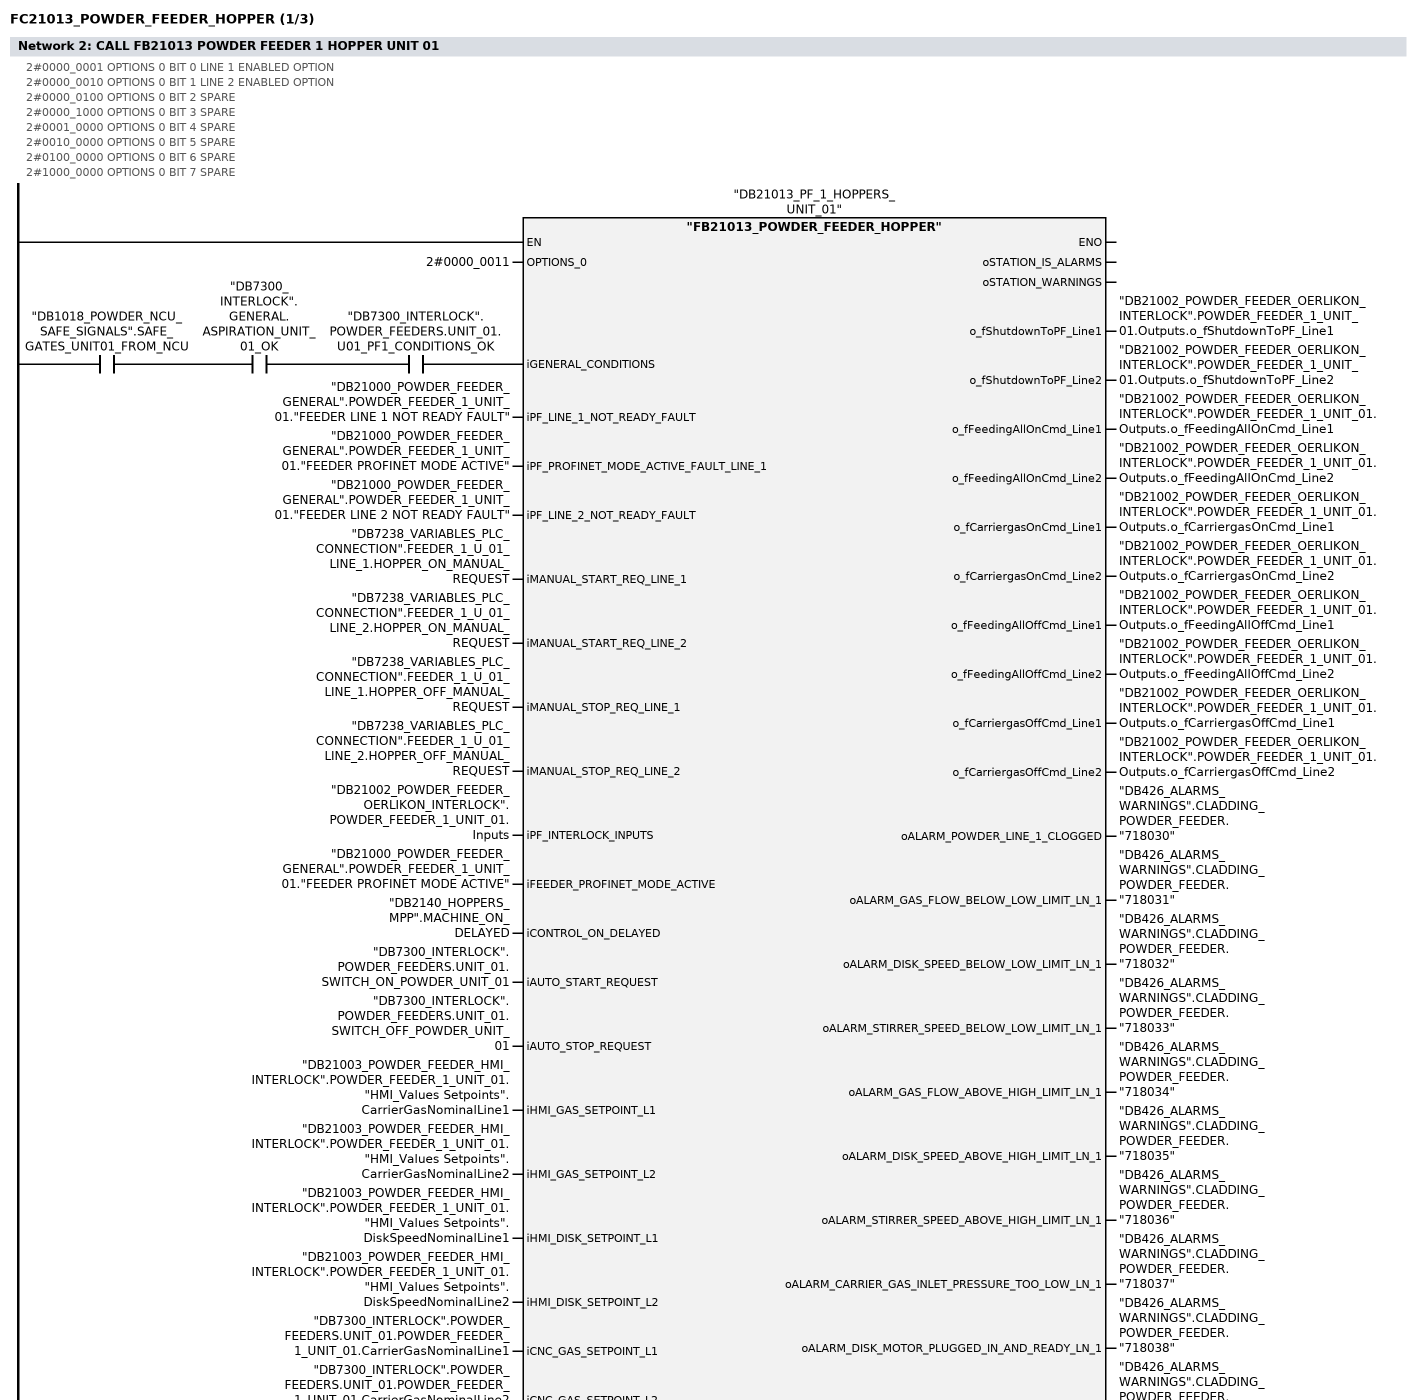
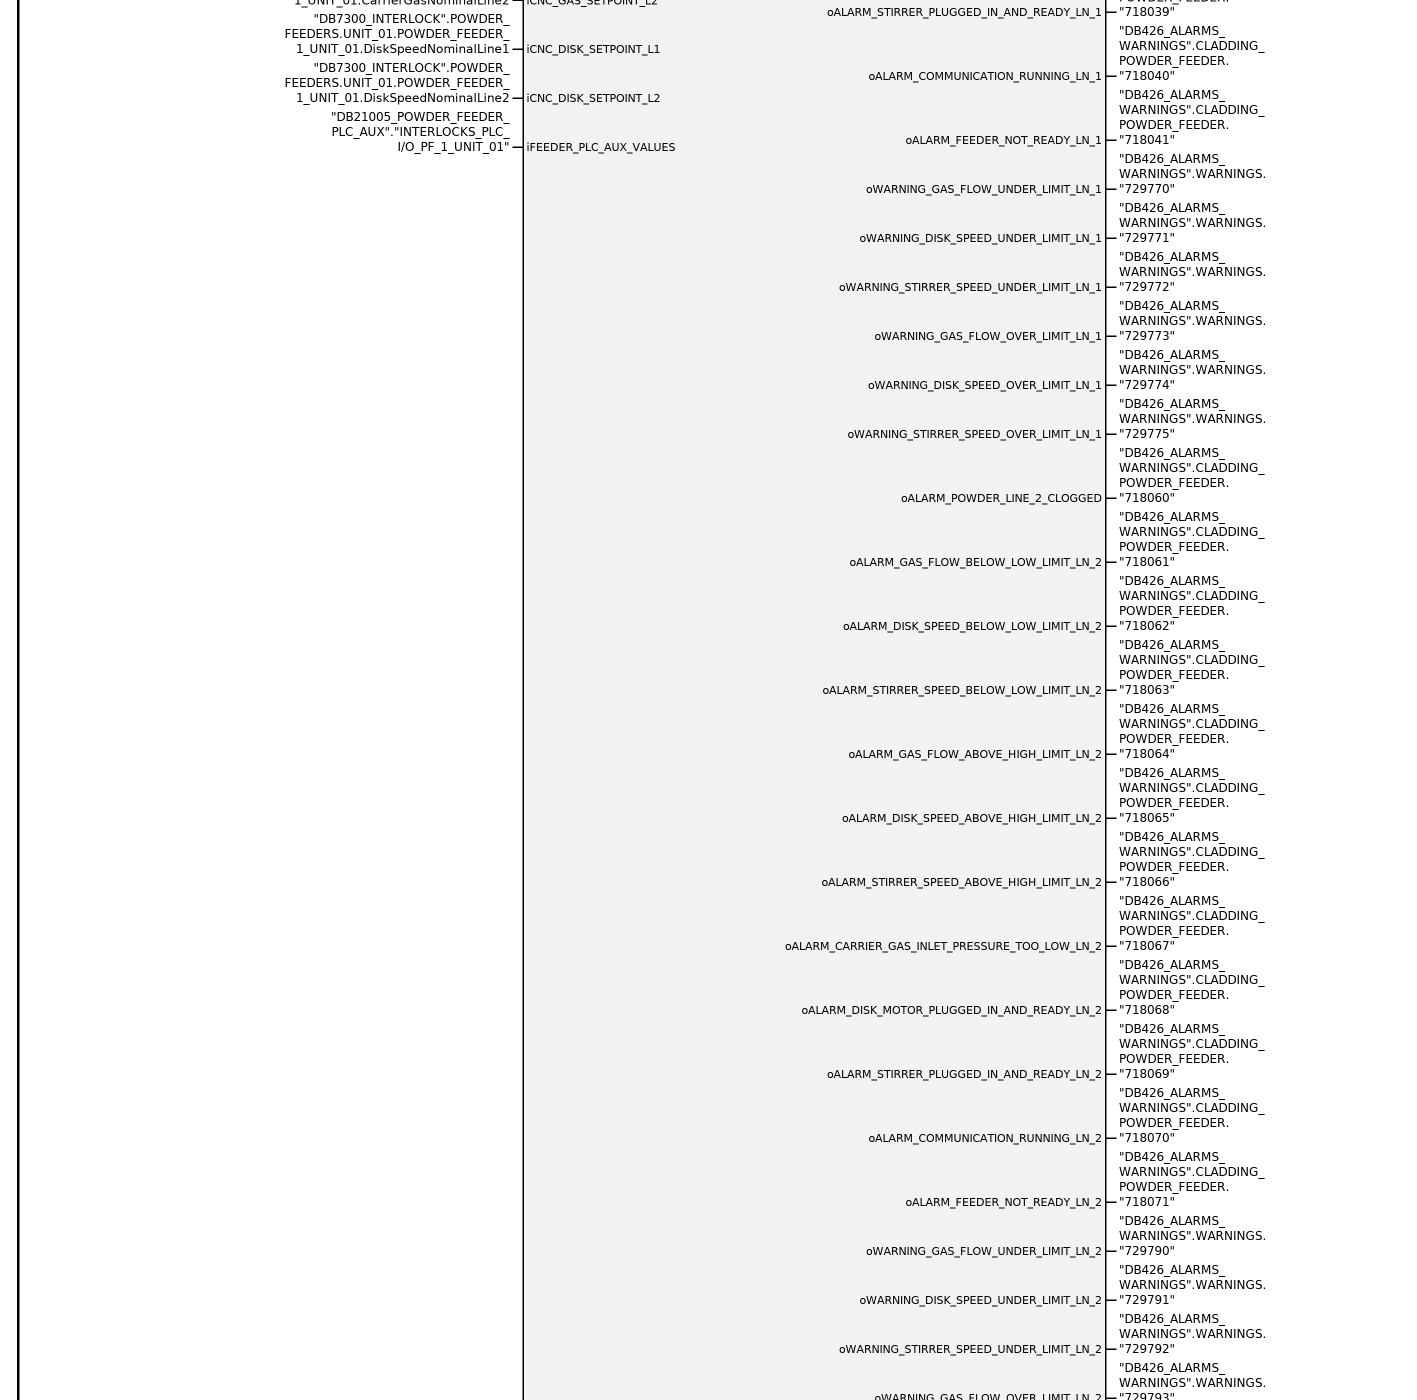
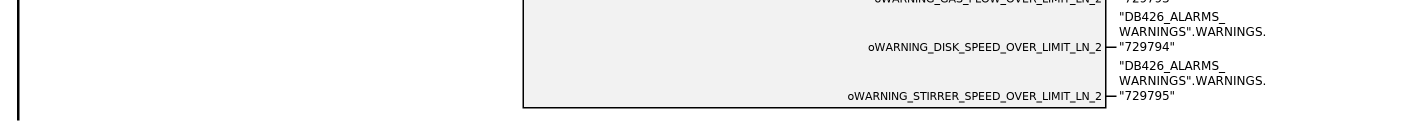
   RUNG wire#powerrail
      "DB21013_PF_1_HOPPERS_UNIT_01"(iGENERAL_CONDITIONS := wire#w1, OPTIONS_0 := 2#0000_0011, iPF_LINE_1_NOT_READY_FAULT := "DB21000_POWDER_FEEDER_GENERAL".POWDER_FEEDER_1_UNIT_01."FEEDER LINE 1 NOT READY FAULT", iPF_PROFINET_MODE_ACTIVE_FAULT_LINE_1 := "DB21000_POWDER_FEEDER_GENERAL".POWDER_FEEDER_1_UNIT_01."FEEDER PROFINET MODE ACTIVE", iPF_LINE_2_NOT_READY_FAULT := "DB21000_POWDER_FEEDER_GENERAL".POWDER_FEEDER_1_UNIT_01."FEEDER LINE 2 NOT READY FAULT", iMANUAL_START_REQ_LINE_1 := "DB7238_VARIABLES_PLC_CONNECTION".FEEDER_1_U_01_LINE_1.HOPPER_ON_MANUAL_REQUEST, iMANUAL_START_REQ_LINE_2 := "DB7238_VARIABLES_PLC_CONNECTION".FEEDER_1_U_01_LINE_2.HOPPER_ON_MANUAL_REQUEST, iMANUAL_STOP_REQ_LINE_1 := "DB7238_VARIABLES_PLC_CONNECTION".FEEDER_1_U_01_LINE_1.HOPPER_OFF_MANUAL_REQUEST, iMANUAL_STOP_REQ_LINE_2 := "DB7238_VARIABLES_PLC_CONNECTION".FEEDER_1_U_01_LINE_2.HOPPER_OFF_MANUAL_REQUEST, iPF_INTERLOCK_INPUTS := "DB21002_POWDER_FEEDER_OERLIKON_INTERLOCK".POWDER_FEEDER_1_UNIT_01.Inputs, iFEEDER_PROFINET_MODE_ACTIVE := "DB21000_POWDER_FEEDER_GENERAL".POWDER_FEEDER_1_UNIT_01."FEEDER PROFINET MODE ACTIVE", iCONTROL_ON_DELAYED := "DB2140_HOPPERS_MPP".MACHINE_ON_DELAYED, iAUTO_START_REQUEST := "DB7300_INTERLOCK".POWDER_FEEDERS.UNIT_01.SWITCH_ON_POWDER_UNIT_01, iAUTO_STOP_REQUEST := "DB7300_INTERLOCK".POWDER_FEEDERS.UNIT_01.SWITCH_OFF_POWDER_UNIT_01, iHMI_GAS_SETPOINT_L1 := "DB21003_POWDER_FEEDER_HMI_INTERLOCK".POWDER_FEEDER_1_UNIT_01."HMI_Values Setpoints".CarrierGasNominalLine1, iHMI_GAS_SETPOINT_L2 := "DB21003_POWDER_FEEDER_HMI_INTERLOCK".POWDER_FEEDER_1_UNIT_01."HMI_Values Setpoints".CarrierGasNominalLine2, iHMI_DISK_SETPOINT_L1 := "DB21003_POWDER_FEEDER_HMI_INTERLOCK".POWDER_FEEDER_1_UNIT_01."HMI_Values Setpoints".DiskSpeedNominalLine1, iHMI_DISK_SETPOINT_L2 := "DB21003_POWDER_FEEDER_HMI_INTERLOCK".POWDER_FEEDER_1_UNIT_01."HMI_Values Setpoints".DiskSpeedNominalLine2, iCNC_GAS_SETPOINT_L1 := "DB7300_INTERLOCK".POWDER_FEEDERS.UNIT_01.POWDER_FEEDER_1_UNIT_01.CarrierGasNominalLine1, iCNC_GAS_SETPOINT_L2 := "DB7300_INTERLOCK".POWDER_FEEDERS.UNIT_01.POWDER_FEEDER_1_UNIT_01.CarrierGasNominalLine2, iCNC_DISK_SETPOINT_L1 := "DB7300_INTERLOCK".POWDER_FEEDERS.UNIT_01.POWDER_FEEDER_1_UNIT_01.DiskSpeedNominalLine1, iCNC_DISK_SETPOINT_L2 := "DB7300_INTERLOCK".POWDER_FEEDERS.UNIT_01.POWDER_FEEDER_1_UNIT_01.DiskSpeedNominalLine2, iFEEDER_PLC_AUX_VALUES := "DB21005_POWDER_FEEDER_PLC_AUX"."INTERLOCKS_PLC_I/O_PF_1_UNIT_01", oSTATION_IS_ALARMS =>, oSTATION_WARNINGS =>, o_fShutdownToPF_Line1 => "DB21002_POWDER_FEEDER_OERLIKON_INTERLOCK".POWDER_FEEDER_1_UNIT_01.Outputs.o_fShutdownToPF_Line1, o_fShutdownToPF_Line2 => "DB21002_POWDER_FEEDER_OERLIKON_INTERLOCK".POWDER_FEEDER_1_UNIT_01.Outputs.o_fShutdownToPF_Line2, o_fFeedingAllOnCmd_Line1 => "DB21002_POWDER_FEEDER_OERLIKON_INTERLOCK".POWDER_FEEDER_1_UNIT_01.Outputs.o_fFeedingAllOnCmd_Line1, o_fFeedingAllOnCmd_Line2 => "DB21002_POWDER_FEEDER_OERLIKON_INTERLOCK".POWDER_FEEDER_1_UNIT_01.Outputs.o_fFeedingAllOnCmd_Line2, o_fCarriergasOnCmd_Line1 => "DB21002_POWDER_FEEDER_OERLIKON_INTERLOCK".POWDER_FEEDER_1_UNIT_01.Outputs.o_fCarriergasOnCmd_Line1, o_fCarriergasOnCmd_Line2 => "DB21002_POWDER_FEEDER_OERLIKON_INTERLOCK".POWDER_FEEDER_1_UNIT_01.Outputs.o_fCarriergasOnCmd_Line2, o_fFeedingAllOffCmd_Line1 => "DB21002_POWDER_FEEDER_OERLIKON_INTERLOCK".POWDER_FEEDER_1_UNIT_01.Outputs.o_fFeedingAllOffCmd_Line1, o_fFeedingAllOffCmd_Line2 => "DB21002_POWDER_FEEDER_OERLIKON_INTERLOCK".POWDER_FEEDER_1_UNIT_01.Outputs.o_fFeedingAllOffCmd_Line2, o_fCarriergasOffCmd_Line1 => "DB21002_POWDER_FEEDER_OERLIKON_INTERLOCK".POWDER_FEEDER_1_UNIT_01.Outputs.o_fCarriergasOffCmd_Line1, o_fCarriergasOffCmd_Line2 => "DB21002_POWDER_FEEDER_OERLIKON_INTERLOCK".POWDER_FEEDER_1_UNIT_01.Outputs.o_fCarriergasOffCmd_Line2, oALARM_POWDER_LINE_1_CLOGGED => "DB426_ALARMS_WARNINGS".CLADDING_POWDER_FEEDER."718030", oALARM_GAS_FLOW_BELOW_LOW_LIMIT_LN_1 => "DB426_ALARMS_WARNINGS".CLADDING_POWDER_FEEDER."718031", oALARM_DISK_SPEED_BELOW_LOW_LIMIT_LN_1 => "DB426_ALARMS_WARNINGS".CLADDING_POWDER_FEEDER."718032", oALARM_STIRRER_SPEED_BELOW_LOW_LIMIT_LN_1 => "DB426_ALARMS_WARNINGS".CLADDING_POWDER_FEEDER."718033", oALARM_GAS_FLOW_ABOVE_HIGH_LIMIT_LN_1 => "DB426_ALARMS_WARNINGS".CLADDING_POWDER_FEEDER."718034", oALARM_DISK_SPEED_ABOVE_HIGH_LIMIT_LN_1 => "DB426_ALARMS_WARNINGS".CLADDING_POWDER_FEEDER."718035", oALARM_STIRRER_SPEED_ABOVE_HIGH_LIMIT_LN_1 => "DB426_ALARMS_WARNINGS".CLADDING_POWDER_FEEDER."718036", oALARM_CARRIER_GAS_INLET_PRESSURE_TOO_LOW_LN_1 => "DB426_ALARMS_WARNINGS".CLADDING_POWDER_FEEDER."718037", oALARM_DISK_MOTOR_PLUGGED_IN_AND_READY_LN_1 => "DB426_ALARMS_WARNINGS".CLADDING_POWDER_FEEDER."718038", oALARM_STIRRER_PLUGGED_IN_AND_READY_LN_1 => "DB426_ALARMS_WARNINGS".CLADDING_POWDER_FEEDER."718039", oALARM_COMMUNICATION_RUNNING_LN_1 => "DB426_ALARMS_WARNINGS".CLADDING_POWDER_FEEDER."718040", oALARM_FEEDER_NOT_READY_LN_1 => "DB426_ALARMS_WARNINGS".CLADDING_POWDER_FEEDER."718041", oWARNING_GAS_FLOW_UNDER_LIMIT_LN_1 => "DB426_ALARMS_WARNINGS".WARNINGS."729770", oWARNING_DISK_SPEED_UNDER_LIMIT_LN_1 => "DB426_ALARMS_WARNINGS".WARNINGS."729771", oWARNING_STIRRER_SPEED_UNDER_LIMIT_LN_1 => "DB426_ALARMS_WARNINGS".WARNINGS."729772", oWARNING_GAS_FLOW_OVER_LIMIT_LN_1 => "DB426_ALARMS_WARNINGS".WARNINGS."729773", oWARNING_DISK_SPEED_OVER_LIMIT_LN_1 => "DB426_ALARMS_WARNINGS".WARNINGS."729774", oWARNING_STIRRER_SPEED_OVER_LIMIT_LN_1 => "DB426_ALARMS_WARNINGS".WARNINGS."729775", oALARM_POWDER_LINE_2_CLOGGED => "DB426_ALARMS_WARNINGS".CLADDING_POWDER_FEEDER."718060", oALARM_GAS_FLOW_BELOW_LOW_LIMIT_LN_2 => "DB426_ALARMS_WARNINGS".CLADDING_POWDER_FEEDER."718061", oALARM_DISK_SPEED_BELOW_LOW_LIMIT_LN_2 => "DB426_ALARMS_WARNINGS".CLADDING_POWDER_FEEDER."718062", oALARM_STIRRER_SPEED_BELOW_LOW_LIMIT_LN_2 => "DB426_ALARMS_WARNINGS".CLADDING_POWDER_FEEDER."718063", oALARM_GAS_FLOW_ABOVE_HIGH_LIMIT_LN_2 => "DB426_ALARMS_WARNINGS".CLADDING_POWDER_FEEDER."718064", oALARM_DISK_SPEED_ABOVE_HIGH_LIMIT_LN_2 => "DB426_ALARMS_WARNINGS".CLADDING_POWDER_FEEDER."718065", oALARM_STIRRER_SPEED_ABOVE_HIGH_LIMIT_LN_2 => "DB426_ALARMS_WARNINGS".CLADDING_POWDER_FEEDER."718066", oALARM_CARRIER_GAS_INLET_PRESSURE_TOO_LOW_LN_2 => "DB426_ALARMS_WARNINGS".CLADDING_POWDER_FEEDER."718067", oALARM_DISK_MOTOR_PLUGGED_IN_AND_READY_LN_2 => "DB426_ALARMS_WARNINGS".CLADDING_POWDER_FEEDER."718068", oALARM_STIRRER_PLUGGED_IN_AND_READY_LN_2 => "DB426_ALARMS_WARNINGS".CLADDING_POWDER_FEEDER."718069", oALARM_COMMUNICATION_RUNNING_LN_2 => "DB426_ALARMS_WARNINGS".CLADDING_POWDER_FEEDER."718070", oALARM_FEEDER_NOT_READY_LN_2 => "DB426_ALARMS_WARNINGS".CLADDING_POWDER_FEEDER."718071", oWARNING_GAS_FLOW_UNDER_LIMIT_LN_2 => "DB426_ALARMS_WARNINGS".WARNINGS."729790", oWARNING_DISK_SPEED_UNDER_LIMIT_LN_2 => "DB426_ALARMS_WARNINGS".WARNINGS."729791", oWARNING_STIRRER_SPEED_UNDER_LIMIT_LN_2 => "DB426_ALARMS_WARNINGS".WARNINGS."729792", oWARNING_GAS_FLOW_OVER_LIMIT_LN_2 => "DB426_ALARMS_WARNINGS".WARNINGS."729793", oWARNING_DISK_SPEED_OVER_LIMIT_LN_2 => "DB426_ALARMS_WARNINGS".WARNINGS."729794", oWARNING_STIRRER_SPEED_OVER_LIMIT_LN_2 => "DB426_ALARMS_WARNINGS".WARNINGS."729795")
   END_RUNG
   RUNG wire#powerrail
      Contact( "DB1018_POWDER_NCU_SAFE_SIGNALS".SAFE_GATES_UNIT01_FROM_NCU )
      Contact( "DB7300_INTERLOCK".GENERAL.ASPIRATION_UNIT_01_OK )
      Contact( "DB7300_INTERLOCK".POWDER_FEEDERS.UNIT_01.U01_PF1_CONDITIONS_OK )
   END_RUNG wire#w1
   // the same network as SCL:
   "DB21013_PF_1_HOPPERS_UNIT_01"(OPTIONS_0 := 2#0000_0011,   // "FB21013_POWDER_FEEDER_HOPPER"
                           iGENERAL_CONDITIONS := "DB1018_POWDER_NCU_SAFE_SIGNALS".SAFE_GATES_UNIT01_FROM_NCU AND "DB7300_INTERLOCK".GENERAL.ASPIRATION_UNIT_01_OK AND "DB7300_INTERLOCK".POWDER_FEEDERS.UNIT_01.U01_PF1_CONDITIONS_OK,
                           iPF_LINE_1_NOT_READY_FAULT := "DB21000_POWDER_FEEDER_GENERAL".POWDER_FEEDER_1_UNIT_01."FEEDER LINE 1 NOT READY FAULT",
                           iPF_PROFINET_MODE_ACTIVE_FAULT_LINE_1 := "DB21000_POWDER_FEEDER_GENERAL".POWDER_FEEDER_1_UNIT_01."FEEDER PROFINET MODE ACTIVE",
                           iPF_LINE_2_NOT_READY_FAULT := "DB21000_POWDER_FEEDER_GENERAL".POWDER_FEEDER_1_UNIT_01."FEEDER LINE 2 NOT READY FAULT",
                           iMANUAL_START_REQ_LINE_1 := "DB7238_VARIABLES_PLC_CONNECTION".FEEDER_1_U_01_LINE_1.HOPPER_ON_MANUAL_REQUEST,
                           iMANUAL_START_REQ_LINE_2 := "DB7238_VARIABLES_PLC_CONNECTION".FEEDER_1_U_01_LINE_2.HOPPER_ON_MANUAL_REQUEST,
                           iMANUAL_STOP_REQ_LINE_1 := "DB7238_VARIABLES_PLC_CONNECTION".FEEDER_1_U_01_LINE_1.HOPPER_OFF_MANUAL_REQUEST,
                           iMANUAL_STOP_REQ_LINE_2 := "DB7238_VARIABLES_PLC_CONNECTION".FEEDER_1_U_01_LINE_2.HOPPER_OFF_MANUAL_REQUEST,
                           iPF_INTERLOCK_INPUTS := "DB21002_POWDER_FEEDER_OERLIKON_INTERLOCK".POWDER_FEEDER_1_UNIT_01.Inputs,
                           iFEEDER_PROFINET_MODE_ACTIVE := "DB21000_POWDER_FEEDER_GENERAL".POWDER_FEEDER_1_UNIT_01."FEEDER PROFINET MODE ACTIVE",
                           iCONTROL_ON_DELAYED := "DB2140_HOPPERS_MPP".MACHINE_ON_DELAYED,
                           iAUTO_START_REQUEST := "DB7300_INTERLOCK".POWDER_FEEDERS.UNIT_01.SWITCH_ON_POWDER_UNIT_01,
                           iAUTO_STOP_REQUEST := "DB7300_INTERLOCK".POWDER_FEEDERS.UNIT_01.SWITCH_OFF_POWDER_UNIT_01,
                           iHMI_GAS_SETPOINT_L1 := "DB21003_POWDER_FEEDER_HMI_INTERLOCK".POWDER_FEEDER_1_UNIT_01."HMI_Values Setpoints".CarrierGasNominalLine1,
                           iHMI_GAS_SETPOINT_L2 := "DB21003_POWDER_FEEDER_HMI_INTERLOCK".POWDER_FEEDER_1_UNIT_01."HMI_Values Setpoints".CarrierGasNominalLine2,
                           iHMI_DISK_SETPOINT_L1 := "DB21003_POWDER_FEEDER_HMI_INTERLOCK".POWDER_FEEDER_1_UNIT_01."HMI_Values Setpoints".DiskSpeedNominalLine1,
                           iHMI_DISK_SETPOINT_L2 := "DB21003_POWDER_FEEDER_HMI_INTERLOCK".POWDER_FEEDER_1_UNIT_01."HMI_Values Setpoints".DiskSpeedNominalLine2,
                           iCNC_GAS_SETPOINT_L1 := "DB7300_INTERLOCK".POWDER_FEEDERS.UNIT_01.POWDER_FEEDER_1_UNIT_01.CarrierGasNominalLine1,
                           iCNC_GAS_SETPOINT_L2 := "DB7300_INTERLOCK".POWDER_FEEDERS.UNIT_01.POWDER_FEEDER_1_UNIT_01.CarrierGasNominalLine2,
                           iCNC_DISK_SETPOINT_L1 := "DB7300_INTERLOCK".POWDER_FEEDERS.UNIT_01.POWDER_FEEDER_1_UNIT_01.DiskSpeedNominalLine1,
                           iCNC_DISK_SETPOINT_L2 := "DB7300_INTERLOCK".POWDER_FEEDERS.UNIT_01.POWDER_FEEDER_1_UNIT_01.DiskSpeedNominalLine2,
                           iFEEDER_PLC_AUX_VALUES := "DB21005_POWDER_FEEDER_PLC_AUX"."INTERLOCKS_PLC_I/O_PF_1_UNIT_01",
                           o_fShutdownToPF_Line1 => "DB21002_POWDER_FEEDER_OERLIKON_INTERLOCK".POWDER_FEEDER_1_UNIT_01.Outputs.o_fShutdownToPF_Line1,
                           o_fShutdownToPF_Line2 => "DB21002_POWDER_FEEDER_OERLIKON_INTERLOCK".POWDER_FEEDER_1_UNIT_01.Outputs.o_fShutdownToPF_Line2,
                           o_fFeedingAllOnCmd_Line1 => "DB21002_POWDER_FEEDER_OERLIKON_INTERLOCK".POWDER_FEEDER_1_UNIT_01.Outputs.o_fFeedingAllOnCmd_Line1,
                           o_fFeedingAllOnCmd_Line2 => "DB21002_POWDER_FEEDER_OERLIKON_INTERLOCK".POWDER_FEEDER_1_UNIT_01.Outputs.o_fFeedingAllOnCmd_Line2,
                           o_fCarriergasOnCmd_Line1 => "DB21002_POWDER_FEEDER_OERLIKON_INTERLOCK".POWDER_FEEDER_1_UNIT_01.Outputs.o_fCarriergasOnCmd_Line1,
                           o_fCarriergasOnCmd_Line2 => "DB21002_POWDER_FEEDER_OERLIKON_INTERLOCK".POWDER_FEEDER_1_UNIT_01.Outputs.o_fCarriergasOnCmd_Line2,
                           o_fFeedingAllOffCmd_Line1 => "DB21002_POWDER_FEEDER_OERLIKON_INTERLOCK".POWDER_FEEDER_1_UNIT_01.Outputs.o_fFeedingAllOffCmd_Line1,
                           o_fFeedingAllOffCmd_Line2 => "DB21002_POWDER_FEEDER_OERLIKON_INTERLOCK".POWDER_FEEDER_1_UNIT_01.Outputs.o_fFeedingAllOffCmd_Line2,
                           o_fCarriergasOffCmd_Line1 => "DB21002_POWDER_FEEDER_OERLIKON_INTERLOCK".POWDER_FEEDER_1_UNIT_01.Outputs.o_fCarriergasOffCmd_Line1,
                           o_fCarriergasOffCmd_Line2 => "DB21002_POWDER_FEEDER_OERLIKON_INTERLOCK".POWDER_FEEDER_1_UNIT_01.Outputs.o_fCarriergasOffCmd_Line2,
                           oALARM_POWDER_LINE_1_CLOGGED => "DB426_ALARMS_WARNINGS".CLADDING_POWDER_FEEDER."718030",
                           oALARM_GAS_FLOW_BELOW_LOW_LIMIT_LN_1 => "DB426_ALARMS_WARNINGS".CLADDING_POWDER_FEEDER."718031",
                           oALARM_DISK_SPEED_BELOW_LOW_LIMIT_LN_1 => "DB426_ALARMS_WARNINGS".CLADDING_POWDER_FEEDER."718032",
                           oALARM_STIRRER_SPEED_BELOW_LOW_LIMIT_LN_1 => "DB426_ALARMS_WARNINGS".CLADDING_POWDER_FEEDER."718033",
                           oALARM_GAS_FLOW_ABOVE_HIGH_LIMIT_LN_1 => "DB426_ALARMS_WARNINGS".CLADDING_POWDER_FEEDER."718034",
                           oALARM_DISK_SPEED_ABOVE_HIGH_LIMIT_LN_1 => "DB426_ALARMS_WARNINGS".CLADDING_POWDER_FEEDER."718035",
                           oALARM_STIRRER_SPEED_ABOVE_HIGH_LIMIT_LN_1 => "DB426_ALARMS_WARNINGS".CLADDING_POWDER_FEEDER."718036",
                           oALARM_CARRIER_GAS_INLET_PRESSURE_TOO_LOW_LN_1 => "DB426_ALARMS_WARNINGS".CLADDING_POWDER_FEEDER."718037",
                           oALARM_DISK_MOTOR_PLUGGED_IN_AND_READY_LN_1 => "DB426_ALARMS_WARNINGS".CLADDING_POWDER_FEEDER."718038",
                           oALARM_STIRRER_PLUGGED_IN_AND_READY_LN_1 => "DB426_ALARMS_WARNINGS".CLADDING_POWDER_FEEDER."718039",
                           oALARM_COMMUNICATION_RUNNING_LN_1 => "DB426_ALARMS_WARNINGS".CLADDING_POWDER_FEEDER."718040",
                           oALARM_FEEDER_NOT_READY_LN_1 => "DB426_ALARMS_WARNINGS".CLADDING_POWDER_FEEDER."718041",
                           oWARNING_GAS_FLOW_UNDER_LIMIT_LN_1 => "DB426_ALARMS_WARNINGS".WARNINGS."729770",
                           oWARNING_DISK_SPEED_UNDER_LIMIT_LN_1 => "DB426_ALARMS_WARNINGS".WARNINGS."729771",
                           oWARNING_STIRRER_SPEED_UNDER_LIMIT_LN_1 => "DB426_ALARMS_WARNINGS".WARNINGS."729772",
                           oWARNING_GAS_FLOW_OVER_LIMIT_LN_1 => "DB426_ALARMS_WARNINGS".WARNINGS."729773",
                           oWARNING_DISK_SPEED_OVER_LIMIT_LN_1 => "DB426_ALARMS_WARNINGS".WARNINGS."729774",
                           oWARNING_STIRRER_SPEED_OVER_LIMIT_LN_1 => "DB426_ALARMS_WARNINGS".WARNINGS."729775",
                           oALARM_POWDER_LINE_2_CLOGGED => "DB426_ALARMS_WARNINGS".CLADDING_POWDER_FEEDER."718060",
                           oALARM_GAS_FLOW_BELOW_LOW_LIMIT_LN_2 => "DB426_ALARMS_WARNINGS".CLADDING_POWDER_FEEDER."718061",
                           oALARM_DISK_SPEED_BELOW_LOW_LIMIT_LN_2 => "DB426_ALARMS_WARNINGS".CLADDING_POWDER_FEEDER."718062",
                           oALARM_STIRRER_SPEED_BELOW_LOW_LIMIT_LN_2 => "DB426_ALARMS_WARNINGS".CLADDING_POWDER_FEEDER."718063",
                           oALARM_GAS_FLOW_ABOVE_HIGH_LIMIT_LN_2 => "DB426_ALARMS_WARNINGS".CLADDING_POWDER_FEEDER."718064",
                           oALARM_DISK_SPEED_ABOVE_HIGH_LIMIT_LN_2 => "DB426_ALARMS_WARNINGS".CLADDING_POWDER_FEEDER."718065",
                           oALARM_STIRRER_SPEED_ABOVE_HIGH_LIMIT_LN_2 => "DB426_ALARMS_WARNINGS".CLADDING_POWDER_FEEDER."718066",
                           oALARM_CARRIER_GAS_INLET_PRESSURE_TOO_LOW_LN_2 => "DB426_ALARMS_WARNINGS".CLADDING_POWDER_FEEDER."718067",
                           oALARM_DISK_MOTOR_PLUGGED_IN_AND_READY_LN_2 => "DB426_ALARMS_WARNINGS".CLADDING_POWDER_FEEDER."718068",
                           oALARM_STIRRER_PLUGGED_IN_AND_READY_LN_2 => "DB426_ALARMS_WARNINGS".CLADDING_POWDER_FEEDER."718069",
                           oALARM_COMMUNICATION_RUNNING_LN_2 => "DB426_ALARMS_WARNINGS".CLADDING_POWDER_FEEDER."718070",
                           oALARM_FEEDER_NOT_READY_LN_2 => "DB426_ALARMS_WARNINGS".CLADDING_POWDER_FEEDER."718071",
                           oWARNING_GAS_FLOW_UNDER_LIMIT_LN_2 => "DB426_ALARMS_WARNINGS".WARNINGS."729790",
                           oWARNING_DISK_SPEED_UNDER_LIMIT_LN_2 => "DB426_ALARMS_WARNINGS".WARNINGS."729791",
                           oWARNING_STIRRER_SPEED_UNDER_LIMIT_LN_2 => "DB426_ALARMS_WARNINGS".WARNINGS."729792",
                           oWARNING_GAS_FLOW_OVER_LIMIT_LN_2 => "DB426_ALARMS_WARNINGS".WARNINGS."729793",
                           oWARNING_DISK_SPEED_OVER_LIMIT_LN_2 => "DB426_ALARMS_WARNINGS".WARNINGS."729794",
                           oWARNING_STIRRER_SPEED_OVER_LIMIT_LN_2 => "DB426_ALARMS_WARNINGS".WARNINGS."729795");
END_REGION

REGION Network 3: /////_UNIT_02_/////
END_REGION

